// TwinCAT 3 PLC project _710_Clamping
// ProgramVersion: 3.1.4024.0
// libraries:
//   Tc2_Standard, * (Beckhoff Automation GmbH)
//   Tc2_System, * (Beckhoff Automation GmbH)
//   Tc3_Module, * (Beckhoff Automation GmbH)
//   VisuDialogs, * (System)
//   VisuSymbols,3.5.10.0,System
// project tree:
//   / GlobalTextList.TcGTLO, PlcTask.TcTTO, Visualization Manager.TcVMO (not stored)
//   GVLs/ Inputs.TcGVL, OP_Memory_DB.TcGVL, Outputs.TcGVL, ROBOT.TcGVL
//   GVLs/PARAMETER/ TRIAL.TcGVL
//   POUs/BIW/ Callblocks.TcPOU, Clamp.TcPOU, Fixture.TcPOU, MHRobot.TcPOU, ROLLER_DOOR.TcPOU, Trunion.TcPOU, Turntable.TcPOU, WeldRobot.TcPOU
//   POUs/ CLAMP_PROCESS.TcPOU, FEEDBACK_FB.TcPOU, FiX_1.TcTLO, MAIN.TcPOU, BLOCK_CALL.TcPOU, MODE_CONTROL.TcPOU, RollerDoor.TcPOU, SENSOR.TcPOU, TRUNION_FB.TcPOU, TURNTABLE_2POS.TcPOU, WELD_ROBOT.TcPOU, MH_ROBOT.TcPOU
//   VISUs/ AUTO_PROCESS.TcVIS, Visualization.TcVIS
// real-time tasks:
//   TASK PlcTask: cycle T#10ms, priority 20, ADS port 350

CONFIGURATION _710_Clamping
    RESOURCE PLC ON TwinCAT3
        TASK PlcTask(INTERVAL := T#10ms, PRIORITY := 20);
        PROGRAM MAIN WITH PlcTask : MAIN;
    END_RESOURCE
END_CONFIGURATION

// ---- GVLs/Inputs.TcGVL
{attribute 'qualified_only'}
VAR_GLOBAL



	i_CC1_Clamp_3_Sensor_HP : BOOL;
	i_CC1_Clamp_3_Sensor_WP : BOOL;
	i_CC1_Clamp_2_Sensor_HP : BOOL;
	i_CC1_Clamp_2_Sensor_WP : BOOL;
	i_CC1_Clamp_1_Sensor_HP : BOOL;
	i_CC1_Clamp_1_Sensor_WP : BOOL;
	i_CC6_Clamp_1_Sensor_HP : BOOL;
	i_CC6_Clamp_1_Sensor_WP : BOOL;
	i_CC4_Clamp_3_Sensor_HP : BOOL;
	i_CC4_Clamp_3_Sensor_WP : BOOL;
	i_PART_CONTROL_B13      : BOOL;
	i_PART_CONTROL_B27      : BOOL;
	i_PART_CONTROL_B14      : BOOL;
	i_PART_CONTROL_B28      : BOOL;
	i_CC4_Clamp_2_Sensor_HP : BOOL;
	i_CC4_Clamp_2_Sensor_WP : BOOL;
	i_CC4_Clamp_1_Sensor_HP : BOOL;
	i_CC4_Clamp_1_Sensor_WP : BOOL;
	i_CC2_Clamp_3_Sensor_HP : BOOL;
	i_CC2_Clamp_3_Sensor_WP : BOOL;
	i_PART_CONTROL_B12      : BOOL;
	i_PART_CONTROL_B26      : BOOL;
	i_PART_CONTROL_B11      : BOOL;
	i_PART_CONTROL_B25      : BOOL;
	i_PART_CONTROL_B10      : BOOL;
	i_PART_CONTROL_B24      : BOOL;
	i_CC3_Clamp_3_Sensor_HP : BOOL;
	i_CC3_Clamp_3_Sensor_WP : BOOL;
	i_CC3_Clamp_2_Sensor_HP : BOOL;
	i_CC3_Clamp_2_Sensor_WP : BOOL;
	i_CC3_Clamp_1_Sensor_HP : BOOL;
	i_CC3_Clamp_1_Sensor_WP : BOOL;
	i_PART_CONTROL_B7       : BOOL;
	i_PART_CONTROL_B21      : BOOL;
	i_PART_CONTROL_B6       : BOOL;
	i_PART_CONTROL_B20      : BOOL;
	i_PART_CONTROL_B5       : BOOL;
	i_PART_CONTROL_B19      : BOOL;
	i_PART_CONTROL_B4       : BOOL;
	i_PART_CONTROL_B18      : BOOL;
	i_PART_CONTROL_B3       : BOOL;
	i_PART_CONTROL_B17      : BOOL;
	i_PART_CONTROL_B2       : BOOL;
	i_PART_CONTROL_B16      : BOOL;
	i_CC2_Clamp_2_Sensor_HP : BOOL;
	i_CC2_Clamp_2_Sensor_WP : BOOL;
	i_CC2_Clamp_1_Sensor_HP : BOOL;
	i_CC2_Clamp_1_Sensor_WP : BOOL;
	i_PART_CONTROL_B9       : BOOL;
	i_PART_CONTROL_B23      : BOOL;
	i_PART_CONTROL_B8       : BOOL;
	i_PART_CONTROL_B22      : BOOL;
	i_CC5_Clamp_1_Sensor_HP : BOOL;
	i_CC5_Clamp_1_Sensor_WP : BOOL;
	i_PART_CONTROL_B1       : BOOL;
	i_PART_CONTROL_B15      : BOOL;
	i_Reset_PB              : BOOL;
	i_OPERATE_START_PB      : BOOL;
	i_CYCLE_START_PB        : BOOL;
    i_STOP_PB               : BOOL;
	//TT SENSOR
	i_1st_TT_Pos             : BOOL;
	i_2nd_TT_Pos             : BOOL;
	i_Drive_1_Ready         : BOOL;
	// TRUNION
	i_Drive_1_TT_Ready      : BOOL;
	i_Trunion_1st_Pos       : BOOL;
	i_Trunion_2nd_Pos       : BOOL;
	// ROLLER DOOR
	i_ROLL_DR_1_TT_Ready    : BOOL;
	i_ROLL_DR_Open_Pos_LS   : BOOL;
	i_ROLL_DR_Close_Pos_LS  : BOOL;
	//ROBOT_WELD
	Robot_Ready             : BOOL;
	Robot_Busy              : BOOL;
	Robot_Complete          : BOOL;
	Robot_Fault             : BOOL;
	PROGRAM_NUMBER          : INT;
	 //MH_ROBOT
	
	MH_Robot_Ready             : BOOL;
	MH_Robot_Busy              : BOOL;
	MH_Robot_Complete          : BOOL;
	MH_Robot_Fault             : BOOL;
	MH_PROGRAM_NUMBER          : INT;
	
	
END_VAR

// ---- GVLs/OP_Memory_DB.TcGVL
{attribute 'qualified_only'}
VAR_GLOBAL
	POWER_ON : BOOL;
    Auto_mode: BOOL;
	Manual_Mode: BOOL;
	TEMP : BOOL;
	
	
	M_CC1_CLAMPING_UNIT1_3_WP : BOOL;
	M_CC1_CLAMPING_UNIT1_3_HP : BOOL;
	M_CC2_CLAMPING_UNIT2_3_WP : BOOL;
	M_CC2_CLAMPING_UNIT2_3_HP : BOOL;
	M_CC3_CLAMPING_UNIT3_3_WP : BOOL;
	M_CC3_CLAMPING_UNIT3_3_HP : BOOL;
	M_CC4_CLAMPING_UNIT4_3_WP : BOOL;
	M_CC4_CLAMPING_UNIT4_3_HP : BOOL;
	M_CC5_CLAMPING_UNIT5_1_WP : BOOL;
	M_CC5_CLAMPING_UNIT5_1_HP : BOOL;
	M_CC6_CLAMPING_UNIT6_1_WP : BOOL;
	M_CC6_CLAMPING_UNIT6_1_HP : BOOL;
    A_CC1_CLAMPING_UNIT1_3_WP : BOOL;
	A_CC1_CLAMPING_UNIT1_3_HP : BOOL;
	A_CC2_CLAMPING_UNIT2_3_WP : BOOL;
	A_CC2_CLAMPING_UNIT2_3_HP : BOOL;
	A_CC3_CLAMPING_UNIT3_3_WP : BOOL;
	A_CC3_CLAMPING_UNIT3_3_HP : BOOL;
	A_CC4_CLAMPING_UNIT4_3_WP : BOOL;
	A_CC4_CLAMPING_UNIT4_3_HP : BOOL;
	A_CC5_CLAMPING_UNIT5_1_WP : BOOL;
	A_CC5_CLAMPING_UNIT5_1_HP : BOOL;
	A_CC6_CLAMPING_UNIT6_1_WP : BOOL;
	A_CC6_CLAMPING_UNIT6_1_HP : BOOL;
	TEMP_CC1_WP_FEEDBACK : BOOL;
	TEMP_CC1_HP_FEEDBACK : BOOL;
	TEMP_CC2_WP_FEEDBACK : BOOL;
	TEMP_CC2_HP_FEEDBACK : BOOL;
	TEMP_CC3_WP_FEEDBACK : BOOL;
	TEMP_CC3_HP_FEEDBACK : BOOL;
	TEMP_CC4_WP_FEEDBACK : BOOL;
	TEMP_CC4_HP_FEEDBACK : BOOL;
	TEMP_CC5_WP_FEEDBACK : BOOL;
	TEMP_CC5_HP_FEEDBACK : BOOL;
	TEMP_CC6_WP_FEEDBACK : BOOL;
	TEMP_CC6_HP_FEEDBACK : BOOL;
	A_FIX1_ALL_CLAMP_WORK : BOOL;
	A_FIX1_ALL_CLAMP_HOME : BOOL;
	A_FIX2_ALL_CLAMP_WORK : BOOL;
	A_FIX2_ALL_CLAMP_HOME : BOOL;
	M_FIX1_ALL_CLAMP_HOME_PB : BOOL;
	//SENSOR
	A_FIX1_PART_1ST : BOOL;
	A_FIX1_PART_2ND : BOOL;
	A_FIX1_PART_3RD : BOOL;
	A_FIX1_PART_4TH : BOOL;
	A_FIX1_PART_5TH : BOOL;
	A_FIX1_PART_6TH : BOOL;
	A_FIX2_PART_1ST : BOOL;
	A_FIX2_PART_2ND : BOOL;
	A_FIX2_PART_3RD : BOOL;
	A_FIX2_PART_4TH : BOOL;
	A_FIX2_PART_5TH : BOOL;
	A_FIX2_PART_6TH : BOOL;
	// TT POSITION
	M_1ST_POSITION_TT_CMD : BOOL;
	M_2ND_POSITION_TT_CMD : BOOL;
	A_1ST_POSITION_TT_CMD : BOOL;
	A_2ND_POSITION_TT_CMD : BOOL;
	A_FEEDBACK_TT_FWD : BOOL;
	A_FEEDBACK_TT_REV : BOOL;
	// Trunion POSITION
	A_Clamp_ok : BOOL;
	M_Fwd_POSITION : BOOL;
	M_Rev_POSITION : BOOL;
	A_Fwd_POSITION : BOOL;
	A_Rev_POSITION : BOOL;
	A_FEEDBACK_TRUNION_FWD : BOOL;
	A_FEEDBACK_TRUNION_REV : BOOL;
	//ROLLER DOOR
	M_Roll_Dr_Open  : BOOL;
	M_Roll_Dr_Close : BOOL;
	A_Open_CMD      : BOOL;
    A_Close_CMD     : BOOL;
	A_Safety_Beam : BOOL;
	A_FEEDBACK_RD_OPEN : BOOL;
	A_FEEDBACK_RD_CLOSE : BOOL;
	//ROBOT
	ROBOT_START : BOOL;
	SAFETY_OK : BOOL;
	ROBOT_JOG : BOOL;
	ROBOT_COMPLETE : BOOL;
	ROBOT_BUSY : BOOL;
	ROBOT_HOME : BOOL;
	TEMP_ROB : BOOL;
	//MH_ROBOT
	MH_ROBOT_START : BOOL;
	MH_SAFETY_OK : BOOL;
	MH_ROBOT_JOG : BOOL;
	MH_ROBOT_COMPLETE : BOOL;
	MH_ROBOT_BUSY : BOOL;
	MH_ROBOT_HOME : BOOL;
	MH_TEMP_ROB : BOOL;
	
	
	
END_VAR

// ---- GVLs/Outputs.TcGVL
{attribute 'qualified_only'}
VAR_GLOBAL


	o_CC1_CLAMPING_UNIT1_3_WP : BOOL;
	o_CC1_CLAMPING_UNIT1_3_HP : BOOL;
	o_CC2_CLAMPING_UNIT2_3_WP : BOOL;
	o_CC2_CLAMPING_UNIT2_3_HP : BOOL;
	o_CC3_CLAMPING_UNIT3_3_WP : BOOL;
	o_CC3_CLAMPING_UNIT3_3_HP : BOOL;
	o_CC4_CLAMPING_UNIT4_3_WP : BOOL;
	o_CC4_CLAMPING_UNIT4_3_HP : BOOL;
	o_CC5_CLAMPING_UNIT5_1_WP : BOOL;
	o_CC5_CLAMPING_UNIT5_1_HP : BOOL;
	o_CC6_CLAMPING_UNIT6_1_WP : BOOL;
	o_CC6_CLAMPING_UNIT6_1_HP : BOOL;
	// TURN TABLE
	o_POSITION_CW_TT : BOOL;
	o_POSITION_CCW_TT : BOOL;
	//TRUNION
	o_Motor_Fwd       : BOOL;
    o_Motor_Rev       : BOOL;
	//ROLLER DOOR
	o_ROLL_DR_Open       : BOOL;
    o_ROLL_DR_Close       : BOOL;
	//Robot
	ROBOT_START : BOOL;
	ROBOT_RESET : BOOL;
	PROGRAM_0 : BOOL;
	PROGRAM_1 : BOOL;
	PROGRAM_2 : BOOL;
	PROGRAM_3 : BOOL;
	//MH_ROBOT 
	MH_ROBOT_START : BOOL;
	MH_ROBOT_RESET : BOOL;
	MH_PROGRAM_0 : BOOL;
	MH_PROGRAM_1 : BOOL;
	MH_PROGRAM_2 : BOOL;
	MH_PROGRAM_3 : BOOL;
	O_FAULT_LAMP : BOOL;
	
END_VAR

// ---- GVLs/PARAMETER/TRIAL.TcGVL
{attribute 'qualified_only'}
VAR_GLOBAL
	
END_VAR

// ---- GVLs/ROBOT.TcGVL
{attribute 'qualified_only'}
VAR_GLOBAL
	START : BOOL;
	STOP : BOOL;
	SAFETY_OK : BOOL;
END_VAR

// ---- POUs/MAIN.TcPOU
PROGRAM MAIN
VAR
END_VAR

BLOCK_CALL();

END_PROGRAM

// ---- POUs/BLOCK_CALL.TcPOU
PROGRAM BLOCK_CALL
VAR
	CLAMP_1_DB : CLAMP_PROCESS;
	CLAMP_2_DB : CLAMP_PROCESS;
	CLAMP_3_DB : CLAMP_PROCESS;
	CLAMP_4_DB : CLAMP_PROCESS;
	CLAMP_5_DB : CLAMP_PROCESS;
	CLAMP_6_DB : CLAMP_PROCESS;
	Feedback_1_DB : Feedback_FB;
	Feedback_2_DB : Feedback_FB;
	Feedback_3_DB : Feedback_FB;
	Feedback_4_DB : Feedback_FB;
	Feedback_5_DB : Feedback_FB;
	Feedback_6_DB : Feedback_FB;
	Feedback_TT1_DB : Feedback_FB;
	Feedback_Trunion_1_DB : Feedback_FB;
	TURNTABLE_2POS_DB : TURNTABLE_2POS;
	TRUNION1_DB : TRUNION_FB;
	ROLLER_DOOR_DB : ROLLER_DOOR;
	RollerDoor_DB : RollerDoor;
    Feedback_RD1_DB : Feedback_FB;
	WELD_ROBOT_DB : WELD_ROBOT;
	MH_ROBOT_DB : MH_ROBOT;
	MODE_CONTROL_DB : MODE_CONTROL;
	SENSOR_DB : SENSOR;
END_VAR

// note: this text did not pass the execution check against the stored diagram
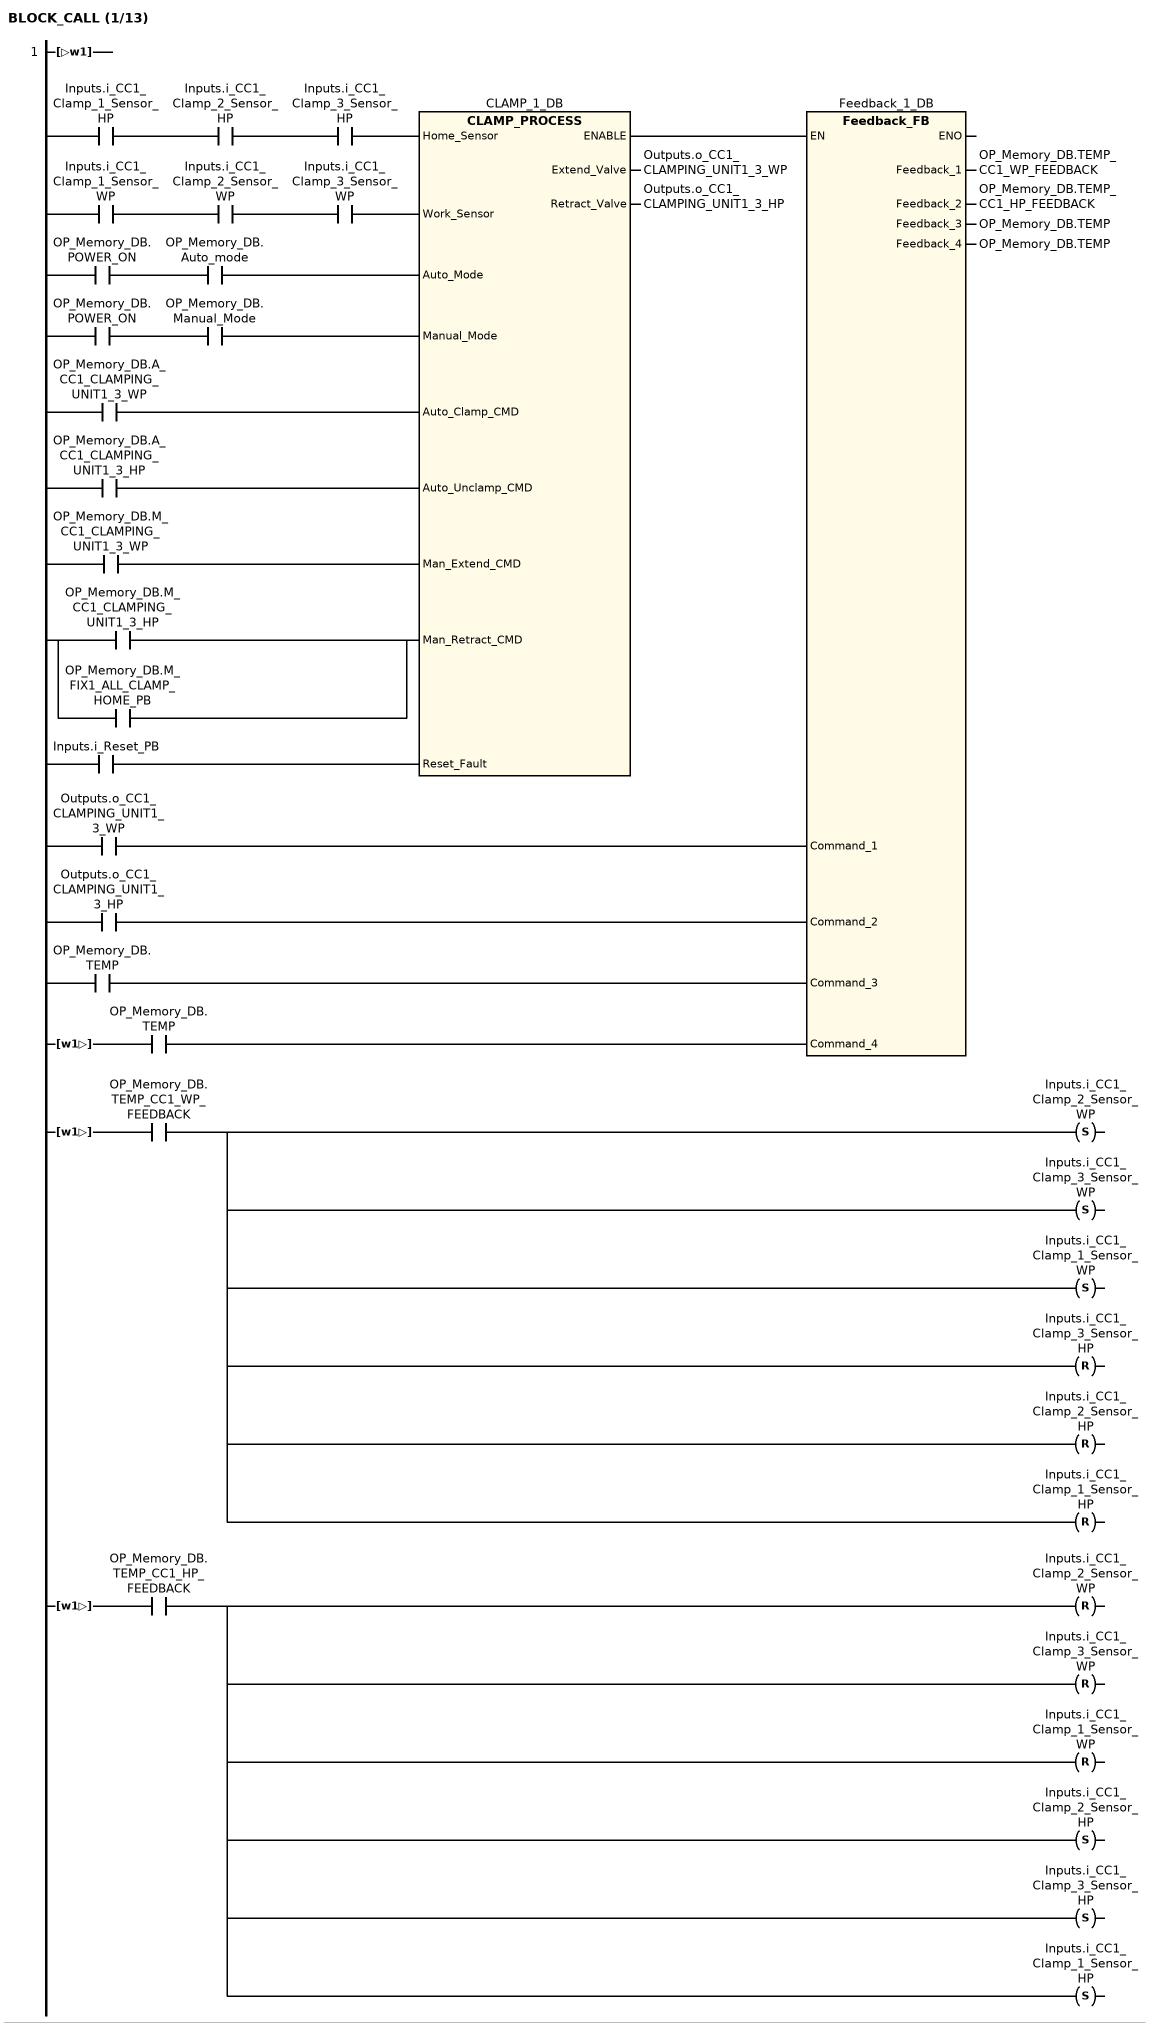
// NETWORK 1
CLAMP_1_DB(
    Home_Sensor := Inputs.i_CC1_Clamp_1_Sensor_HP AND Inputs.i_CC1_Clamp_2_Sensor_HP AND Inputs.i_CC1_Clamp_3_Sensor_HP,
    Work_Sensor := Inputs.i_CC1_Clamp_1_Sensor_WP AND Inputs.i_CC1_Clamp_2_Sensor_WP AND Inputs.i_CC1_Clamp_3_Sensor_WP,
    Auto_Mode := OP_Memory_DB.POWER_ON AND OP_Memory_DB.Auto_mode,
    Manual_Mode := OP_Memory_DB.POWER_ON AND OP_Memory_DB.Manual_Mode,
    Auto_Clamp_CMD := OP_Memory_DB.A_CC1_CLAMPING_UNIT1_3_WP,
    Auto_Unclamp_CMD := OP_Memory_DB.A_CC1_CLAMPING_UNIT1_3_HP,
    Man_Extend_CMD := OP_Memory_DB.M_CC1_CLAMPING_UNIT1_3_WP,
    Man_Retract_CMD := OP_Memory_DB.M_CC1_CLAMPING_UNIT1_3_HP OR OP_Memory_DB.M_FIX1_ALL_CLAMP_HOME_PB,
    Reset_Fault := Inputs.i_Reset_PB,
    Extend_Valve => Outputs.o_CC1_CLAMPING_UNIT1_3_WP,
    Retract_Valve => Outputs.o_CC1_CLAMPING_UNIT1_3_HP); // CLAMP_PROCESS
Feedback_1_DB(
    EN := CLAMP_1_DB.ENABLE,
    Command_1 := Outputs.o_CC1_CLAMPING_UNIT1_3_WP,
    Command_2 := Outputs.o_CC1_CLAMPING_UNIT1_3_HP,
    Command_3 := OP_Memory_DB.TEMP,
    Command_4 := OP_Memory_DB.TEMP,
    Feedback_1 => OP_Memory_DB.TEMP_CC1_WP_FEEDBACK,
    Feedback_2 => OP_Memory_DB.TEMP_CC1_HP_FEEDBACK,
    Feedback_3 => OP_Memory_DB.TEMP,
    Feedback_4 => OP_Memory_DB.TEMP); // Feedback_FB
Inputs.i_CC1_Clamp_2_Sensor_WP S= OP_Memory_DB.TEMP_CC1_WP_FEEDBACK;
Inputs.i_CC1_Clamp_3_Sensor_WP S= OP_Memory_DB.TEMP_CC1_WP_FEEDBACK;
Inputs.i_CC1_Clamp_1_Sensor_WP S= OP_Memory_DB.TEMP_CC1_WP_FEEDBACK;
Inputs.i_CC1_Clamp_3_Sensor_HP R= OP_Memory_DB.TEMP_CC1_WP_FEEDBACK;
Inputs.i_CC1_Clamp_2_Sensor_HP R= OP_Memory_DB.TEMP_CC1_WP_FEEDBACK;
Inputs.i_CC1_Clamp_1_Sensor_HP R= OP_Memory_DB.TEMP_CC1_WP_FEEDBACK;
Inputs.i_CC1_Clamp_2_Sensor_WP R= OP_Memory_DB.TEMP_CC1_HP_FEEDBACK;
Inputs.i_CC1_Clamp_3_Sensor_WP R= OP_Memory_DB.TEMP_CC1_HP_FEEDBACK;
Inputs.i_CC1_Clamp_1_Sensor_WP R= OP_Memory_DB.TEMP_CC1_HP_FEEDBACK;
Inputs.i_CC1_Clamp_2_Sensor_HP S= OP_Memory_DB.TEMP_CC1_HP_FEEDBACK;
Inputs.i_CC1_Clamp_3_Sensor_HP S= OP_Memory_DB.TEMP_CC1_HP_FEEDBACK;
Inputs.i_CC1_Clamp_1_Sensor_HP S= OP_Memory_DB.TEMP_CC1_HP_FEEDBACK;

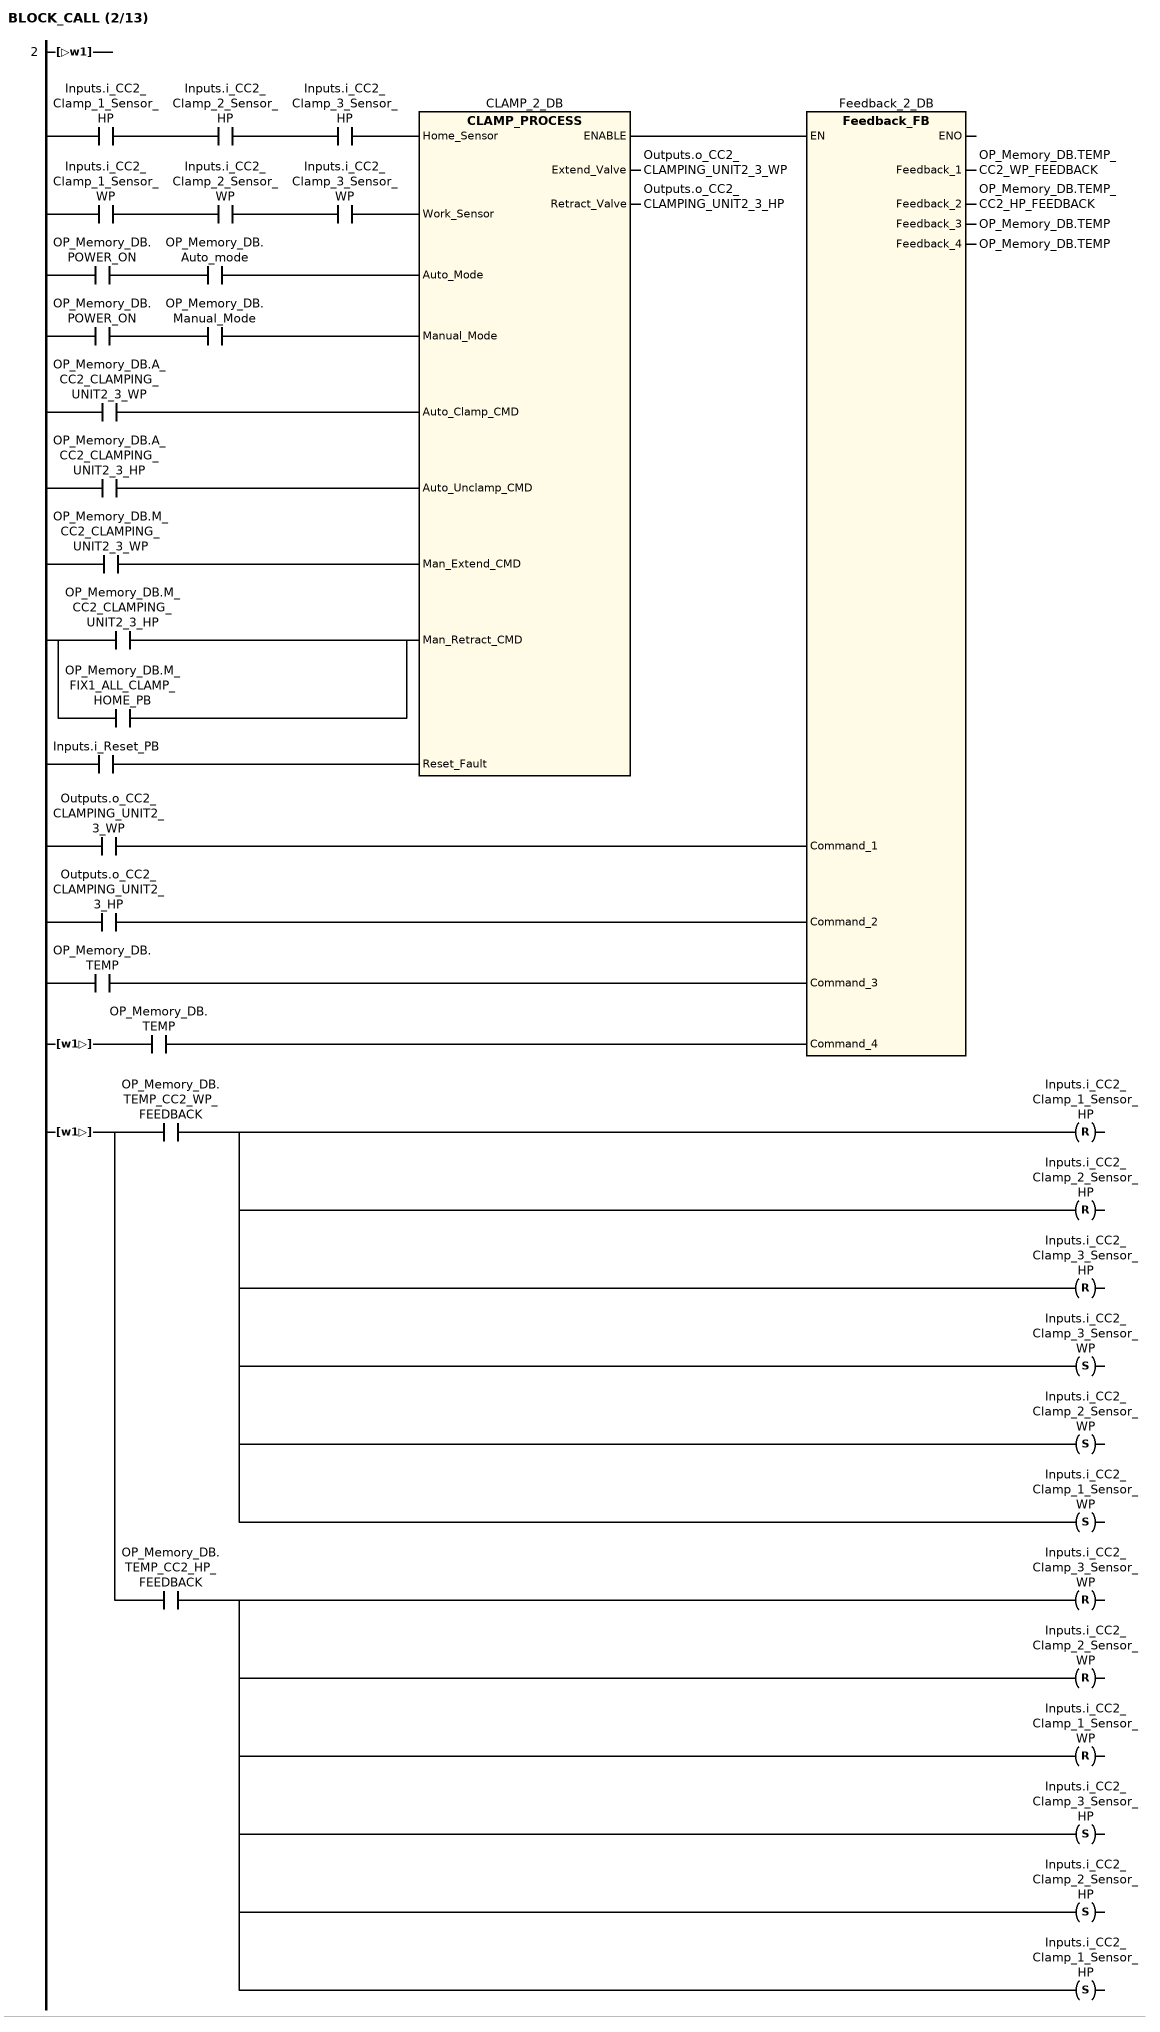
// NETWORK 2
CLAMP_2_DB(
    Home_Sensor := Inputs.i_CC2_Clamp_1_Sensor_HP AND Inputs.i_CC2_Clamp_2_Sensor_HP AND Inputs.i_CC2_Clamp_3_Sensor_HP,
    Work_Sensor := Inputs.i_CC2_Clamp_1_Sensor_WP AND Inputs.i_CC2_Clamp_2_Sensor_WP AND Inputs.i_CC2_Clamp_3_Sensor_WP,
    Auto_Mode := OP_Memory_DB.POWER_ON AND OP_Memory_DB.Auto_mode,
    Manual_Mode := OP_Memory_DB.POWER_ON AND OP_Memory_DB.Manual_Mode,
    Auto_Clamp_CMD := OP_Memory_DB.A_CC2_CLAMPING_UNIT2_3_WP,
    Auto_Unclamp_CMD := OP_Memory_DB.A_CC2_CLAMPING_UNIT2_3_HP,
    Man_Extend_CMD := OP_Memory_DB.M_CC2_CLAMPING_UNIT2_3_WP,
    Man_Retract_CMD := OP_Memory_DB.M_CC2_CLAMPING_UNIT2_3_HP OR OP_Memory_DB.M_FIX1_ALL_CLAMP_HOME_PB,
    Reset_Fault := Inputs.i_Reset_PB,
    Extend_Valve => Outputs.o_CC2_CLAMPING_UNIT2_3_WP,
    Retract_Valve => Outputs.o_CC2_CLAMPING_UNIT2_3_HP); // CLAMP_PROCESS
Feedback_2_DB(
    EN := CLAMP_2_DB.ENABLE,
    Command_1 := Outputs.o_CC2_CLAMPING_UNIT2_3_WP,
    Command_2 := Outputs.o_CC2_CLAMPING_UNIT2_3_HP,
    Command_3 := OP_Memory_DB.TEMP,
    Command_4 := OP_Memory_DB.TEMP,
    Feedback_1 => OP_Memory_DB.TEMP_CC2_WP_FEEDBACK,
    Feedback_2 => OP_Memory_DB.TEMP_CC2_HP_FEEDBACK,
    Feedback_3 => OP_Memory_DB.TEMP,
    Feedback_4 => OP_Memory_DB.TEMP); // Feedback_FB
Inputs.i_CC2_Clamp_1_Sensor_HP R= OP_Memory_DB.TEMP_CC2_WP_FEEDBACK;
Inputs.i_CC2_Clamp_2_Sensor_HP R= OP_Memory_DB.TEMP_CC2_WP_FEEDBACK;
Inputs.i_CC2_Clamp_3_Sensor_HP R= OP_Memory_DB.TEMP_CC2_WP_FEEDBACK;
Inputs.i_CC2_Clamp_3_Sensor_WP S= OP_Memory_DB.TEMP_CC2_WP_FEEDBACK;
Inputs.i_CC2_Clamp_2_Sensor_WP S= OP_Memory_DB.TEMP_CC2_WP_FEEDBACK;
Inputs.i_CC2_Clamp_1_Sensor_WP S= OP_Memory_DB.TEMP_CC2_WP_FEEDBACK;
Inputs.i_CC2_Clamp_3_Sensor_WP R= OP_Memory_DB.TEMP_CC2_HP_FEEDBACK;
Inputs.i_CC2_Clamp_2_Sensor_WP R= OP_Memory_DB.TEMP_CC2_HP_FEEDBACK;
Inputs.i_CC2_Clamp_1_Sensor_WP R= OP_Memory_DB.TEMP_CC2_HP_FEEDBACK;
Inputs.i_CC2_Clamp_3_Sensor_HP S= OP_Memory_DB.TEMP_CC2_HP_FEEDBACK;
Inputs.i_CC2_Clamp_2_Sensor_HP S= OP_Memory_DB.TEMP_CC2_HP_FEEDBACK;
Inputs.i_CC2_Clamp_1_Sensor_HP S= OP_Memory_DB.TEMP_CC2_HP_FEEDBACK;

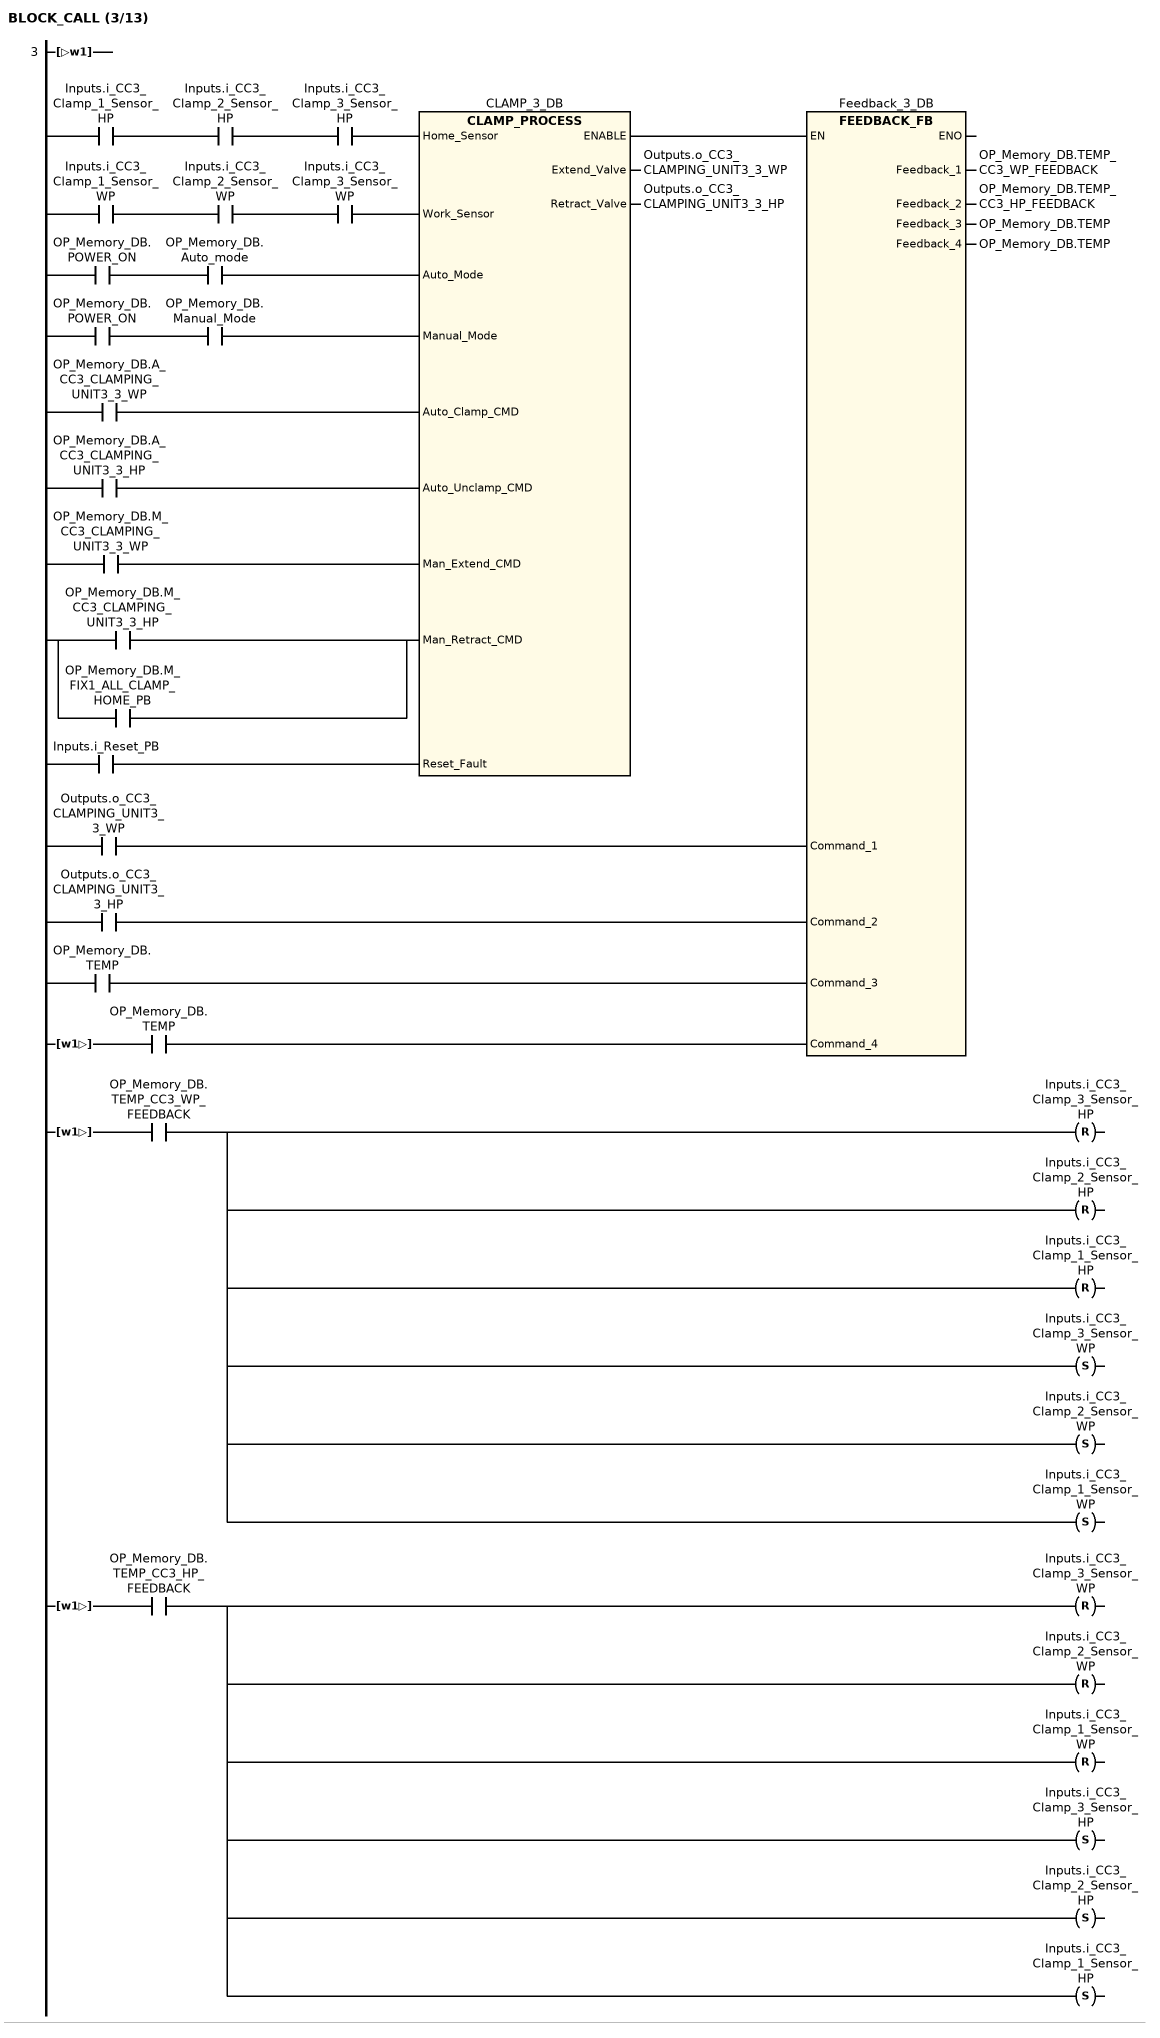
// NETWORK 3
CLAMP_3_DB(
    Home_Sensor := Inputs.i_CC3_Clamp_1_Sensor_HP AND Inputs.i_CC3_Clamp_2_Sensor_HP AND Inputs.i_CC3_Clamp_3_Sensor_HP,
    Work_Sensor := Inputs.i_CC3_Clamp_1_Sensor_WP AND Inputs.i_CC3_Clamp_2_Sensor_WP AND Inputs.i_CC3_Clamp_3_Sensor_WP,
    Auto_Mode := OP_Memory_DB.POWER_ON AND OP_Memory_DB.Auto_mode,
    Manual_Mode := OP_Memory_DB.POWER_ON AND OP_Memory_DB.Manual_Mode,
    Auto_Clamp_CMD := OP_Memory_DB.A_CC3_CLAMPING_UNIT3_3_WP,
    Auto_Unclamp_CMD := OP_Memory_DB.A_CC3_CLAMPING_UNIT3_3_HP,
    Man_Extend_CMD := OP_Memory_DB.M_CC3_CLAMPING_UNIT3_3_WP,
    Man_Retract_CMD := OP_Memory_DB.M_CC3_CLAMPING_UNIT3_3_HP OR OP_Memory_DB.M_FIX1_ALL_CLAMP_HOME_PB,
    Reset_Fault := Inputs.i_Reset_PB,
    Extend_Valve => Outputs.o_CC3_CLAMPING_UNIT3_3_WP,
    Retract_Valve => Outputs.o_CC3_CLAMPING_UNIT3_3_HP); // CLAMP_PROCESS
Feedback_3_DB(
    EN := CLAMP_3_DB.ENABLE,
    Command_1 := Outputs.o_CC3_CLAMPING_UNIT3_3_WP,
    Command_2 := Outputs.o_CC3_CLAMPING_UNIT3_3_HP,
    Command_3 := OP_Memory_DB.TEMP,
    Command_4 := OP_Memory_DB.TEMP,
    Feedback_1 => OP_Memory_DB.TEMP_CC3_WP_FEEDBACK,
    Feedback_2 => OP_Memory_DB.TEMP_CC3_HP_FEEDBACK,
    Feedback_3 => OP_Memory_DB.TEMP,
    Feedback_4 => OP_Memory_DB.TEMP); // FEEDBACK_FB
Inputs.i_CC3_Clamp_3_Sensor_HP R= OP_Memory_DB.TEMP_CC3_WP_FEEDBACK;
Inputs.i_CC3_Clamp_2_Sensor_HP R= OP_Memory_DB.TEMP_CC3_WP_FEEDBACK;
Inputs.i_CC3_Clamp_1_Sensor_HP R= OP_Memory_DB.TEMP_CC3_WP_FEEDBACK;
Inputs.i_CC3_Clamp_3_Sensor_WP S= OP_Memory_DB.TEMP_CC3_WP_FEEDBACK;
Inputs.i_CC3_Clamp_2_Sensor_WP S= OP_Memory_DB.TEMP_CC3_WP_FEEDBACK;
Inputs.i_CC3_Clamp_1_Sensor_WP S= OP_Memory_DB.TEMP_CC3_WP_FEEDBACK;
Inputs.i_CC3_Clamp_3_Sensor_WP R= OP_Memory_DB.TEMP_CC3_HP_FEEDBACK;
Inputs.i_CC3_Clamp_2_Sensor_WP R= OP_Memory_DB.TEMP_CC3_HP_FEEDBACK;
Inputs.i_CC3_Clamp_1_Sensor_WP R= OP_Memory_DB.TEMP_CC3_HP_FEEDBACK;
Inputs.i_CC3_Clamp_3_Sensor_HP S= OP_Memory_DB.TEMP_CC3_HP_FEEDBACK;
Inputs.i_CC3_Clamp_2_Sensor_HP S= OP_Memory_DB.TEMP_CC3_HP_FEEDBACK;
Inputs.i_CC3_Clamp_1_Sensor_HP S= OP_Memory_DB.TEMP_CC3_HP_FEEDBACK;

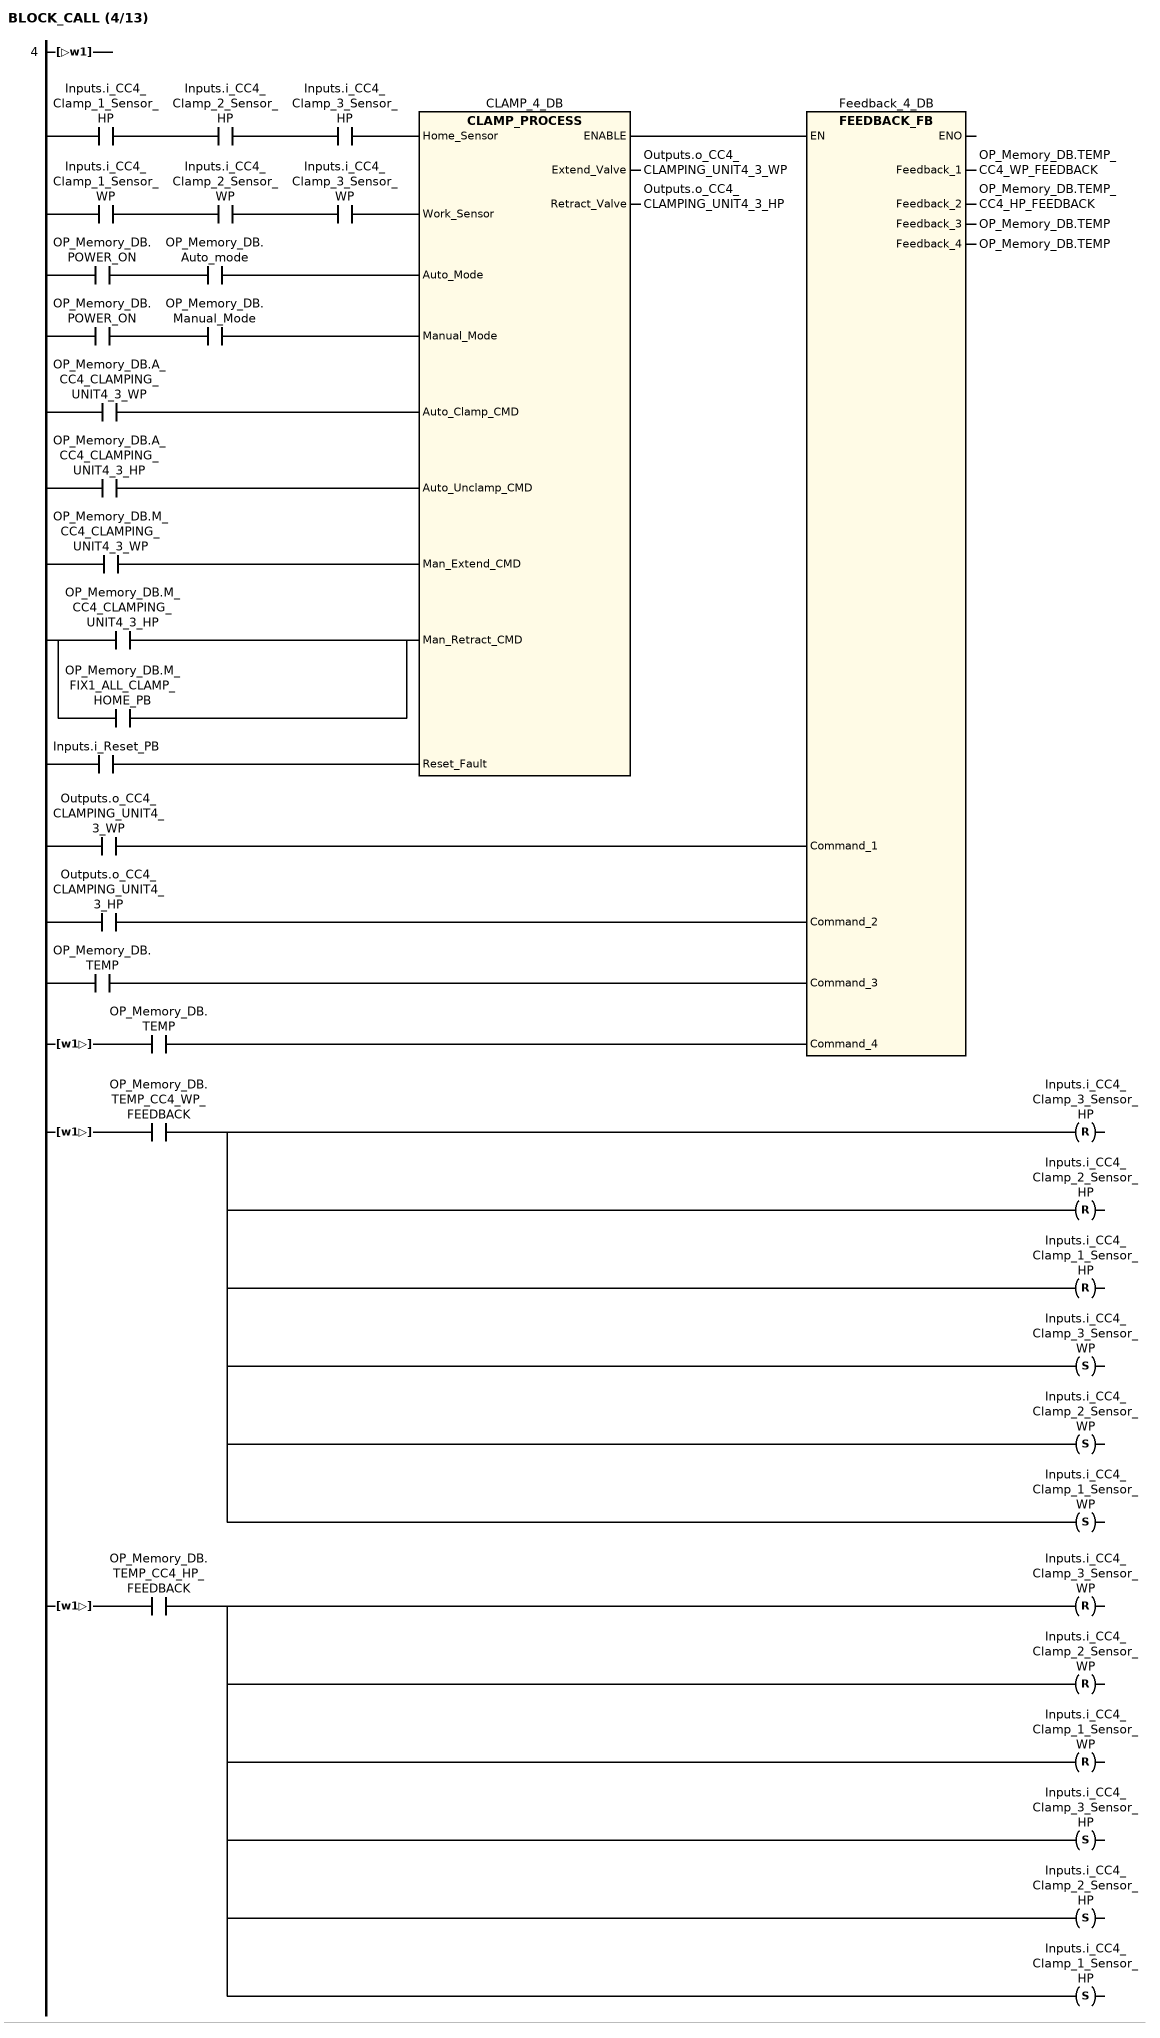
// NETWORK 4
CLAMP_4_DB(
    Home_Sensor := Inputs.i_CC4_Clamp_1_Sensor_HP AND Inputs.i_CC4_Clamp_2_Sensor_HP AND Inputs.i_CC4_Clamp_3_Sensor_HP,
    Work_Sensor := Inputs.i_CC4_Clamp_1_Sensor_WP AND Inputs.i_CC4_Clamp_2_Sensor_WP AND Inputs.i_CC4_Clamp_3_Sensor_WP,
    Auto_Mode := OP_Memory_DB.POWER_ON AND OP_Memory_DB.Auto_mode,
    Manual_Mode := OP_Memory_DB.POWER_ON AND OP_Memory_DB.Manual_Mode,
    Auto_Clamp_CMD := OP_Memory_DB.A_CC4_CLAMPING_UNIT4_3_WP,
    Auto_Unclamp_CMD := OP_Memory_DB.A_CC4_CLAMPING_UNIT4_3_HP,
    Man_Extend_CMD := OP_Memory_DB.M_CC4_CLAMPING_UNIT4_3_WP,
    Man_Retract_CMD := OP_Memory_DB.M_CC4_CLAMPING_UNIT4_3_HP OR OP_Memory_DB.M_FIX1_ALL_CLAMP_HOME_PB,
    Reset_Fault := Inputs.i_Reset_PB,
    Extend_Valve => Outputs.o_CC4_CLAMPING_UNIT4_3_WP,
    Retract_Valve => Outputs.o_CC4_CLAMPING_UNIT4_3_HP); // CLAMP_PROCESS
Feedback_4_DB(
    EN := CLAMP_4_DB.ENABLE,
    Command_1 := Outputs.o_CC4_CLAMPING_UNIT4_3_WP,
    Command_2 := Outputs.o_CC4_CLAMPING_UNIT4_3_HP,
    Command_3 := OP_Memory_DB.TEMP,
    Command_4 := OP_Memory_DB.TEMP,
    Feedback_1 => OP_Memory_DB.TEMP_CC4_WP_FEEDBACK,
    Feedback_2 => OP_Memory_DB.TEMP_CC4_HP_FEEDBACK,
    Feedback_3 => OP_Memory_DB.TEMP,
    Feedback_4 => OP_Memory_DB.TEMP); // FEEDBACK_FB
Inputs.i_CC4_Clamp_3_Sensor_HP R= OP_Memory_DB.TEMP_CC4_WP_FEEDBACK;
Inputs.i_CC4_Clamp_2_Sensor_HP R= OP_Memory_DB.TEMP_CC4_WP_FEEDBACK;
Inputs.i_CC4_Clamp_1_Sensor_HP R= OP_Memory_DB.TEMP_CC4_WP_FEEDBACK;
Inputs.i_CC4_Clamp_3_Sensor_WP S= OP_Memory_DB.TEMP_CC4_WP_FEEDBACK;
Inputs.i_CC4_Clamp_2_Sensor_WP S= OP_Memory_DB.TEMP_CC4_WP_FEEDBACK;
Inputs.i_CC4_Clamp_1_Sensor_WP S= OP_Memory_DB.TEMP_CC4_WP_FEEDBACK;
Inputs.i_CC4_Clamp_3_Sensor_WP R= OP_Memory_DB.TEMP_CC4_HP_FEEDBACK;
Inputs.i_CC4_Clamp_2_Sensor_WP R= OP_Memory_DB.TEMP_CC4_HP_FEEDBACK;
Inputs.i_CC4_Clamp_1_Sensor_WP R= OP_Memory_DB.TEMP_CC4_HP_FEEDBACK;
Inputs.i_CC4_Clamp_3_Sensor_HP S= OP_Memory_DB.TEMP_CC4_HP_FEEDBACK;
Inputs.i_CC4_Clamp_2_Sensor_HP S= OP_Memory_DB.TEMP_CC4_HP_FEEDBACK;
Inputs.i_CC4_Clamp_1_Sensor_HP S= OP_Memory_DB.TEMP_CC4_HP_FEEDBACK;

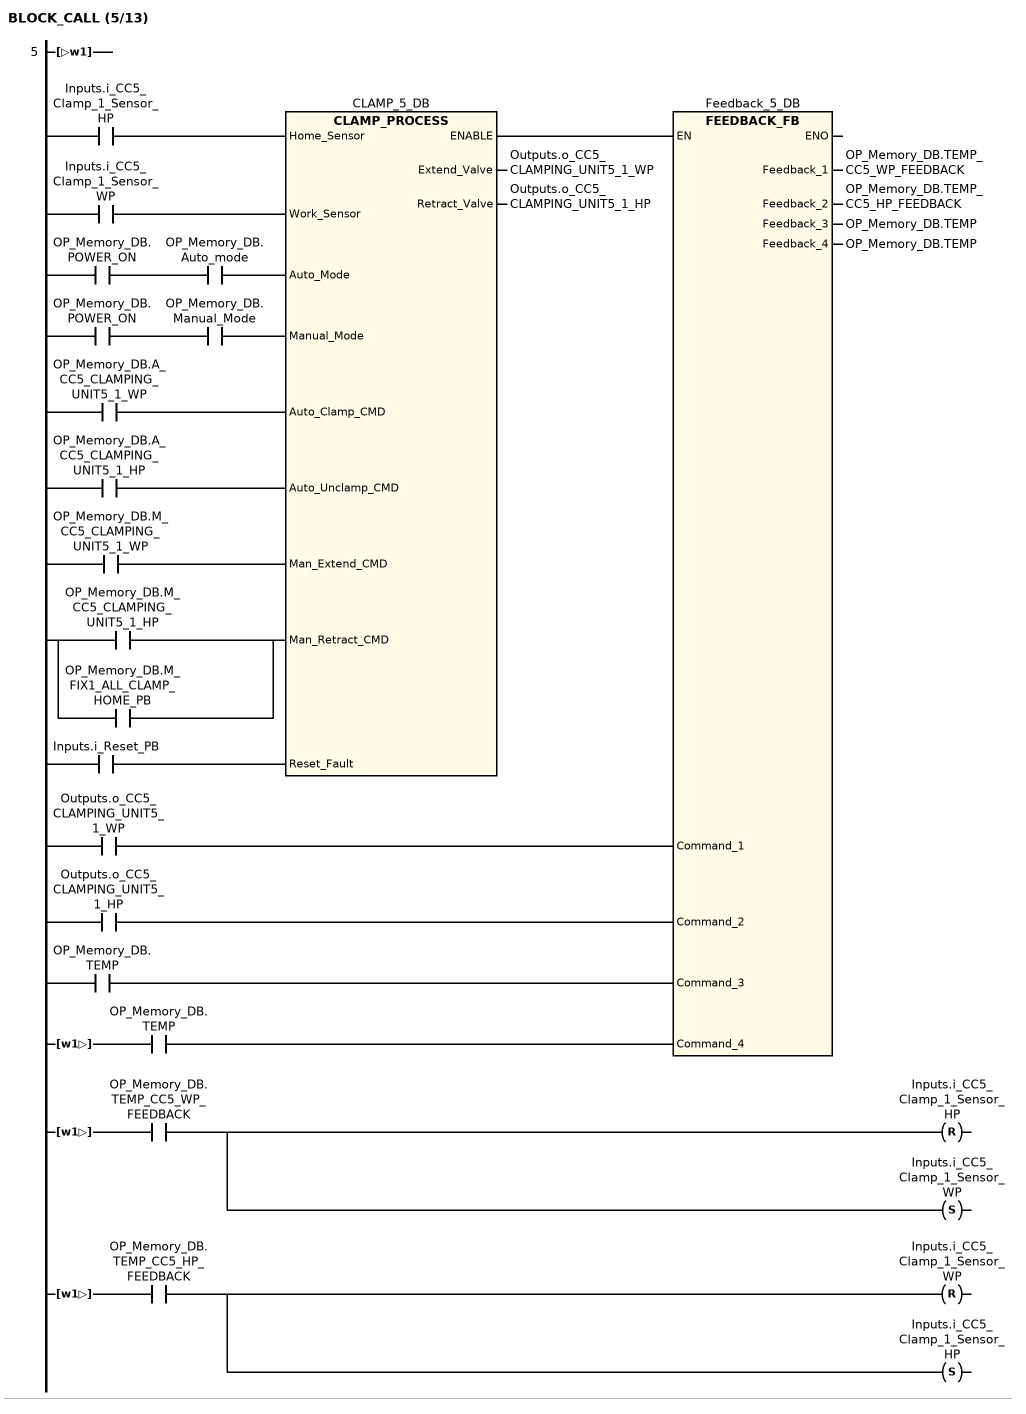
// NETWORK 5
CLAMP_5_DB(
    Home_Sensor := Inputs.i_CC5_Clamp_1_Sensor_HP,
    Work_Sensor := Inputs.i_CC5_Clamp_1_Sensor_WP,
    Auto_Mode := OP_Memory_DB.POWER_ON AND OP_Memory_DB.Auto_mode,
    Manual_Mode := OP_Memory_DB.POWER_ON AND OP_Memory_DB.Manual_Mode,
    Auto_Clamp_CMD := OP_Memory_DB.A_CC5_CLAMPING_UNIT5_1_WP,
    Auto_Unclamp_CMD := OP_Memory_DB.A_CC5_CLAMPING_UNIT5_1_HP,
    Man_Extend_CMD := OP_Memory_DB.M_CC5_CLAMPING_UNIT5_1_WP,
    Man_Retract_CMD := OP_Memory_DB.M_CC5_CLAMPING_UNIT5_1_HP OR OP_Memory_DB.M_FIX1_ALL_CLAMP_HOME_PB,
    Reset_Fault := Inputs.i_Reset_PB,
    Extend_Valve => Outputs.o_CC5_CLAMPING_UNIT5_1_WP,
    Retract_Valve => Outputs.o_CC5_CLAMPING_UNIT5_1_HP); // CLAMP_PROCESS
Feedback_5_DB(
    EN := CLAMP_5_DB.ENABLE,
    Command_1 := Outputs.o_CC5_CLAMPING_UNIT5_1_WP,
    Command_2 := Outputs.o_CC5_CLAMPING_UNIT5_1_HP,
    Command_3 := OP_Memory_DB.TEMP,
    Command_4 := OP_Memory_DB.TEMP,
    Feedback_1 => OP_Memory_DB.TEMP_CC5_WP_FEEDBACK,
    Feedback_2 => OP_Memory_DB.TEMP_CC5_HP_FEEDBACK,
    Feedback_3 => OP_Memory_DB.TEMP,
    Feedback_4 => OP_Memory_DB.TEMP); // FEEDBACK_FB
Inputs.i_CC5_Clamp_1_Sensor_HP R= OP_Memory_DB.TEMP_CC5_WP_FEEDBACK;
Inputs.i_CC5_Clamp_1_Sensor_WP S= OP_Memory_DB.TEMP_CC5_WP_FEEDBACK;
Inputs.i_CC5_Clamp_1_Sensor_WP R= OP_Memory_DB.TEMP_CC5_HP_FEEDBACK;
Inputs.i_CC5_Clamp_1_Sensor_HP S= OP_Memory_DB.TEMP_CC5_HP_FEEDBACK;

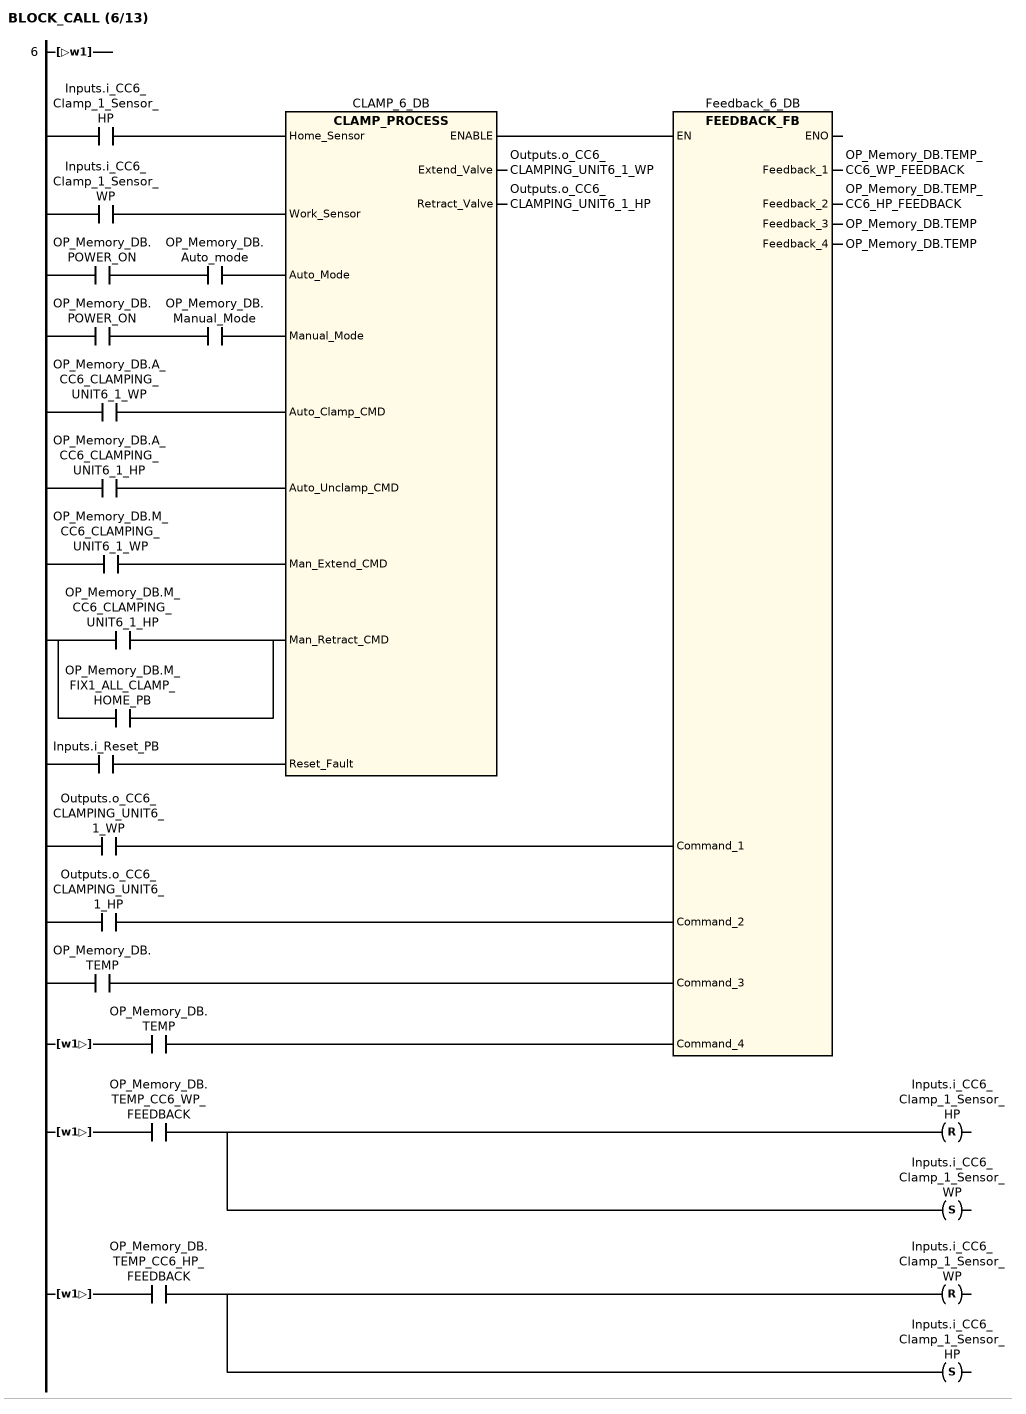
// NETWORK 6
CLAMP_6_DB(
    Home_Sensor := Inputs.i_CC6_Clamp_1_Sensor_HP,
    Work_Sensor := Inputs.i_CC6_Clamp_1_Sensor_WP,
    Auto_Mode := OP_Memory_DB.POWER_ON AND OP_Memory_DB.Auto_mode,
    Manual_Mode := OP_Memory_DB.POWER_ON AND OP_Memory_DB.Manual_Mode,
    Auto_Clamp_CMD := OP_Memory_DB.A_CC6_CLAMPING_UNIT6_1_WP,
    Auto_Unclamp_CMD := OP_Memory_DB.A_CC6_CLAMPING_UNIT6_1_HP,
    Man_Extend_CMD := OP_Memory_DB.M_CC6_CLAMPING_UNIT6_1_WP,
    Man_Retract_CMD := OP_Memory_DB.M_CC6_CLAMPING_UNIT6_1_HP OR OP_Memory_DB.M_FIX1_ALL_CLAMP_HOME_PB,
    Reset_Fault := Inputs.i_Reset_PB,
    Extend_Valve => Outputs.o_CC6_CLAMPING_UNIT6_1_WP,
    Retract_Valve => Outputs.o_CC6_CLAMPING_UNIT6_1_HP); // CLAMP_PROCESS
Feedback_6_DB(
    EN := CLAMP_6_DB.ENABLE,
    Command_1 := Outputs.o_CC6_CLAMPING_UNIT6_1_WP,
    Command_2 := Outputs.o_CC6_CLAMPING_UNIT6_1_HP,
    Command_3 := OP_Memory_DB.TEMP,
    Command_4 := OP_Memory_DB.TEMP,
    Feedback_1 => OP_Memory_DB.TEMP_CC6_WP_FEEDBACK,
    Feedback_2 => OP_Memory_DB.TEMP_CC6_HP_FEEDBACK,
    Feedback_3 => OP_Memory_DB.TEMP,
    Feedback_4 => OP_Memory_DB.TEMP); // FEEDBACK_FB
Inputs.i_CC6_Clamp_1_Sensor_HP R= OP_Memory_DB.TEMP_CC6_WP_FEEDBACK;
Inputs.i_CC6_Clamp_1_Sensor_WP S= OP_Memory_DB.TEMP_CC6_WP_FEEDBACK;
Inputs.i_CC6_Clamp_1_Sensor_WP R= OP_Memory_DB.TEMP_CC6_HP_FEEDBACK;
Inputs.i_CC6_Clamp_1_Sensor_HP S= OP_Memory_DB.TEMP_CC6_HP_FEEDBACK;

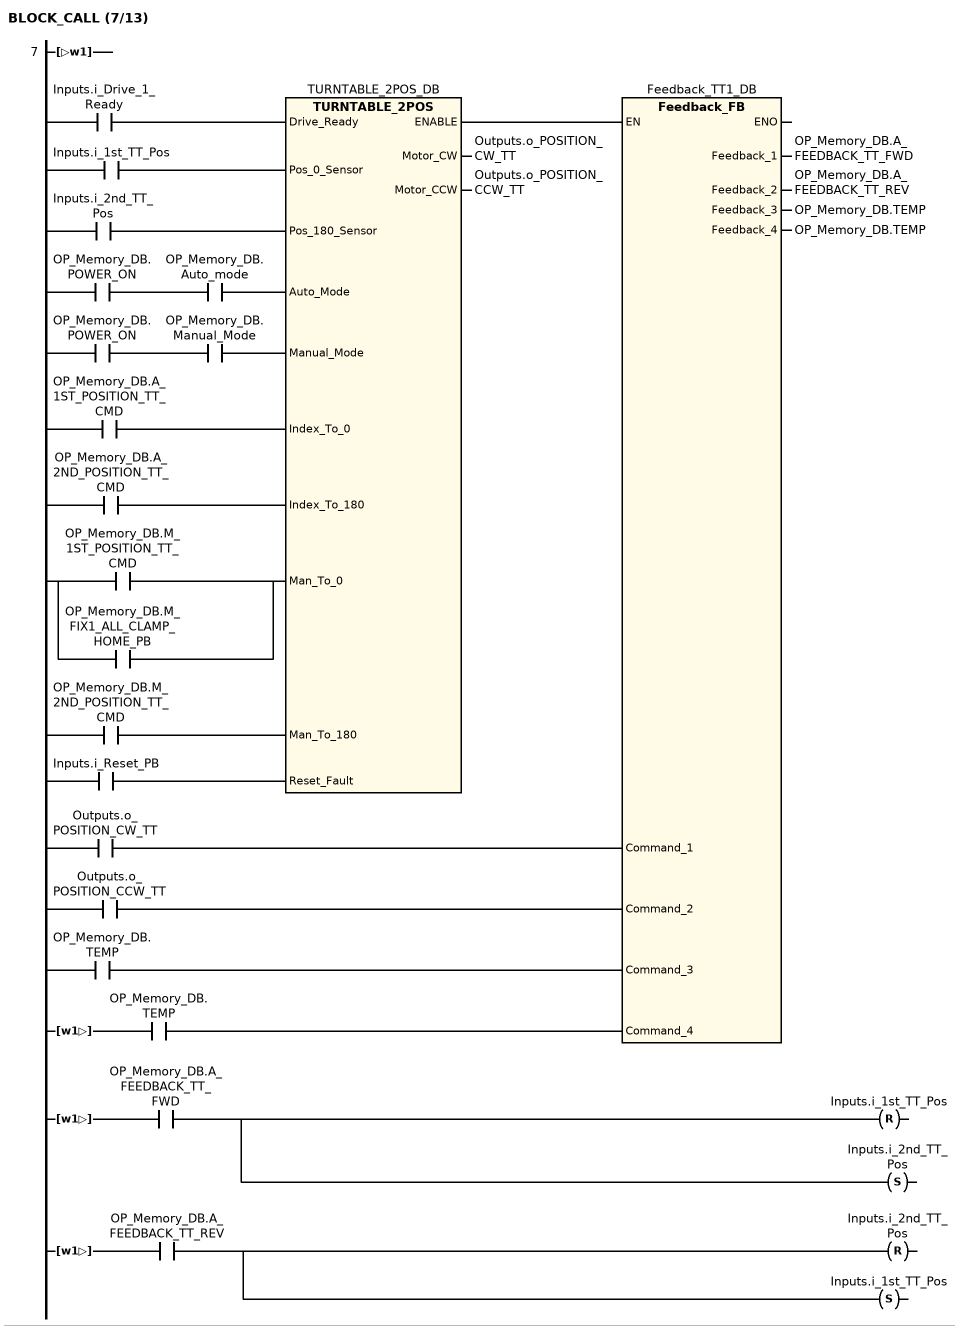
// NETWORK 7
TURNTABLE_2POS_DB(
    Drive_Ready := Inputs.i_Drive_1_Ready,
    Pos_0_Sensor := Inputs.i_1st_TT_Pos,
    Pos_180_Sensor := Inputs.i_2nd_TT_Pos,
    Auto_Mode := OP_Memory_DB.POWER_ON AND OP_Memory_DB.Auto_mode,
    Manual_Mode := OP_Memory_DB.POWER_ON AND OP_Memory_DB.Manual_Mode,
    Index_To_0 := OP_Memory_DB.A_1ST_POSITION_TT_CMD,
    Index_To_180 := OP_Memory_DB.A_2ND_POSITION_TT_CMD,
    Man_To_0 := OP_Memory_DB.M_1ST_POSITION_TT_CMD OR OP_Memory_DB.M_FIX1_ALL_CLAMP_HOME_PB,
    Man_To_180 := OP_Memory_DB.M_2ND_POSITION_TT_CMD,
    Reset_Fault := Inputs.i_Reset_PB,
    Motor_CW => Outputs.o_POSITION_CW_TT,
    Motor_CCW => Outputs.o_POSITION_CCW_TT); // TURNTABLE_2POS
Feedback_TT1_DB(
    EN := TURNTABLE_2POS_DB.ENABLE,
    Command_1 := Outputs.o_POSITION_CW_TT,
    Command_2 := Outputs.o_POSITION_CCW_TT,
    Command_3 := OP_Memory_DB.TEMP,
    Command_4 := OP_Memory_DB.TEMP,
    Feedback_1 => OP_Memory_DB.A_FEEDBACK_TT_FWD,
    Feedback_2 => OP_Memory_DB.A_FEEDBACK_TT_REV,
    Feedback_3 => OP_Memory_DB.TEMP,
    Feedback_4 => OP_Memory_DB.TEMP); // Feedback_FB
Inputs.i_1st_TT_Pos R= OP_Memory_DB.A_FEEDBACK_TT_FWD;
Inputs.i_2nd_TT_Pos S= OP_Memory_DB.A_FEEDBACK_TT_FWD;
Inputs.i_2nd_TT_Pos R= OP_Memory_DB.A_FEEDBACK_TT_REV;
Inputs.i_1st_TT_Pos S= OP_Memory_DB.A_FEEDBACK_TT_REV;

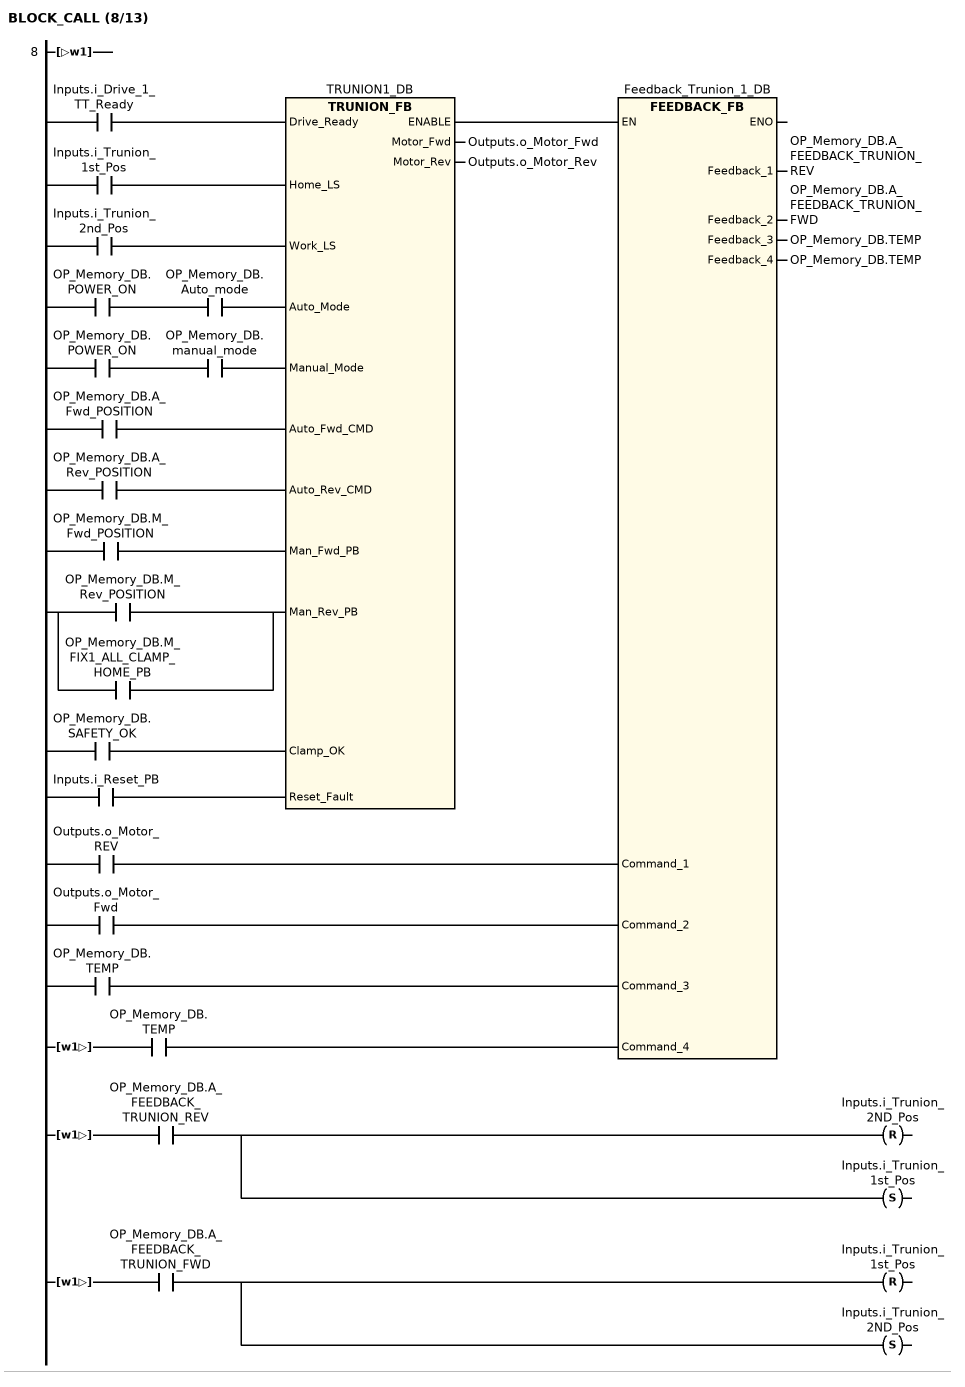
// NETWORK 8
TRUNION1_DB(
    Drive_Ready := Inputs.i_Drive_1_TT_Ready,
    Home_LS := Inputs.i_Trunion_1st_Pos,
    Work_LS := Inputs.i_Trunion_2nd_Pos,
    Auto_Mode := OP_Memory_DB.POWER_ON AND OP_Memory_DB.Auto_mode,
    Manual_Mode := OP_Memory_DB.POWER_ON AND OP_Memory_DB.manual_mode,
    Auto_Fwd_CMD := OP_Memory_DB.A_Fwd_POSITION,
    Auto_Rev_CMD := OP_Memory_DB.A_Rev_POSITION,
    Man_Fwd_PB := OP_Memory_DB.M_Fwd_POSITION,
    Man_Rev_PB := OP_Memory_DB.M_Rev_POSITION OR OP_Memory_DB.M_FIX1_ALL_CLAMP_HOME_PB,
    Clamp_OK := OP_Memory_DB.SAFETY_OK,
    Reset_Fault := Inputs.i_Reset_PB,
    Motor_Fwd => Outputs.o_Motor_Fwd,
    Motor_Rev => Outputs.o_Motor_Rev); // TRUNION_FB
Feedback_Trunion_1_DB(
    EN := TRUNION1_DB.ENABLE,
    Command_1 := Outputs.o_Motor_REV,
    Command_2 := Outputs.o_Motor_Fwd,
    Command_3 := OP_Memory_DB.TEMP,
    Command_4 := OP_Memory_DB.TEMP,
    Feedback_1 => OP_Memory_DB.A_FEEDBACK_TRUNION_REV,
    Feedback_2 => OP_Memory_DB.A_FEEDBACK_TRUNION_FWD,
    Feedback_3 => OP_Memory_DB.TEMP,
    Feedback_4 => OP_Memory_DB.TEMP); // FEEDBACK_FB
Inputs.i_Trunion_2ND_Pos R= OP_Memory_DB.A_FEEDBACK_TRUNION_REV;
Inputs.i_Trunion_1st_Pos S= OP_Memory_DB.A_FEEDBACK_TRUNION_REV;
Inputs.i_Trunion_1st_Pos R= OP_Memory_DB.A_FEEDBACK_TRUNION_FWD;
Inputs.i_Trunion_2ND_Pos S= OP_Memory_DB.A_FEEDBACK_TRUNION_FWD;

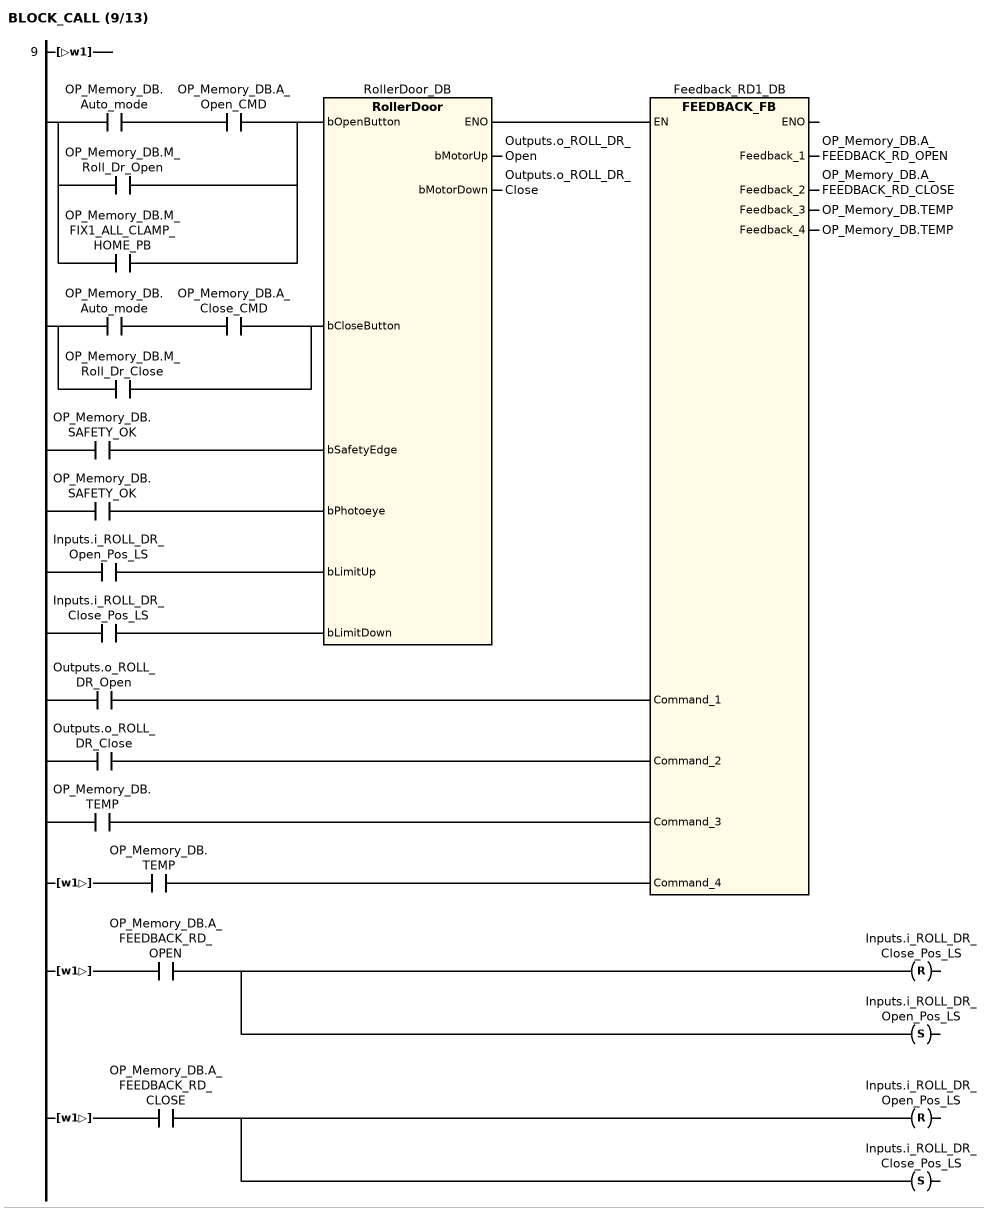
// NETWORK 9
RollerDoor_DB(
    bOpenButton := OP_Memory_DB.Auto_mode AND OP_Memory_DB.A_Open_CMD OR OP_Memory_DB.M_Roll_Dr_Open OR OP_Memory_DB.M_FIX1_ALL_CLAMP_HOME_PB,
    bCloseButton := OP_Memory_DB.Auto_mode AND OP_Memory_DB.A_Close_CMD OR OP_Memory_DB.M_Roll_Dr_Close,
    bSafetyEdge := OP_Memory_DB.SAFETY_OK,
    bPhotoeye := OP_Memory_DB.SAFETY_OK,
    bLimitUp := Inputs.i_ROLL_DR_Open_Pos_LS,
    bLimitDown := Inputs.i_ROLL_DR_Close_Pos_LS,
    bMotorUp => Outputs.o_ROLL_DR_Open,
    bMotorDown => Outputs.o_ROLL_DR_Close); // RollerDoor
Feedback_RD1_DB(
    EN := TRUE,
    Command_1 := Outputs.o_ROLL_DR_Open,
    Command_2 := Outputs.o_ROLL_DR_Close,
    Command_3 := OP_Memory_DB.TEMP,
    Command_4 := OP_Memory_DB.TEMP,
    Feedback_1 => OP_Memory_DB.A_FEEDBACK_RD_OPEN,
    Feedback_2 => OP_Memory_DB.A_FEEDBACK_RD_CLOSE,
    Feedback_3 => OP_Memory_DB.TEMP,
    Feedback_4 => OP_Memory_DB.TEMP); // FEEDBACK_FB
Inputs.i_ROLL_DR_Close_Pos_LS R= OP_Memory_DB.A_FEEDBACK_RD_OPEN;
Inputs.i_ROLL_DR_Open_Pos_LS S= OP_Memory_DB.A_FEEDBACK_RD_OPEN;
Inputs.i_ROLL_DR_Open_Pos_LS R= OP_Memory_DB.A_FEEDBACK_RD_CLOSE;
Inputs.i_ROLL_DR_Close_Pos_LS S= OP_Memory_DB.A_FEEDBACK_RD_CLOSE;

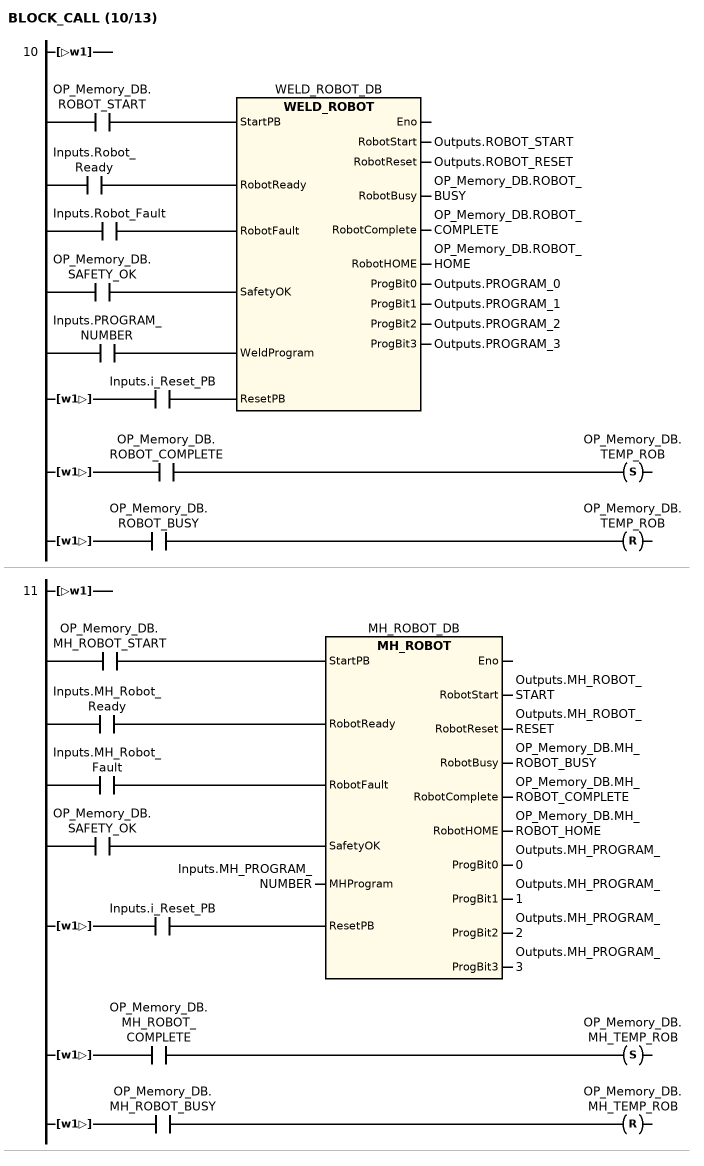
// NETWORK 10
WELD_ROBOT_DB(
    StartPB := OP_Memory_DB.ROBOT_START,
    RobotReady := Inputs.Robot_Ready,
    RobotFault := Inputs.Robot_Fault,
    SafetyOK := OP_Memory_DB.SAFETY_OK,
    WeldProgram := Inputs.PROGRAM_NUMBER,
    ResetPB := Inputs.i_Reset_PB,
    RobotStart => Outputs.ROBOT_START,
    RobotReset => Outputs.ROBOT_RESET,
    RobotBusy => OP_Memory_DB.ROBOT_BUSY,
    RobotComplete => OP_Memory_DB.ROBOT_COMPLETE,
    RobotHOME => OP_Memory_DB.ROBOT_HOME,
    ProgBit0 => Outputs.PROGRAM_0,
    ProgBit1 => Outputs.PROGRAM_1,
    ProgBit2 => Outputs.PROGRAM_2,
    ProgBit3 => Outputs.PROGRAM_3); // WELD_ROBOT
OP_Memory_DB.TEMP_ROB S= OP_Memory_DB.ROBOT_COMPLETE;
OP_Memory_DB.TEMP_ROB R= OP_Memory_DB.ROBOT_BUSY;

// NETWORK 11
MH_ROBOT_DB(
    StartPB := OP_Memory_DB.MH_ROBOT_START,
    RobotReady := Inputs.MH_Robot_Ready,
    RobotFault := Inputs.MH_Robot_Fault,
    SafetyOK := OP_Memory_DB.SAFETY_OK,
    MHProgram := Inputs.MH_PROGRAM_NUMBER,
    ResetPB := Inputs.i_Reset_PB,
    RobotStart => Outputs.MH_ROBOT_START,
    RobotReset => Outputs.MH_ROBOT_RESET,
    RobotBusy => OP_Memory_DB.MH_ROBOT_BUSY,
    RobotComplete => OP_Memory_DB.MH_ROBOT_COMPLETE,
    RobotHOME => OP_Memory_DB.MH_ROBOT_HOME,
    ProgBit0 => Outputs.MH_PROGRAM_0,
    ProgBit1 => Outputs.MH_PROGRAM_1,
    ProgBit2 => Outputs.MH_PROGRAM_2,
    ProgBit3 => Outputs.MH_PROGRAM_3); // MH_ROBOT
OP_Memory_DB.MH_TEMP_ROB S= OP_Memory_DB.MH_ROBOT_COMPLETE;
OP_Memory_DB.MH_TEMP_ROB R= OP_Memory_DB.MH_ROBOT_BUSY;

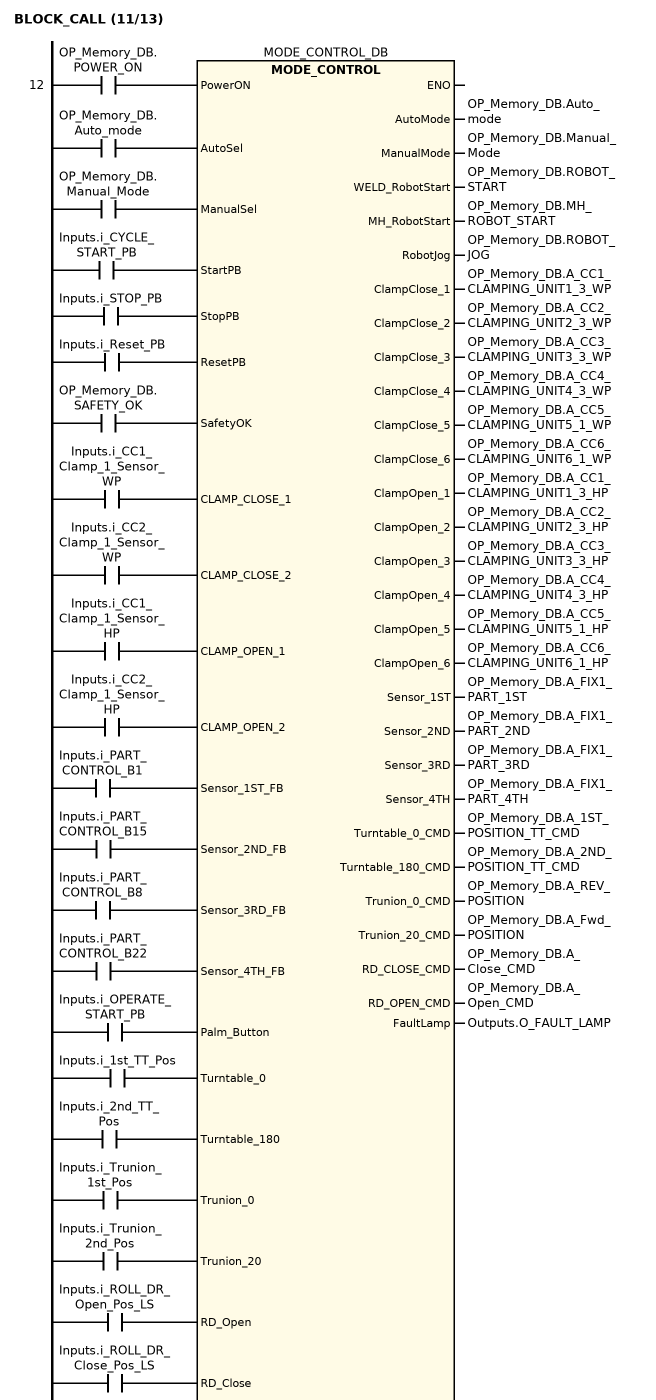
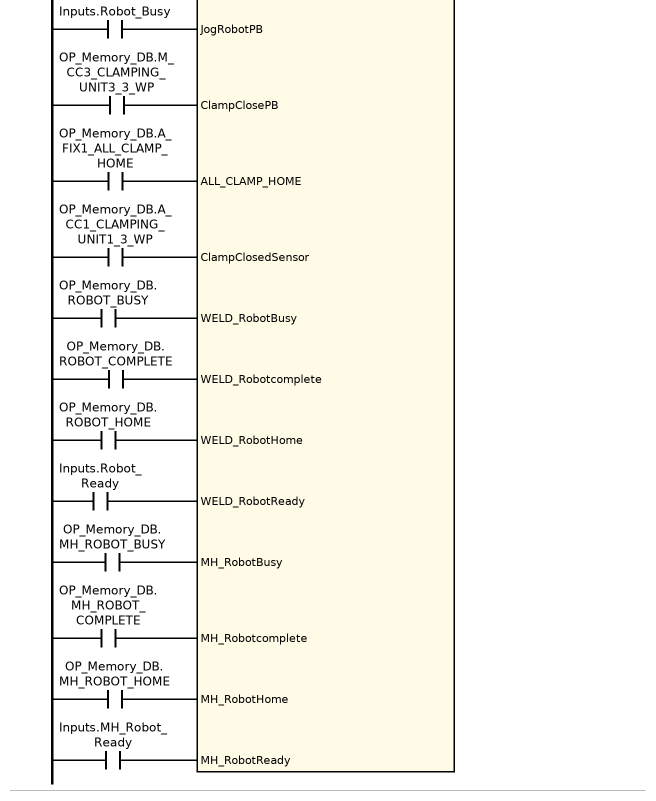
// NETWORK 12
MODE_CONTROL_DB(
    PowerON := OP_Memory_DB.POWER_ON,
    AutoSel := OP_Memory_DB.Auto_mode,
    ManualSel := OP_Memory_DB.Manual_Mode,
    StartPB := Inputs.i_CYCLE_START_PB,
    StopPB := Inputs.i_STOP_PB,
    ResetPB := Inputs.i_Reset_PB,
    SafetyOK := OP_Memory_DB.SAFETY_OK,
    CLAMP_CLOSE_1 := Inputs.i_CC1_Clamp_1_Sensor_WP,
    CLAMP_CLOSE_2 := Inputs.i_CC2_Clamp_1_Sensor_WP,
    CLAMP_OPEN_1 := Inputs.i_CC1_Clamp_1_Sensor_HP,
    CLAMP_OPEN_2 := Inputs.i_CC2_Clamp_1_Sensor_HP,
    Sensor_1ST_FB := Inputs.i_PART_CONTROL_B1,
    Sensor_2ND_FB := Inputs.i_PART_CONTROL_B15,
    Sensor_3RD_FB := Inputs.i_PART_CONTROL_B8,
    Sensor_4TH_FB := Inputs.i_PART_CONTROL_B22,
    Palm_Button := Inputs.i_OPERATE_START_PB,
    Turntable_0 := Inputs.i_1st_TT_Pos,
    Turntable_180 := Inputs.i_2nd_TT_Pos,
    Trunion_0 := Inputs.i_Trunion_1st_Pos,
    Trunion_20 := Inputs.i_Trunion_2nd_Pos,
    RD_Open := Inputs.i_ROLL_DR_Open_Pos_LS,
    RD_Close := Inputs.i_ROLL_DR_Close_Pos_LS,
    JogRobotPB := Inputs.Robot_Busy,
    ClampClosePB := OP_Memory_DB.M_CC3_CLAMPING_UNIT3_3_WP,
    ALL_CLAMP_HOME := OP_Memory_DB.A_FIX1_ALL_CLAMP_HOME,
    ClampClosedSensor := OP_Memory_DB.A_CC1_CLAMPING_UNIT1_3_WP,
    WELD_RobotBusy := OP_Memory_DB.ROBOT_BUSY,
    WELD_Robotcomplete := OP_Memory_DB.ROBOT_COMPLETE,
    WELD_RobotHome := OP_Memory_DB.ROBOT_HOME,
    WELD_RobotReady := Inputs.Robot_Ready,
    MH_RobotBusy := OP_Memory_DB.MH_ROBOT_BUSY,
    MH_Robotcomplete := OP_Memory_DB.MH_ROBOT_COMPLETE,
    MH_RobotHome := OP_Memory_DB.MH_ROBOT_HOME,
    MH_RobotReady := Inputs.MH_Robot_Ready,
    AutoMode => OP_Memory_DB.Auto_mode,
    ManualMode => OP_Memory_DB.Manual_Mode,
    WELD_RobotStart => OP_Memory_DB.ROBOT_START,
    MH_RobotStart => OP_Memory_DB.MH_ROBOT_START,
    RobotJog => OP_Memory_DB.ROBOT_JOG,
    ClampClose_1 => OP_Memory_DB.A_CC1_CLAMPING_UNIT1_3_WP,
    ClampClose_2 => OP_Memory_DB.A_CC2_CLAMPING_UNIT2_3_WP,
    ClampClose_3 => OP_Memory_DB.A_CC3_CLAMPING_UNIT3_3_WP,
    ClampClose_4 => OP_Memory_DB.A_CC4_CLAMPING_UNIT4_3_WP,
    ClampClose_5 => OP_Memory_DB.A_CC5_CLAMPING_UNIT5_1_WP,
    ClampClose_6 => OP_Memory_DB.A_CC6_CLAMPING_UNIT6_1_WP,
    ClampOpen_1 => OP_Memory_DB.A_CC1_CLAMPING_UNIT1_3_HP,
    ClampOpen_2 => OP_Memory_DB.A_CC2_CLAMPING_UNIT2_3_HP,
    ClampOpen_3 => OP_Memory_DB.A_CC3_CLAMPING_UNIT3_3_HP,
    ClampOpen_4 => OP_Memory_DB.A_CC4_CLAMPING_UNIT4_3_HP,
    ClampOpen_5 => OP_Memory_DB.A_CC5_CLAMPING_UNIT5_1_HP,
    ClampOpen_6 => OP_Memory_DB.A_CC6_CLAMPING_UNIT6_1_HP,
    Sensor_1ST => OP_Memory_DB.A_FIX1_PART_1ST,
    Sensor_2ND => OP_Memory_DB.A_FIX1_PART_2ND,
    Sensor_3RD => OP_Memory_DB.A_FIX1_PART_3RD,
    Sensor_4TH => OP_Memory_DB.A_FIX1_PART_4TH,
    Turntable_0_CMD => OP_Memory_DB.A_1ST_POSITION_TT_CMD,
    Turntable_180_CMD => OP_Memory_DB.A_2ND_POSITION_TT_CMD,
    Trunion_0_CMD => OP_Memory_DB.A_REV_POSITION,
    Trunion_20_CMD => OP_Memory_DB.A_Fwd_POSITION,
    RD_CLOSE_CMD => OP_Memory_DB.A_Close_CMD,
    RD_OPEN_CMD => OP_Memory_DB.A_Open_CMD,
    FaultLamp => Outputs.O_FAULT_LAMP); // MODE_CONTROL

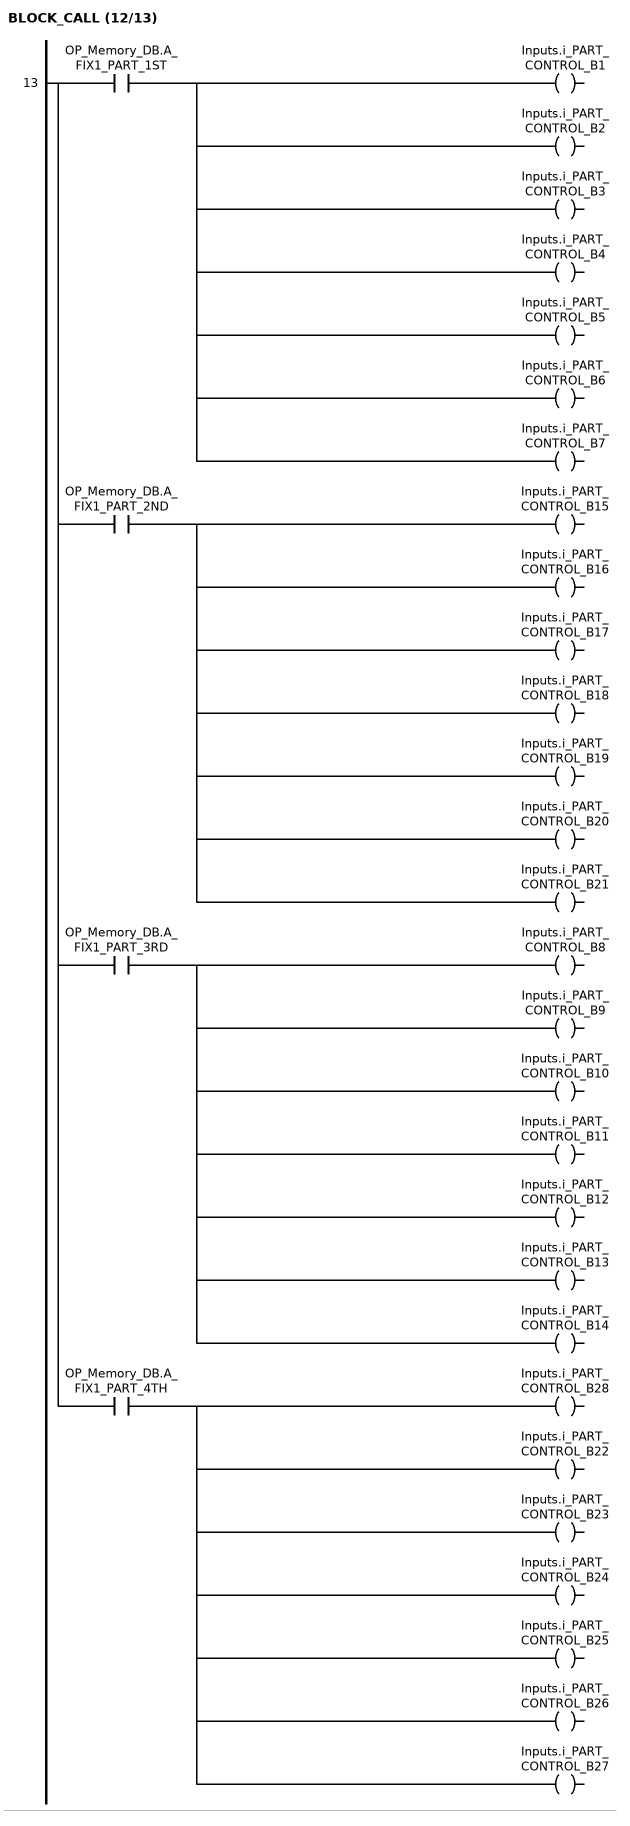
// NETWORK 13
Inputs.i_PART_CONTROL_B1 := OP_Memory_DB.A_FIX1_PART_1ST;
Inputs.i_PART_CONTROL_B2 := OP_Memory_DB.A_FIX1_PART_1ST;
Inputs.i_PART_CONTROL_B3 := OP_Memory_DB.A_FIX1_PART_1ST;
Inputs.i_PART_CONTROL_B4 := OP_Memory_DB.A_FIX1_PART_1ST;
Inputs.i_PART_CONTROL_B5 := OP_Memory_DB.A_FIX1_PART_1ST;
Inputs.i_PART_CONTROL_B6 := OP_Memory_DB.A_FIX1_PART_1ST;
Inputs.i_PART_CONTROL_B7 := OP_Memory_DB.A_FIX1_PART_1ST;
Inputs.i_PART_CONTROL_B15 := OP_Memory_DB.A_FIX1_PART_2ND;
Inputs.i_PART_CONTROL_B16 := OP_Memory_DB.A_FIX1_PART_2ND;
Inputs.i_PART_CONTROL_B17 := OP_Memory_DB.A_FIX1_PART_2ND;
Inputs.i_PART_CONTROL_B18 := OP_Memory_DB.A_FIX1_PART_2ND;
Inputs.i_PART_CONTROL_B19 := OP_Memory_DB.A_FIX1_PART_2ND;
Inputs.i_PART_CONTROL_B20 := OP_Memory_DB.A_FIX1_PART_2ND;
Inputs.i_PART_CONTROL_B21 := OP_Memory_DB.A_FIX1_PART_2ND;
Inputs.i_PART_CONTROL_B8 := OP_Memory_DB.A_FIX1_PART_3RD;
Inputs.i_PART_CONTROL_B9 := OP_Memory_DB.A_FIX1_PART_3RD;
Inputs.i_PART_CONTROL_B10 := OP_Memory_DB.A_FIX1_PART_3RD;
Inputs.i_PART_CONTROL_B11 := OP_Memory_DB.A_FIX1_PART_3RD;
Inputs.i_PART_CONTROL_B12 := OP_Memory_DB.A_FIX1_PART_3RD;
Inputs.i_PART_CONTROL_B13 := OP_Memory_DB.A_FIX1_PART_3RD;
Inputs.i_PART_CONTROL_B14 := OP_Memory_DB.A_FIX1_PART_3RD;
Inputs.i_PART_CONTROL_B28 := OP_Memory_DB.A_FIX1_PART_4TH;
Inputs.i_PART_CONTROL_B22 := OP_Memory_DB.A_FIX1_PART_4TH;
Inputs.i_PART_CONTROL_B23 := OP_Memory_DB.A_FIX1_PART_4TH;
Inputs.i_PART_CONTROL_B24 := OP_Memory_DB.A_FIX1_PART_4TH;
Inputs.i_PART_CONTROL_B25 := OP_Memory_DB.A_FIX1_PART_4TH;
Inputs.i_PART_CONTROL_B26 := OP_Memory_DB.A_FIX1_PART_4TH;
Inputs.i_PART_CONTROL_B27 := OP_Memory_DB.A_FIX1_PART_4TH;

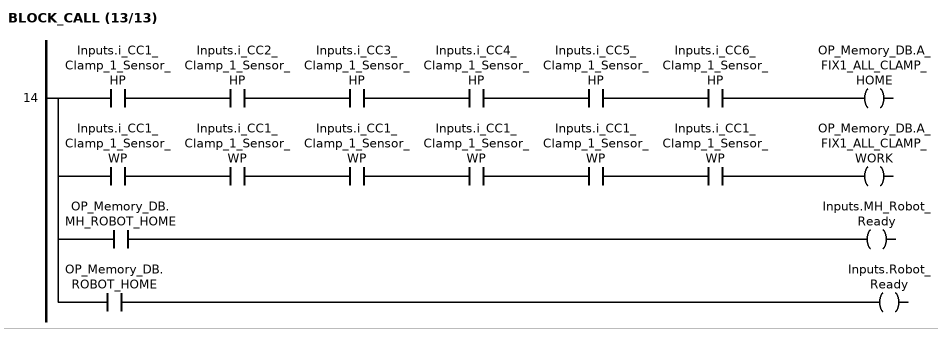
// NETWORK 14
OP_Memory_DB.A_FIX1_ALL_CLAMP_HOME := ((((Inputs.i_CC1_Clamp_1_Sensor_HP AND Inputs.i_CC2_Clamp_1_Sensor_HP) AND Inputs.i_CC3_Clamp_1_Sensor_HP) AND Inputs.i_CC4_Clamp_1_Sensor_HP) AND Inputs.i_CC5_Clamp_1_Sensor_HP) AND Inputs.i_CC6_Clamp_1_Sensor_HP;
OP_Memory_DB.A_FIX1_ALL_CLAMP_WORK := ((((Inputs.i_CC1_Clamp_1_Sensor_WP AND Inputs.i_CC1_Clamp_1_Sensor_WP) AND Inputs.i_CC1_Clamp_1_Sensor_WP) AND Inputs.i_CC1_Clamp_1_Sensor_WP) AND Inputs.i_CC1_Clamp_1_Sensor_WP) AND Inputs.i_CC1_Clamp_1_Sensor_WP;
Inputs.MH_Robot_Ready := OP_Memory_DB.MH_ROBOT_HOME;
Inputs.Robot_Ready := OP_Memory_DB.ROBOT_HOME;

END_PROGRAM

// ---- POUs/CLAMP_PROCESS.TcPOU
FUNCTION_BLOCK CLAMP_PROCESS
VAR_INPUT
    Home_Sensor       : BOOL;
    Work_Sensor       : BOOL;
    Auto_Mode         : BOOL;
    Manual_Mode       : BOOL;

    Auto_Clamp_CMD    : BOOL;
    Auto_Unclamp_CMD  : BOOL;

    Man_Extend_CMD    : BOOL;
    Man_Retract_CMD   : BOOL;

    Reset_Fault       : BOOL;

END_VAR
VAR_OUTPUT
	ENABLE : BOOL;
	 Extend_Valve      : BOOL;
    Retract_Valve     : BOOL;

END_VAR
VAR
  State             : INT := 0;
  // Timers
    T_Extend          : TON;
    T_Retract         : TON;

    // Alarms
    Alarm_Extend_Timeout : BOOL;
    Alarm_Retract_Timeout: BOOL;
    Alarm_Sensor_Error   : BOOL;

END_VAR

// ----------------------------
// Mode Selection
// ----------------------------
IF Auto_Mode THEN

    CASE State OF

        // HOME
        0:
            IF Auto_Clamp_CMD THEN
                State := 1;
            END_IF;

        // MOVING TO WORK
        1:
            Extend_Valve := TRUE;

            T_Extend(IN := TRUE, PT := T#2S);

            IF Work_Sensor THEN
                Extend_Valve := FALSE;
                T_Extend(IN := FALSE);
                State := 2;
            ELSIF T_Extend.Q THEN
                Alarm_Extend_Timeout := TRUE;
                State := 99;
            END_IF;
			 // WORK
        2:
            IF Auto_Unclamp_CMD THEN
                State := 3;
            END_IF;

        // MOVING TO HOME
        3:
            Retract_Valve := TRUE;

            T_Retract(IN := TRUE, PT := T#2S);

            IF Home_Sensor THEN
                Retract_Valve := FALSE;
                T_Retract(IN := FALSE);
                State := 0;
            ELSIF T_Retract.Q THEN
                Alarm_Retract_Timeout := TRUE;
                State := 99;
            END_IF;

        // FAULT
        99:
            Extend_Valve  := FALSE;
            Retract_Valve := FALSE;

            IF Reset_Fault THEN
                Alarm_Extend_Timeout  := FALSE;
                Alarm_Retract_Timeout := FALSE;
                Alarm_Sensor_Error    := FALSE;
                State := 0;
            END_IF;
 END_CASE;

END_IF;
// ----------------------------
// Manual Mode
// ----------------------------
IF Manual_Mode AND NOT Auto_Mode THEN
    State := 0;
    // No state machine, direct control with interlock
    IF Man_Extend_CMD AND NOT Work_Sensor THEN
        Extend_Valve := TRUE;
    ELSE
        Extend_Valve := FALSE;
    END_IF;

    IF Man_Retract_CMD AND NOT Home_Sensor THEN
        Retract_Valve := TRUE;
    ELSE
        Retract_Valve := FALSE;
    END_IF;

END_IF;


// ----------------------------
// Final Safety Interlock
// ----------------------------
IF Extend_Valve AND Retract_Valve THEN
    Extend_Valve  := FALSE;
    Retract_Valve := FALSE;
END_IF;

END_FUNCTION_BLOCK

// ---- POUs/FEEDBACK_FB.TcPOU
FUNCTION_BLOCK FEEDBACK_FB
VAR_INPUT
	EN : BOOL;
	Command_1  : BOOL;
	Command_2  : BOOL;
	Command_3  : BOOL;
	Command_4  : BOOL;
END_VAR
VAR_OUTPUT
	ENO           : BOOL;
	Feedback_1    : BOOL;     
    Feedback_2    : BOOL;
	Feedback_3    : BOOL;     
    Feedback_4    : BOOL;     
	
END_VAR
VAR
	   fb1_Time       : TON;
	   fb2_Time       : TON;
	   fb3_Time       : TON;
	   fb4_Time       : TON;
	   fbDelay1 : TIME := T#1S;
	   fbDelay2 : TIME := T#1S;
	   fbDelay3 : TIME := T#1S;
	   fbDelay4 : TIME := T#1S;
END_VAR


////////////////FEEDBACK 1 DELAY//////////////

IF Command_1 THEN
	fb1_Time(IN := Command_1, PT :=fbDelay1);
	Feedback_1 := fb1_Time.Q;
ELSE 
	Feedback_1 :=FALSE;
	fb1_Time(IN := FALSE);
END_IF;
	
////////////////FEEDBACK 2 DELAY//////////////

IF Command_2 THEN
	fb2_Time(IN := Command_2, PT := fbDelay2);
	Feedback_2 := fb2_Time.Q;
ELSE 
	Feedback_2 :=FALSE;	
	fb2_Time(IN := FALSE);
END_IF;
	
////////////////FEEDBACK 3 DELAY//////////////

IF Command_3 THEN
	fB3_Time(IN := Command_3, PT := fbDelay3);
	Feedback_3 := fb3_Time.Q;
ELSE 
	Feedback_3 :=FALSE;	
	fb3_Time(IN := FALSE);
END_IF;
	
////////////////FEEDBACK 4 DELAY//////////////

IF Command_4 THEN
	fb4_Time(IN := Command_4, PT := fbDelay4);
	Feedback_4 := fb4_Time.Q;
ELSE 
	Feedback_4 :=FALSE;	
	fb4_Time(IN := FALSE);
END_IF;

END_FUNCTION_BLOCK

// ---- POUs/TURNTABLE_2POS.TcPOU
FUNCTION_BLOCK TURNTABLE_2POS
VAR_INPUT
	Drive_Ready : BOOL;
    Pos_0_Sensor    : BOOL;
    Pos_180_Sensor    : BOOL;

    Auto_Mode      : BOOL;
    Manual_Mode    : BOOL;

    Index_To_0     : BOOL;
    Index_To_180     : BOOL;

    Man_To_0       : BOOL;
    Man_To_180       : BOOL;

    Reset_Fault    : BOOL;
END_VAR
VAR_OUTPUT
	ENABLE : BOOL;
    Motor_CW       : BOOL;
    Motor_CCW      : BOOL;
END_VAR
VAR
	  State          : INT := 0;
	  T_Move         : TON;
	  Alarm_Move_Timeout : BOOL;
      Alarm_Sensor_Error : BOOL;
END_VAR

// Sensor Validation
// ----------------------------
IF Pos_0_Sensor AND Pos_180_Sensor THEN
    Alarm_Sensor_Error := TRUE;
    State := 99;
END_IF;


// ----------------------------
// AUTO MODE
// ----------------------------
IF Auto_Mode THEN

    CASE State OF

        // At Position 0*
        0:
            IF Index_To_180 THEN
                State := 1;
            END_IF;
			 // Moving to 180*
        1:
            Motor_CW := TRUE;
            T_Move(IN := TRUE, PT := T#8S);

            IF Pos_180_Sensor THEN
                Motor_CW := FALSE;
                T_Move(IN := FALSE);
                State := 2;
            ELSIF T_Move.Q THEN
                Alarm_Move_Timeout := TRUE;
                State := 99;
            END_IF;

        // At Position B
        2:
            IF Index_To_0 THEN
                State := 3;
            END_IF;
 // Moving to A
        3:
            Motor_CCW := TRUE;
            T_Move(IN := TRUE, PT := T#6S);

            IF Pos_0_Sensor THEN
                Motor_CCW := FALSE;
                T_Move(IN := FALSE);
                State := 0;
            ELSIF T_Move.Q THEN
                Alarm_Move_Timeout := TRUE;
                State := 99;
            END_IF;

        // Fault
        99:
            Motor_CW  := FALSE;
            Motor_CCW := FALSE;

            IF Reset_Fault THEN
                Alarm_Move_Timeout := FALSE;
                Alarm_Sensor_Error := FALSE;
                State := 0;
            END_IF;
			 END_CASE;

END_IF;


// ----------------------------
// MANUAL MODE
// ----------------------------
IF Manual_Mode AND NOT Auto_Mode THEN
      State := 0;
    IF Man_To_180 AND NOT Pos_180_Sensor THEN
        Motor_CW := TRUE;
    ELSE
        Motor_CW := FALSE;
    END_IF;

    IF Man_To_0 AND NOT Pos_0_Sensor THEN
        Motor_CCW := TRUE;
    ELSE
        Motor_CCW := FALSE;
    END_IF;

END_IF;
// ----------------------------
// FINAL SAFETY INTERLOCK
// ----------------------------
IF Motor_CW AND Motor_CCW THEN
    Motor_CW  := FALSE;
    Motor_CCW := FALSE;
END_IF;

END_FUNCTION_BLOCK

// ---- POUs/TRUNION_FB.TcPOU
FUNCTION_BLOCK TRUNION_FB
VAR_INPUT
	Drive_Ready : BOOL;
    Home_LS         : BOOL;
    Work_LS         : BOOL;

    Auto_Mode       : BOOL;
    Manual_Mode     : BOOL;

    Auto_Fwd_CMD    : BOOL;
    Auto_Rev_CMD    : BOOL;

    Man_Fwd_PB      : BOOL;
    Man_Rev_PB      : BOOL;

    Clamp_OK        : BOOL;

    Reset_Fault     : BOOL;

END_VAR
VAR_OUTPUT
	ENABLE : BOOL;
	Motor_Fwd       : BOOL;
    Motor_Rev       : BOOL;
END_VAR
VAR
	State           : INT := 0;
	// Timer
    T_Move          : TON;
    // Status
    Busy            : BOOL;
    At_Home         : BOOL;
    At_Work         : BOOL;
    Fault           : BOOL;
    // Alarms
    Alarm_MoveTimeout : BOOL;
    Alarm_SensorFault : BOOL;
    Alarm_ClampMissing: BOOL;
END_VAR

// SENSOR VALIDATION
// --------------------------------------
(*IF NOT Drive_Ready AND Home_LS AND Work_LS THEN
    Alarm_SensorFault := TRUE;
    Fault := TRUE;
    State := 99;
END_IF;*)


// --------------------------------------
// AUTO MODE
// --------------------------------------
IF Auto_Mode THEN

    CASE State OF

        // ----------------------------------
        // HOME POSITION
        // ----------------------------------
        0:
            At_Home := TRUE;
            At_Work := FALSE;
            Busy := FALSE;

            IF Auto_Fwd_CMD THEN
				   // Clamp check before motion
                IF Clamp_OK THEN
                    State := 1;
                ELSE
                    Alarm_ClampMissing := TRUE;
                    Fault := TRUE;
                    State := 99;
                END_IF;

            END_IF;


        // ----------------------------------
        // MOVING FORWARD
        // ----------------------------------
		1:
            Busy := TRUE;

            Motor_Fwd := TRUE;
            Motor_Rev := FALSE;

            T_Move(IN := TRUE, PT := T#8S);

            IF Work_LS THEN

                Motor_Fwd := FALSE;
                T_Move(IN := FALSE);

                At_Home := FALSE;
                At_Work := TRUE;
                Busy := FALSE;

                State := 2;

            ELSIF T_Move.Q THEN

                Alarm_MoveTimeout := TRUE;
                Fault := TRUE;
                State := 99;
			END_IF;
			 // ----------------------------------
        // WORK POSITION
        // ----------------------------------
        2:
            IF Auto_Rev_CMD THEN
                State := 3;
            END_IF;


        // ----------------------------------
        // MOVING HOME
        // ----------------------------------
        3:
            Busy := TRUE;

            Motor_Fwd := FALSE;
            Motor_Rev := TRUE;

            T_Move(IN := TRUE, PT := T#8S);
			 IF Home_LS THEN

                Motor_Rev := FALSE;
                T_Move(IN := FALSE);

                At_Home := TRUE;
                At_Work := FALSE;
                Busy := FALSE;

                State := 0;

            ELSIF T_Move.Q THEN

                Alarm_MoveTimeout := TRUE;
                Fault := TRUE;
                State := 99;

            END_IF;

  // ----------------------------------
        // FAULT STATE
        // ----------------------------------
        99:
            Motor_Fwd := FALSE;
            Motor_Rev := FALSE;
            Busy := FALSE;

            IF Reset_Fault THEN

                Alarm_MoveTimeout := FALSE;
                Alarm_SensorFault := FALSE;
                Alarm_ClampMissing := FALSE;

                Fault := FALSE;

                State := 0;

            END_IF;

    END_CASE;

END_IF;
// --------------------------------------
// MANUAL MODE
// --------------------------------------
IF Manual_Mode AND NOT Auto_Mode THEN
     State := 0;
    // Forward Jog
    IF Man_Fwd_PB AND NOT Work_LS THEN

        IF Clamp_OK THEN
			
            Motor_Fwd := TRUE;
        ELSE
            Alarm_ClampMissing := TRUE;
        END_IF;

    ELSE
        Motor_Fwd := FALSE;
    END_IF;


    // Reverse Jog
    IF Man_Rev_PB AND NOT Home_LS THEN
        Motor_Rev := TRUE;
    ELSE
        Motor_Rev := FALSE;
    END_IF;

END_IF;
// --------------------------------------
// SAFETY INTERLOCK
// --------------------------------------
IF Motor_Fwd AND Motor_Rev THEN
    Motor_Fwd := FALSE;
    Motor_Rev := FALSE;
END_IF;

END_FUNCTION_BLOCK

// ---- POUs/BIW/ROLLER_DOOR.TcPOU
FUNCTION_BLOCK ROLLER_DOOR
VAR_INPUT
	Door_Open_LS      : BOOL;
    Door_Close_LS     : BOOL;

    Open_CMD          : BOOL;
    Close_CMD         : BOOL;

    Auto_Mode         : BOOL;
    Manual_Mode       : BOOL;

    Man_Open_PB       : BOOL;
    Man_Close_PB      : BOOL;

    Safety_Beam       : BOOL;
    Reset_Fault       : BOOL;
END_VAR
VAR_OUTPUT
	ENO : BOOL;
	Motor_Open        : BOOL;
    Motor_Close       : BOOL;

END_VAR
VAR
	 State             : INT := 0;
    // Timers
    T_Open            : TON;
    T_Close           : TON;
	 // Status
    Door_Open_OK      : BOOL;
    Door_Close_OK     : BOOL;
    Busy              : BOOL;
    Fault             : BOOL;

    // Alarms
    Alarm_OpenTimeout : BOOL;
    Alarm_CloseTimeout: BOOL;
    Alarm_SensorFault : BOOL;
    Alarm_Obstacle    : BOOL;

END_VAR

// SENSOR VALIDATION
// ------------------------------------
IF Door_Open_LS AND Door_Close_LS THEN
    Alarm_SensorFault := TRUE;
    Fault := TRUE;
    State := 99;
END_IF;
// ------------------------------------
// AUTO MODE
// ------------------------------------
IF Auto_Mode AND NOT Manual_Mode THEN
    IF Open_CMD AND NOT Door_Open_LS THEN
        Motor_Open := TRUE;
    ELSE
        Motor_Open := FALSE;
    END_IF;
	
    IF Close_CMD AND NOT Door_Close_LS AND NOT Safety_Beam THEN
        Motor_Close := TRUE;
    ELSE
        Motor_Close := FALSE;
    END_IF;
	END_IF;


// ------------------------------------
// MANUAL MODE
// ------------------------------------
IF Manual_Mode AND NOT Auto_Mode THEN

    // Manual OPEN
    IF Man_Open_PB AND NOT Door_Open_LS THEN
        Motor_Open := TRUE;
    ELSE
        Motor_Open := FALSE;
    END_IF;


    // Manual CLOSE
    IF Man_Close_PB AND NOT Door_Close_LS AND NOT Safety_Beam THEN
        Motor_Close := TRUE;
    ELSE
        Motor_Close := FALSE;
    END_IF;
	END_IF;


// ------------------------------------
// FINAL SAFETY INTERLOCK
// ------------------------------------
IF Motor_Open AND Motor_Close THEN
    Motor_Open := FALSE;
    Motor_Close := FALSE;
	END_IF;

END_FUNCTION_BLOCK

// ---- POUs/RollerDoor.TcPOU
FUNCTION_BLOCK PUBLIC RollerDoor
VAR_INPUT
	
    bOpenButton     : BOOL;     // Pushbutton / Pull-cord
    bCloseButton    : BOOL;     // Pushbutton
    bSafetyEdge     : BOOL;     // Bottom edge sensor (Normally Closed for safety)
    bPhotoeye       : BOOL;     // Obstruction sensor (Normally Closed)
    bLimitUp        : BOOL;     // Door fully open sensor
    bLimitDown      : BOOL;     // Door fully closed sensor


END_VAR
VAR_OUTPUT
	ENO             : BOOL;
    bMotorUp        : BOOL;     // Up Contactor
    bMotorDown      : BOOL;     // Down Contactor

END_VAR
VAR
	
    nState          : INT;      // 0: Stopped, 10: Opening, 20: Closing, 99: Error
    fbAutoCloseTimer: TON;      // Automatically close after opening

END_VAR

// Auto-Close Timer: Starts when door is fully open
//fbAutoCloseTimer(IN := bLimitUp, PT := T#10S);

CASE nState OF
    0: // STOPPED
        bMotorUp   := FALSE;
        bMotorDown := FALSE;
        
        IF bOpenButton AND NOT bLimitUp THEN
            nState := 10;
        ELSIF bCloseButton  AND NOT bLimitDown THEN
            // Only allow closing if safety is clear
            IF bSafetyEdge AND bPhotoeye THEN
                nState := 20;
            END_IF
        END_IF

    10: // OPENING
        bMotorUp   := TRUE;
        bMotorDown := FALSE;
        
        IF bLimitUp OR bCloseButton THEN
            nState := 0; // Stop if reached limit or close pressed
        END_IF

    20: // CLOSING
        bMotorUp   := FALSE;
        bMotorDown := TRUE;
        
        // Safety Reversal: If something is hit or detected, open immediately
        IF NOT bSafetyEdge OR NOT bPhotoeye THEN
            nState := 10; 
        ELSIF bLimitDown OR bOpenButton THEN
            nState := 0;
        END_IF

    99: // ERROR / EMERGENCY STOP
        bMotorUp   := FALSE;
        bMotorDown := FALSE;
END_CASE

END_FUNCTION_BLOCK

// ---- POUs/WELD_ROBOT.TcPOU
FUNCTION_BLOCK WELD_ROBOT
VAR_INPUT
	StartPB : BOOL;
	RobotReady : BOOL;
	
	
	RobotFault : BOOL;
	SafetyOK : BOOL;
	WeldProgram : INT;
	ResetPB : BOOL;
	
END_VAR
VAR_OUTPUT
	Eno : BOOL;
	RobotStart : BOOL;
	RobotReset : BOOL;
	RobotBusy : BOOL;
	RobotComplete : BOOL;
	RobotHOME : BOOL;
	ProgBit0 : BOOL;
	ProgBit1 : BOOL;
	ProgBit2 : BOOL;
	ProgBit3 : BOOL;
	
END_VAR
VAR
	ProgNum: INT;
	T_Weld_Time : TON;
	
	AutoRequest : BOOL;
    StartEdge   : R_TRIG;
    CycleRun    : BOOL;
    FaultLamp  : BOOL;
	CycleComplete : BOOL;
	Step : INT;
END_VAR

(*0 = Idle
10 = Send Program Number
20 = Start Robot
30 = Wait Busy
40 = Wait Complete
50 = Cycle Finish
900 = Fault*)
IF NOT SafetyOK THEN Step := 0;
	
END_IF
CASE Step OF

0:   RobotHOME := TRUE;
     //RobotStart := FALSE;
     RobotBusy := FALSE;
	 T_Weld_Time(IN :=FALSE);
	 
	 RobotComplete := FALSE;
    IF StartPB AND SafetyOK THEN
       Step := 10;
    END_IF;

10:
    WeldProgram := 5;
	RobotBusy := TRUE;
	RobotHOME := FALSE;
    Step := 20;

20:
    //RobotStart := TRUE;
	//RobotBusy := FALSE;
	//RobotComplete := TRUE;
	T_Weld_Time(IN := TRUE, PT :=T#5S);
   
    IF T_Weld_Time.Q THEN
       RobotComplete := TRUE; RobotStart := FALSE; RobotBusy := FALSE;
       Step := 30;
    END_IF;

30:
    IF RobotComplete THEN
		//T_Weld_Time.Q :=FALSE;
       Step := 0;
    END_IF;



END_CASE;

END_FUNCTION_BLOCK

// ---- POUs/MH_ROBOT.TcPOU
FUNCTION_BLOCK MH_ROBOT
VAR_INPUT
	StartPB : BOOL;
	RobotReady : BOOL;
	
	
	RobotFault : BOOL;
	SafetyOK : BOOL;
	MHProgram : INT;
	ResetPB : BOOL;
	
END_VAR
VAR_OUTPUT
	Eno : BOOL;
	RobotStart : BOOL;
	RobotReset : BOOL;
	RobotBusy : BOOL;
	RobotComplete : BOOL;
	RobotHOME : BOOL;
	ProgBit0 : BOOL;
	ProgBit1 : BOOL;
	ProgBit2 : BOOL;
	ProgBit3 : BOOL;
	
END_VAR
VAR
	ProgNum: INT;
	T_MH_Time : TON;
	
	AutoRequest : BOOL;
    StartEdge   : R_TRIG;
    CycleRun    : BOOL;
    FaultLamp  : BOOL;
	CycleComplete : BOOL;
	Step : INT;
END_VAR

(*0 = Idle
10 = Send Program Number
20 = Start Robot
30 = Wait Busy
40 = Wait Complete
50 = Cycle Finish
900 = Fault*)
IF NOT SafetyOK THEN Step := 0;
	
END_IF
CASE Step OF

0:   RobotHOME := TRUE;
     //RobotStart := FALSE;
     RobotBusy := FALSE;
	 T_MH_Time(IN :=FALSE);
	 
	 RobotComplete := FALSE;
    IF StartPB AND SafetyOK THEN
       Step := 10;
    END_IF;

10:
    MHProgram := 5;
	RobotBusy := TRUE;
	RobotHOME := FALSE;
    Step := 20;

20:
    //RobotStart := TRUE;
	//RobotBusy := FALSE;
	//RobotComplete := TRUE;
	T_MH_Time(IN := TRUE, PT :=T#7S);
   
    IF T_MH_Time.Q THEN
       RobotComplete := TRUE; RobotStart := FALSE; RobotBusy := FALSE;
       Step := 30;
    END_IF;

30:
    IF RobotComplete THEN
		//T_Weld_Time.Q :=FALSE;
       Step := 0;
    END_IF;



END_CASE;

END_FUNCTION_BLOCK

// ---- POUs/MODE_CONTROL.TcPOU
FUNCTION_BLOCK MODE_CONTROL
VAR_INPUT
	PowerON : BOOL;
	AutoSel : BOOL;
	ManualSel : BOOL;
	StartPB : BOOL;
	StopPB : BOOL;
	ResetPB : BOOL;
	SafetyOK : BOOL;
	CLAMP_CLOSE_1 : BOOL;
	CLAMP_CLOSE_2 : BOOL;
	CLAMP_OPEN_1 : BOOL;
	CLAMP_OPEN_2 : BOOL;
	Sensor_1ST_FB : BOOL;
	Sensor_2ND_FB : BOOL;
	Sensor_3RD_FB : BOOL;
	Sensor_4TH_FB : BOOL;
	Palm_Button : BOOL;
	Turntable_0 : BOOL;
	Turntable_180 : BOOL;
	Trunion_0 : BOOL;
	Trunion_20 : BOOL;
	RD_Open : BOOL;
	RD_Close : BOOL;
	
	JogRobotPB : BOOL;
	ClampClosePB : BOOL;
	ALL_CLAMP_HOME : BOOL;
	ClampClosedSensor : BOOL;
	WELD_RobotBusy : BOOL;
	WELD_Robotcomplete : BOOL;
	WELD_RobotHome : BOOL;
	WELD_RobotReady : BOOL;
	MH_RobotBusy : BOOL;
	MH_Robotcomplete : BOOL;
	MH_RobotHome : BOOL;
	MH_RobotReady : BOOL;
END_VAR
VAR_OUTPUT
	ENO : BOOL;
	AutoMode :BOOL;
	ManualMode : BOOL;
	WELD_RobotStart : BOOL;
	MH_RobotStart : BOOL;
	RobotJog : BOOL;
	ClampClose_1 : BOOL;
	ClampClose_2 : BOOL;
	ClampClose_3 : BOOL;
	ClampClose_4 : BOOL;
	ClampClose_5 : BOOL;
	ClampClose_6 : BOOL;
	ClampOpen_1 : BOOL;
	ClampOpen_2 : BOOL;
	ClampOpen_3 : BOOL;
	ClampOpen_4 : BOOL;
	ClampOpen_5 : BOOL;
	ClampOpen_6 : BOOL;
	Sensor_1ST : BOOL;
	Sensor_2ND : BOOL;
	Sensor_3RD : BOOL;
	Sensor_4TH : BOOL;
	Turntable_0_CMD : BOOL;
	Turntable_180_CMD : BOOL;
	Trunion_0_CMD : BOOL;
	Trunion_20_CMD : BOOL;
	RD_CLOSE_CMD : BOOL;
	RD_OPEN_CMD : BOOL;
	FaultLamp : BOOL;
	
END_VAR
VAR
	AutoMode_Sel_db       : BOOL;
    ManualMode_Sel_db     : BOOL;

    CycleRun       : BOOL;
    FaultLatch     : BOOL;

    Step           : INT := 0;

    StartEdge      : R_TRIG;
END_VAR


// ---------------------------------------
// Mode Selection
// ---------------------------------------

IF PowerON AND AutoSel AND SafetyOK THEN
    AutoMode := TRUE;
    ManualMode := FALSE;
END_IF;

IF PowerON AND NOT AutoSel THEN
    ManualMode := TRUE;
    AutoMode := FALSE;
	
	Step := 0;
END_IF;


// ---------------------------------------
// Fault Handling
// ---------------------------------------

IF NOT SafetyOK THEN
    FaultLatch := TRUE;
END_IF;

IF ResetPB THEN
    FaultLatch := FALSE;
END_IF;

FaultLamp := FaultLatch;
// ---------------------------------------
// MANUAL MODE
// ---------------------------------------

IF ManualMode AND NOT FaultLatch THEN

    // Manual Robot Jog
    RobotJog := JogRobotPB;
    RD_CLOSE_CMD :=FALSE;
	RD_OPEN_CMD :=FALSE;
    // Manual Clamp Control
    //ClampClose := ClampClosePB;

END_IF;


// ---------------------------------------
// AUTO MODE
// ---------------------------------------

IF AutoMode THEN //AND ALL_CLAMP_HOME AND Turntable_0 AND Trunion_0 AND RD_Open AND NOT FaultLatch THEN

    StartEdge(CLK := StartPB);

    CASE Step OF
    // -----------------------------------
    // CYCLE START
    // -----------------------------------

    0:
        WELD_RobotStart := FALSE;
		MH_RobotStart := FALSE;
		//RD_OPEN_CMD :=FALSE;
		//RD_CLOSE_CMD :=FALSE;
		
        CycleRun := FALSE;

        IF  StartEdge.Q AND WELD_RobotReady THEN
            Step := 10;
            
        END_IF;
    // -----------------------------------
    // RD_CLOSE-0
    // -----------------------------------

    10:
        RD_CLOSE_CMD := TRUE;

        IF RD_Close THEN
			RD_CLOSE_CMD := FALSE;
            Step := 20;
        END_IF;
	// -----------------------------------
    // TRUNION-20
    // -----------------------------------

    20:
        Trunion_20_CMD := TRUE;

        IF Trunion_20 THEN
			Trunion_20_CMD:=FALSE;
            Step := 30;
        END_IF;
    // -----------------------------------
    // RD_OPEN-0
    // -----------------------------------

    30:
        RD_OPEN_CMD := TRUE;

        IF RD_Open THEN
            Step := 40;
			 RD_OPEN_CMD := FALSE;
        END_IF;
	// -----------------------------------
    // Operator Load_1ST PART
    // -----------------------------------

    40:
        

        Sensor_1ST := TRUE ;
        //Sensor_2ND := TRUE;
        //Sensor_3RD := TRUE;
        //Sensor_4TH := TRUE; 
	   IF  Sensor_1ST_FB AND Palm_Button THEN
            Step := 50;
        END_IF;
	// -----------------------------------
    // Operator Load_2ND PART
    // -----------------------------------
     50:
        // Sensor_1ST := TRUE ;
        Sensor_2ND := TRUE;
        //Sensor_3RD := TRUE;
        //Sensor_4TH := TRUE; 
	   IF Sensor_2ND_FB AND Palm_Button THEN
            Step := 60;
        END_IF;
		
    // -----------------------------------
    // Clamp Close_1ST,3RD,5TH
    // -----------------------------------

    60:
        ClampClose_1 := TRUE;
		ClampClose_3 := TRUE;
		ClampClose_5 := TRUE;
        IF ClampClosedSensor THEN
            Step := 70;
        END_IF;
   // -----------------------------------
    // RD_CLOSE-0
    // -----------------------------------

    70:
        RD_CLOSE_CMD := TRUE;
        ClampClose_1 := FALSE;
		ClampClose_3 := FALSE;
		ClampClose_5 := FALSE;
        IF CLAMP_CLOSE_1 AND RD_Close THEN
            Step := 80;
        END_IF;
	// -----------------------------------
    // TRUNION-80
    // -----------------------------------

    80:
        Trunion_20_CMD := TRUE;
        RD_CLOSE_CMD := FALSE;
        IF Trunion_20 THEN
			 Trunion_20_CMD := FALSE;
            Step := 90;
        END_IF;
    // -----------------------------------
    // RD_OPEN-0
    // -----------------------------------

    90:
        RD_OPEN_CMD := TRUE;
       
        IF RD_Open THEN
			 RD_OPEN_CMD := FALSE;
            Step := 100;
        END_IF;
	// -----------------------------------
    // Operator Load_3RD_PART
    // -----------------------------------

    100:
       Sensor_3RD := TRUE ;
        //Sensor_2ND := TRUE;
        //Sensor_3RD := TRUE;
        //Sensor_4TH := TRUE; 
	   IF Sensor_3RD_FB AND Palm_Button THEN
            Step := 110;
        END_IF;
   // -----------------------------------
    // Operator Load_4TH_PART
    // -----------------------------------

    110:
       // Sensor_1ST := TRUE ;
        Sensor_4TH := TRUE;
        //Sensor_3RD := TRUE;
        //Sensor_4TH := TRUE; 
	   IF Sensor_4TH_FB AND Palm_Button THEN
            Step := 120;
        END_IF;
	//------------------------------
	// RD_CLOSE-0
    // -----------------------------------

    120:
        RD_CLOSE_CMD := TRUE;
        IF RD_Close THEN
			RD_CLOSE_CMD := FALSE;
            Step := 130;
        END_IF;
	// -----------------------------------
    //  CLAMP CLOSE 2ND,4TH, 6TH
    // -----------------------------------

    130: ClampClose_2 := TRUE;
		 ClampClose_4 := TRUE;
		 ClampClose_6 := TRUE;
         
        
        IF CLAMP_CLOSE_2 THEN
			
            Step := 140;
        END_IF;
	// -----------------------------------
    // TURNTABLE-180* AND TRUNION_0*
    // -----------------------------------

    140: ClampClose_2 := FALSE;
		 ClampClose_4 := FALSE;
		 ClampClose_6 := FALSE;
         Turntable_180_CMD := TRUE;
         Trunion_0_CMD := TRUE;
        IF Turntable_180 AND  Trunion_0 THEN
			Turntable_180_CMD := FALSE;
			Trunion_0_CMD := FALSE;
            Step := 150;
        END_IF;
   
	

    // -----------------------------------
    // Start WELD_Robot
    // -----------------------------------

    150:
        WELD_RobotStart := TRUE;

        IF WELD_Robotcomplete THEN
            WELD_RobotStart := FALSE;
            Step := 160;
        END_IF;


    // -----------------------------------
    // CLAMP OPEN 1ST,3RD,5TH
    // -----------------------------------

    160:
        CycleRun := TRUE;
		ClampOpen_1 := TRUE;
		ClampOpen_3 := TRUE;
		ClampOpen_5 := TRUE;
        IF  CLAMP_OPEN_1 THEN
	    ClampOpen_1 := FALSE;
		ClampOpen_3 := FALSE;
		ClampOpen_5 := FALSE;
            Step := 170;
        END_IF;
    // -----------------------------------
    // RD_OPEN
    // -----------------------------------
		
	170: 
        RD_OPEN_CMD := TRUE;
        
        IF RD_Open THEN
			RD_OPEN_CMD := FALSE;
            Step := 180;
        END_IF;
		
	

    // -----------------------------------
    // Start MH_Robot_1ST
    // -----------------------------------

    180:
        MH_RobotStart := TRUE;
		Sensor_1ST := FALSE;
        Sensor_2ND := FALSE;
        IF MH_Robotcomplete AND NOT Sensor_1ST_FB AND NOT Sensor_2ND_FB  THEN
            MH_RobotStart := FALSE;
            Step := 190;
        END_IF;
	// -----------------------------------
    // TRUNION_45
    // -----------------------------------	
	 190:
        Trunion_20_CMD := TRUE;
        RD_CLOSE_CMD := FALSE;
        IF Trunion_20 THEN
			 Trunion_20_CMD := FALSE;
            Step := 200;
        END_IF;
    
	// -----------------------------------
    // Start UNCLAMP 2ND, 4TH,6TH
    // -----------------------------------
		
    200:
        CycleRun := TRUE;
		ClampOpen_2 := TRUE;
		ClampOpen_4 := TRUE;
		ClampOpen_6 := TRUE;
        IF CLAMP_OPEN_2 THEN
	    ClampOpen_2 := FALSE;
		ClampOpen_4 := FALSE;
		ClampOpen_6 := FALSE;
            Step := 210;
        END_IF;
	// -----------------------------------
    // Start MH_Robot_2ND
    // -----------------------------------
		
     210:
        MH_RobotStart := TRUE;
		Sensor_3RD := FALSE;
		Sensor_4TH := FALSE;
        IF MH_RobotBusy AND NOT Sensor_3RD_FB AND NOT Sensor_4TH_FB THEN
            MH_RobotStart := FALSE;
            Step := 220;
        END_IF;
// -----------------------------------
    // Cycle Finish
    // -----------------------------------

    220:
        CycleRun := FALSE;
        
        Step := 0;

    END_CASE;

END_IF;

END_FUNCTION_BLOCK

// ---- POUs/SENSOR.TcPOU
FUNCTION_BLOCK SENSOR
VAR_INPUT
	SENSOR_1 : BOOL;
	SENSOR_2 : BOOL;
	SENSOR_3 : BOOL;
	SENSOR_4 : BOOL;
	SENSOR_5 : BOOL;
	SENSOR_6 : BOOL;
	SENSOR_7 : BOOL;
	SENSOR_8 : BOOL;
	SENSOR_9 : BOOL;
	SENSOR_10 : BOOL;
	SENSOR_11 : BOOL;
	SENSOR_12 : BOOL;
	SENSOR_13 : BOOL;
	SENSOR_14 : BOOL;
	SENSOR_15 : BOOL;
	SENSOR_16 : BOOL;
	SENSOR_17 : BOOL;
	SENSOR_18 : BOOL;
	SENSOR_19 : BOOL;
	SENSOR_20 : BOOL;
	SENSOR_21 : BOOL;
	SENSOR_22 : BOOL;
	SENSOR_23 : BOOL;
	SENSOR_24 : BOOL;
	SENSOR_25 : BOOL;
	SENSOR_26 : BOOL;
	SENSOR_27 : BOOL;
	SENSOR_28 : BOOL;
	
	
	
	
	
	
END_VAR
VAR_OUTPUT
	ENO : BOOL;
    SENSOR_SET_1 : BOOL;
	SENSOR_SET_2 : BOOL;
	SENSOR_SET_3 : BOOL;
	SENSOR_SET_4 : BOOL;
	SENSOR_SET_5 : BOOL;
	SENSOR_SET_6 : BOOL;
	
	
END_VAR
VAR
END_VAR

IF    (SENSOR_1 AND SENSOR_2 AND SENSOR_3 AND SENSOR_4 AND SENSOR_5 AND SENSOR_6 AND SENSOR_7)
OR	  (SENSOR_2 AND SENSOR_3 AND SENSOR_4 AND SENSOR_5 AND SENSOR_6 AND SENSOR_7)
THEN  SENSOR_SET_1 := TRUE; 

ELSIF (SENSOR_15 AND SENSOR_16 AND SENSOR_17 AND SENSOR_18 AND SENSOR_19 AND SENSOR_20 AND SENSOR_21)
OR    (SENSOR_16 AND SENSOR_17 AND SENSOR_18 AND SENSOR_19 AND SENSOR_20 AND SENSOR_21)	   
THEN  SENSOR_SET_2 := TRUE;	
 
ELSIF (SENSOR_8 AND SENSOR_9 AND SENSOR_10 AND SENSOR_11 AND SENSOR_12 AND SENSOR_13 AND SENSOR_14)
OR    (SENSOR_8 AND SENSOR_9 AND SENSOR_10 AND SENSOR_11 AND SENSOR_12 AND SENSOR_13 )
THEN  SENSOR_SET_3 := TRUE;

ELSIF (SENSOR_22 AND SENSOR_23 AND SENSOR_24 AND SENSOR_25 AND SENSOR_26 AND SENSOR_27 AND SENSOR_28)
OR    (SENSOR_22 AND SENSOR_23 AND SENSOR_24 AND SENSOR_25 AND SENSOR_26 AND SENSOR_27 )
THEN  SENSOR_SET_4 := TRUE;

ELSIF NOT SENSOR_1 AND NOT SENSOR_2 AND NOT SENSOR_3 AND NOT SENSOR_4 AND NOT SENSOR_5 AND NOT SENSOR_6 AND NOT SENSOR_7 AND
	 NOT SENSOR_8 AND NOT SENSOR_9 AND NOT SENSOR_10 AND NOT SENSOR_11 AND NOT SENSOR_12 AND NOT SENSOR_13 AND NOT SENSOR_14 AND
	  NOT SENSOR_15 AND NOT SENSOR_16 AND NOT SENSOR_17 AND NOT SENSOR_18 AND NOT SENSOR_19 AND NOT SENSOR_20 AND NOT SENSOR_21 
THEN  SENSOR_SET_5 := TRUE;
	
   
ELSIF NOT SENSOR_8 AND NOT SENSOR_9 AND NOT SENSOR_10 AND NOT SENSOR_11 AND NOT SENSOR_12 AND NOT SENSOR_13 AND NOT SENSOR_14 AND
	  NOT SENSOR_22 AND NOT SENSOR_23 AND NOT SENSOR_24 AND NOT SENSOR_25 AND NOT SENSOR_26 AND NOT SENSOR_27 AND NOT SENSOR_28 
THEN  SENSOR_SET_6 := TRUE;
END_IF

(*IF CLAMP_1_WORK AND CLAMP_2_WORK AND CLAMP_3_WORK AND CLAMP_4_WORK AND CLAMP_5_WORK AND CLAMP_6_WORK
THEN ALL_CLAMP_WORK := TRUE;
END_IF
IF CLAMP_1_HOME AND CLAMP_2_HOME AND CLAMP_3_HOME AND CLAMP_4_HOME AND CLAMP_5_HOME AND CLAMP_6_HOME
THEN ALL_CLAMP_HOME := TRUE;
END_IF   
IF CLAMP_1_WORK 
THEN CLAMP_SET_1 :=TRUE;
END_IF
IF CLAMP_1_HOME 
THEN CLAMP_RESET_1 :=TRUE;
END_IF

IF CLAMP_2_WORK 
THEN  CLAMP_SET_2 :=TRUE;
END_IF

IF CLAMP_2_HOME  
THEN  CLAMP_RESET_2 :=TRUE;
END_IF

IF CLAMP_3_WORK 
THEN  CLAMP_SET_3 :=TRUE;
END_IF

IF CLAMP_3_HOME 
THEN  CLAMP_RESET_3 :=TRUE;
END_IF
IF CLAMP_4_WORK 
THEN  CLAMP_SET_4 :=TRUE;
END_IF
IF CLAMP_4_HOME
THEN  CLAMP_RESET_4 :=TRUE;
END_IF
IF CLAMP_5_WORK 
THEN  CLAMP_SET_5 :=TRUE;
END_IF
IF CLAMP_5_HOME 
THEN  CLAMP_RESET_5 :=TRUE;
END_IF
IF CLAMP_6_WORK 
THEN  CLAMP_SET_6 :=TRUE;
END_IF
IF CLAMP_6_HOME 
THEN  CLAMP_RESET_6 :=TRUE;
END_IF*)

(*IF CLAMP_1_HOME AND CLAMP_2_HOME AND CLAMP_3_HOME AND CLAMP_4_HOME AND CLAMP_5_HOME AND CLAMP_6_HOME
THEN ALL_CLAMP_HOME := TRUE;
   
ELSIF CLAMP_1_HOME AND CLAMP_3_HOME AND CLAMP_5_HOME
THEN CLAMP_RESET_1 :=TRUE;

ELSIF CLAMP_2_HOME AND CLAMP_4_HOME AND CLAMP_6_HOME
THEN  CLAMP_RESET_2 :=TRUE;

ELSIF CLAMP_2_HOME AND CLAMP_4_HOME AND CLAMP_6_HOME
THEN  CLAMP_RESET_2 :=TRUE;

END_IF*)

END_FUNCTION_BLOCK

// ---- POUs/BIW/Trunion.TcPOU
FUNCTION_BLOCK PUBLIC Trunion
VAR_INPUT
	
    bStart          : BOOL;     // Start rotation command
    bHomeSensor     : BOOL;     // Proximity sensor for position  
  
END_VAR

VAR_OUTPUT
	ENO             : BOOL;
    bMotorRun       : BOOL;     // Command to the motor/drive 

END_VAR

VAR	
    nState          : INT := 0; // 0: Idle, 10: Starting, 20: Rotating, 30: Stopping
    fbTimer         : TON;      // Safety timeout timer

END_VAR

CASE nState OF
    0: // IDLE - Wait for Start Command
        bMotorRun := FALSE;
        IF bStart THEN
            nState := 10;
        END_IF
        
    10: // STARTING - Turn on motor and wait for sensor to clear
        bMotorRun := TRUE;
        IF NOT bHomeSensor THEN // Wait for current part to move away
            nState := 20;
        END_IF
        
    20: // ROTATING - Looking for the next slot
        bMotorRun := TRUE;
        IF bHomeSensor THEN // Sensor detects the next 90-degree slot
            nState := 30;
        END_IF
        
    30: // STOPPING - Stop motor and return to Idle
        bMotorRun := FALSE;
        IF NOT bStart THEN // Require button release to reset
            nState := 0;
        END_IF
END_CASE

// Optional: Safety Timeout to prevent motor burnout if sensor fails
fbTimer(IN := (nState = 20), PT := T#5S);
IF fbTimer.Q THEN
    bMotorRun := FALSE;
    nState := 0; // Or transition to an Error State
END_IF

END_FUNCTION_BLOCK

// ---- POUs/BIW/Callblocks.TcPOU
PROGRAM Callblocks
VAR
	
CC1_Clamp_Unit1_3 : clamp;
CC2_Clamp_Unit2_3 : clamp;
CC3_Clamp_Unit3_3 : clamp;
CC4_Clamp_Unit4_3 : clamp;
CC5_Clamp_Unit5_1 : clamp;
CC6_Clamp_Unit6_1 : clamp;

Temp_bool : BOOL;
Feedback_Unit1  : Feedback_FB;
Feedback_Unit2  : Feedback_FB;
Feedback_Unit3  : Feedback_FB;
Feedback_Unit4  : Feedback_FB;
Feedback_Unit5  : Feedback_FB;
Feedback_Unit6  : Feedback_FB;


Door           : RollerDoor;
Trunion        : Trunion;
TT             : Turntable ;
Robot1         : Weldrobot;
Robot2         : MHrobot;

END_VAR

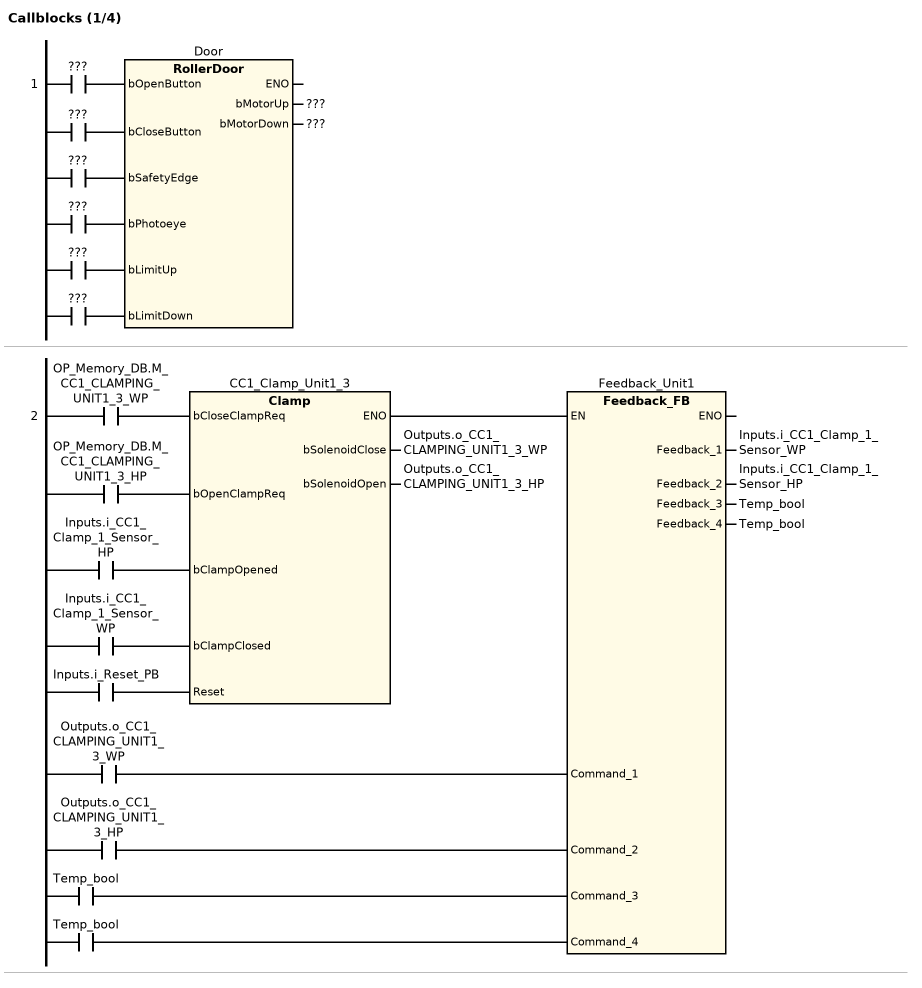
// NETWORK 1
Door(); // RollerDoor

// NETWORK 2
CC1_Clamp_Unit1_3(
    bCloseClampReq := OP_Memory_DB.M_CC1_CLAMPING_UNIT1_3_WP,
    bOpenClampReq := OP_Memory_DB.M_CC1_CLAMPING_UNIT1_3_HP,
    bClampOpened := Inputs.i_CC1_Clamp_1_Sensor_HP,
    bClampClosed := Inputs.i_CC1_Clamp_1_Sensor_WP,
    Reset := Inputs.i_Reset_PB,
    bSolenoidClose => Outputs.o_CC1_CLAMPING_UNIT1_3_WP,
    bSolenoidOpen => Outputs.o_CC1_CLAMPING_UNIT1_3_HP); // Clamp
Feedback_Unit1(
    EN := TRUE,
    Command_1 := Outputs.o_CC1_CLAMPING_UNIT1_3_WP,
    Command_2 := Outputs.o_CC1_CLAMPING_UNIT1_3_HP,
    Command_3 := Temp_bool,
    Command_4 := Temp_bool,
    Feedback_1 => Inputs.i_CC1_Clamp_1_Sensor_WP,
    Feedback_2 => Inputs.i_CC1_Clamp_1_Sensor_HP,
    Feedback_3 => Temp_bool,
    Feedback_4 => Temp_bool); // Feedback_FB

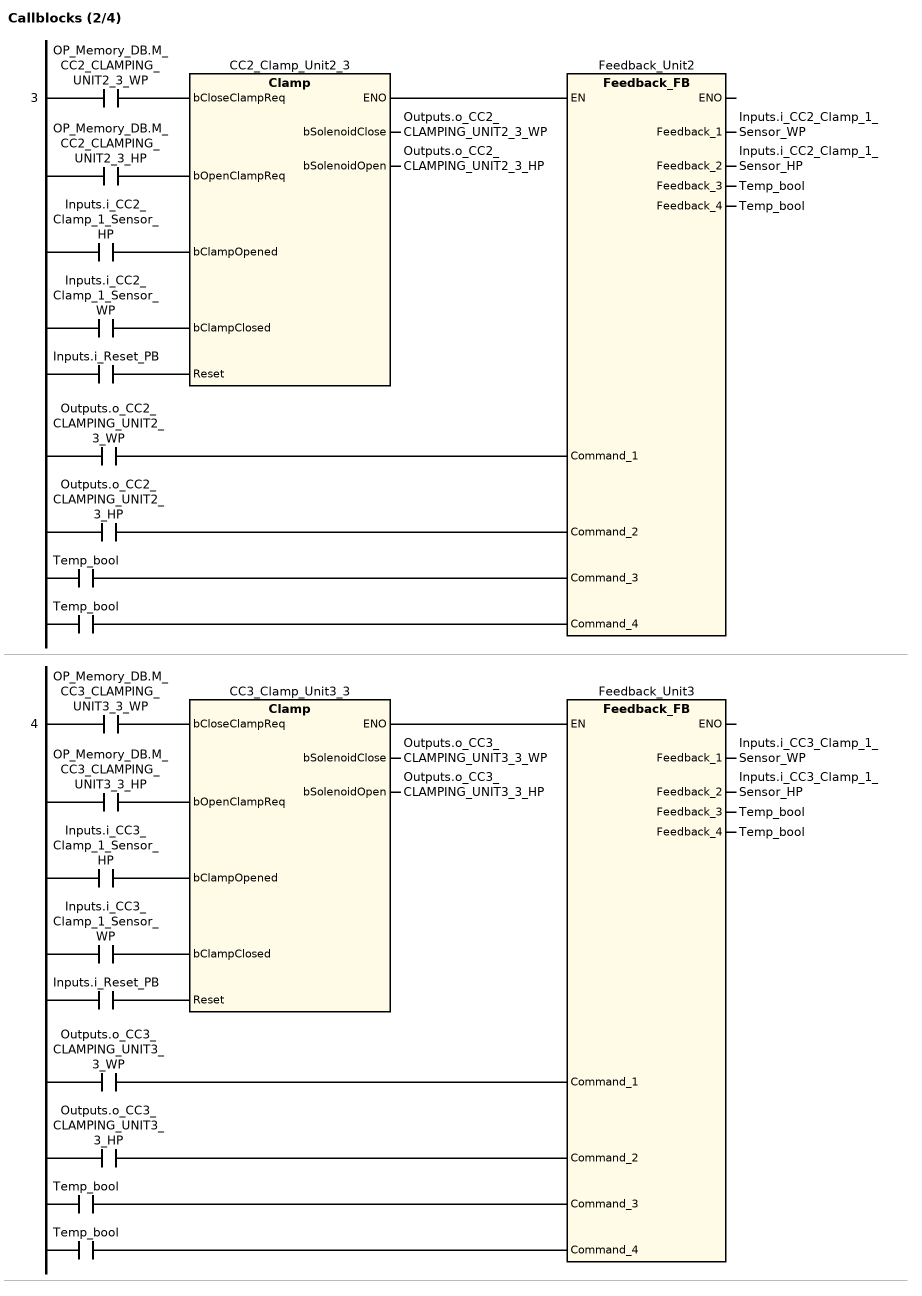
// NETWORK 3
CC2_Clamp_Unit2_3(
    bCloseClampReq := OP_Memory_DB.M_CC2_CLAMPING_UNIT2_3_WP,
    bOpenClampReq := OP_Memory_DB.M_CC2_CLAMPING_UNIT2_3_HP,
    bClampOpened := Inputs.i_CC2_Clamp_1_Sensor_HP,
    bClampClosed := Inputs.i_CC2_Clamp_1_Sensor_WP,
    Reset := Inputs.i_Reset_PB,
    bSolenoidClose => Outputs.o_CC2_CLAMPING_UNIT2_3_WP,
    bSolenoidOpen => Outputs.o_CC2_CLAMPING_UNIT2_3_HP); // Clamp
Feedback_Unit2(
    EN := TRUE,
    Command_1 := Outputs.o_CC2_CLAMPING_UNIT2_3_WP,
    Command_2 := Outputs.o_CC2_CLAMPING_UNIT2_3_HP,
    Command_3 := Temp_bool,
    Command_4 := Temp_bool,
    Feedback_1 => Inputs.i_CC2_Clamp_1_Sensor_WP,
    Feedback_2 => Inputs.i_CC2_Clamp_1_Sensor_HP,
    Feedback_3 => Temp_bool,
    Feedback_4 => Temp_bool); // Feedback_FB

// NETWORK 4
CC3_Clamp_Unit3_3(
    bCloseClampReq := OP_Memory_DB.M_CC3_CLAMPING_UNIT3_3_WP,
    bOpenClampReq := OP_Memory_DB.M_CC3_CLAMPING_UNIT3_3_HP,
    bClampOpened := Inputs.i_CC3_Clamp_1_Sensor_HP,
    bClampClosed := Inputs.i_CC3_Clamp_1_Sensor_WP,
    Reset := Inputs.i_Reset_PB,
    bSolenoidClose => Outputs.o_CC3_CLAMPING_UNIT3_3_WP,
    bSolenoidOpen => Outputs.o_CC3_CLAMPING_UNIT3_3_HP); // Clamp
Feedback_Unit3(
    EN := TRUE,
    Command_1 := Outputs.o_CC3_CLAMPING_UNIT3_3_WP,
    Command_2 := Outputs.o_CC3_CLAMPING_UNIT3_3_HP,
    Command_3 := Temp_bool,
    Command_4 := Temp_bool,
    Feedback_1 => Inputs.i_CC3_Clamp_1_Sensor_WP,
    Feedback_2 => Inputs.i_CC3_Clamp_1_Sensor_HP,
    Feedback_3 => Temp_bool,
    Feedback_4 => Temp_bool); // Feedback_FB

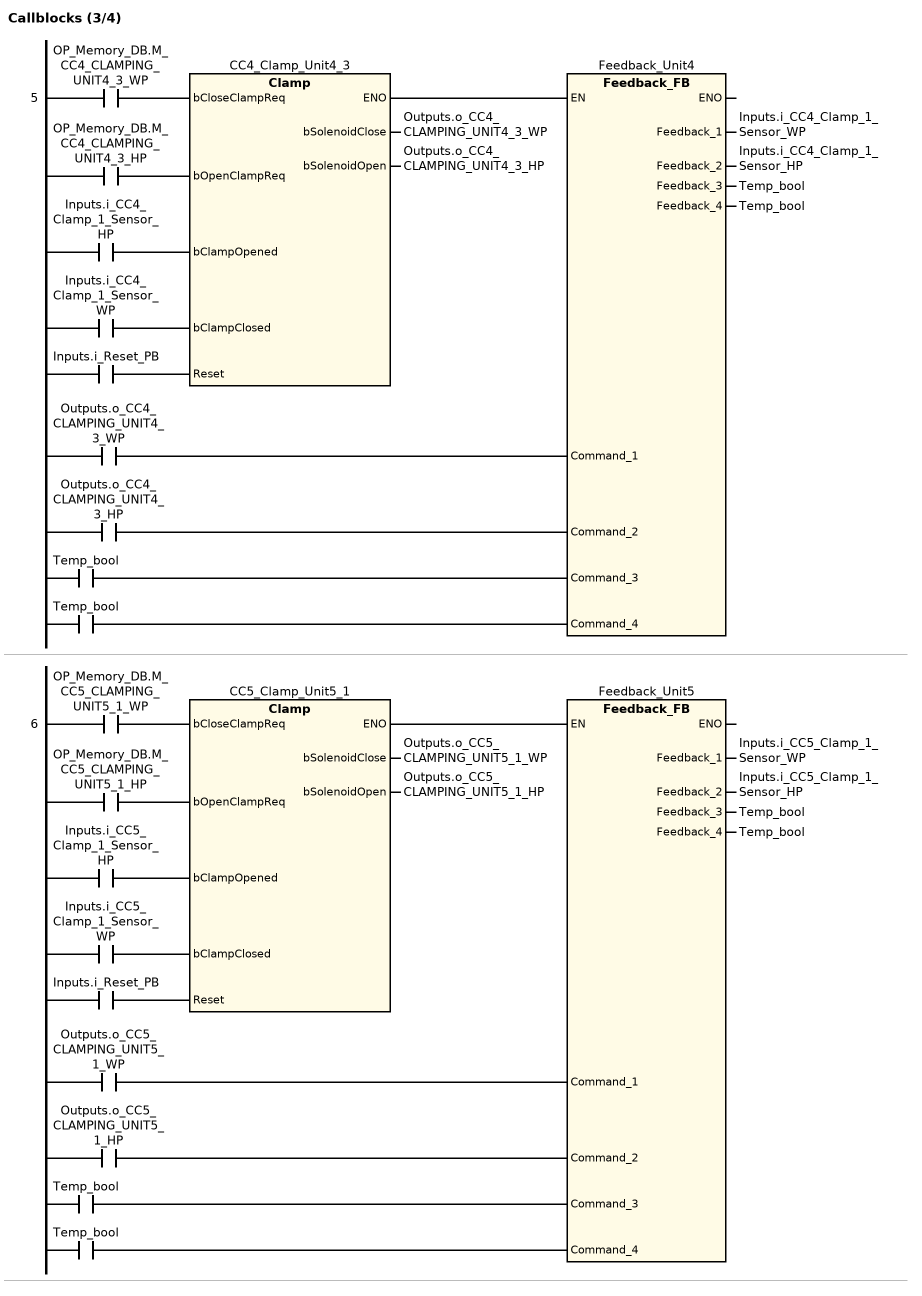
// NETWORK 5
CC4_Clamp_Unit4_3(
    bCloseClampReq := OP_Memory_DB.M_CC4_CLAMPING_UNIT4_3_WP,
    bOpenClampReq := OP_Memory_DB.M_CC4_CLAMPING_UNIT4_3_HP,
    bClampOpened := Inputs.i_CC4_Clamp_1_Sensor_HP,
    bClampClosed := Inputs.i_CC4_Clamp_1_Sensor_WP,
    Reset := Inputs.i_Reset_PB,
    bSolenoidClose => Outputs.o_CC4_CLAMPING_UNIT4_3_WP,
    bSolenoidOpen => Outputs.o_CC4_CLAMPING_UNIT4_3_HP); // Clamp
Feedback_Unit4(
    EN := TRUE,
    Command_1 := Outputs.o_CC4_CLAMPING_UNIT4_3_WP,
    Command_2 := Outputs.o_CC4_CLAMPING_UNIT4_3_HP,
    Command_3 := Temp_bool,
    Command_4 := Temp_bool,
    Feedback_1 => Inputs.i_CC4_Clamp_1_Sensor_WP,
    Feedback_2 => Inputs.i_CC4_Clamp_1_Sensor_HP,
    Feedback_3 => Temp_bool,
    Feedback_4 => Temp_bool); // Feedback_FB

// NETWORK 6
CC5_Clamp_Unit5_1(
    bCloseClampReq := OP_Memory_DB.M_CC5_CLAMPING_UNIT5_1_WP,
    bOpenClampReq := OP_Memory_DB.M_CC5_CLAMPING_UNIT5_1_HP,
    bClampOpened := Inputs.i_CC5_Clamp_1_Sensor_HP,
    bClampClosed := Inputs.i_CC5_Clamp_1_Sensor_WP,
    Reset := Inputs.i_Reset_PB,
    bSolenoidClose => Outputs.o_CC5_CLAMPING_UNIT5_1_WP,
    bSolenoidOpen => Outputs.o_CC5_CLAMPING_UNIT5_1_HP); // Clamp
Feedback_Unit5(
    EN := TRUE,
    Command_1 := Outputs.o_CC5_CLAMPING_UNIT5_1_WP,
    Command_2 := Outputs.o_CC5_CLAMPING_UNIT5_1_HP,
    Command_3 := Temp_bool,
    Command_4 := Temp_bool,
    Feedback_1 => Inputs.i_CC5_Clamp_1_Sensor_WP,
    Feedback_2 => Inputs.i_CC5_Clamp_1_Sensor_HP,
    Feedback_3 => Temp_bool,
    Feedback_4 => Temp_bool); // Feedback_FB

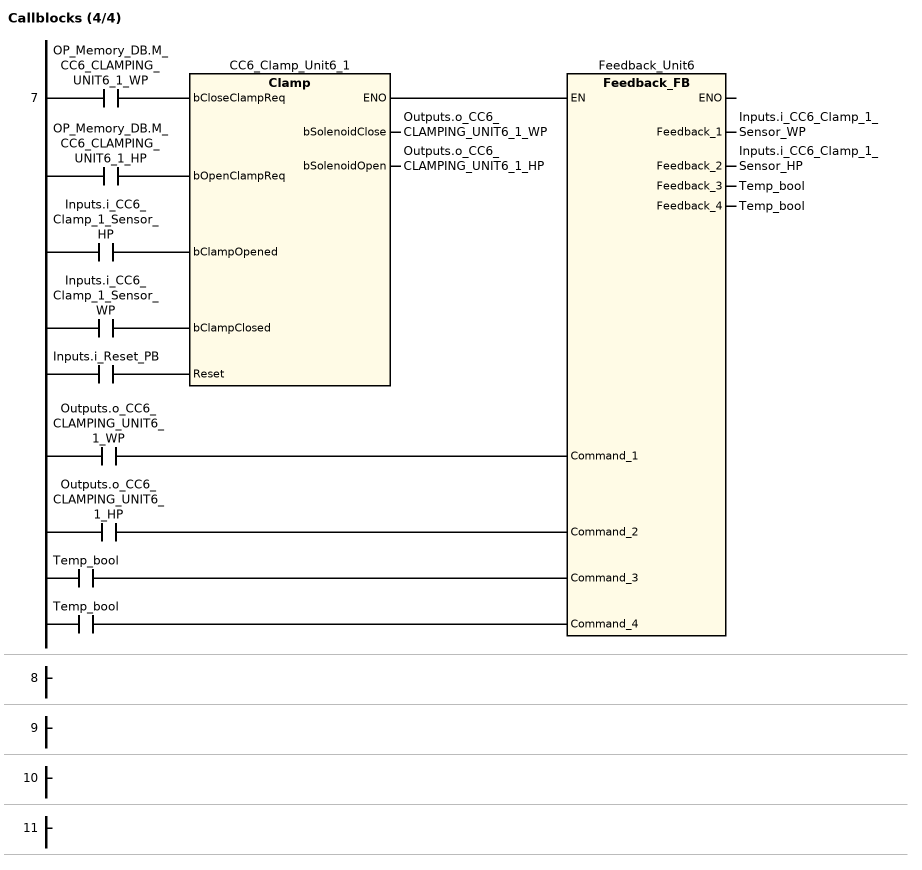
// NETWORK 7
CC6_Clamp_Unit6_1(
    bCloseClampReq := OP_Memory_DB.M_CC6_CLAMPING_UNIT6_1_WP,
    bOpenClampReq := OP_Memory_DB.M_CC6_CLAMPING_UNIT6_1_HP,
    bClampOpened := Inputs.i_CC6_Clamp_1_Sensor_HP,
    bClampClosed := Inputs.i_CC6_Clamp_1_Sensor_WP,
    Reset := Inputs.i_Reset_PB,
    bSolenoidClose => Outputs.o_CC6_CLAMPING_UNIT6_1_WP,
    bSolenoidOpen => Outputs.o_CC6_CLAMPING_UNIT6_1_HP); // Clamp
Feedback_Unit6(
    EN := TRUE,
    Command_1 := Outputs.o_CC6_CLAMPING_UNIT6_1_WP,
    Command_2 := Outputs.o_CC6_CLAMPING_UNIT6_1_HP,
    Command_3 := Temp_bool,
    Command_4 := Temp_bool,
    Feedback_1 => Inputs.i_CC6_Clamp_1_Sensor_WP,
    Feedback_2 => Inputs.i_CC6_Clamp_1_Sensor_HP,
    Feedback_3 => Temp_bool,
    Feedback_4 => Temp_bool); // Feedback_FB

// NETWORK 8

// NETWORK 9

// NETWORK 10

// NETWORK 11

END_PROGRAM

// ---- POUs/BIW/Clamp.TcPOU
FUNCTION_BLOCK PUBLIC Clamp
VAR_INPUT
	
    bCloseClampReq  : BOOL;     // Command to close (from HMI or Logic)
    bOpenClampReq   : BOOL;     // Command to open
    
    bClampOpened    : BOOL;     // Sensor: Clamp is fully back
    bClampClosed    : BOOL;     // Sensor: Clamp is fully forward/extended
	Reset		    : BOOL;
    
END_VAR
VAR_OUTPUT
	ENO             : BOOL;
    bSolenoidClose  : BOOL;     // Output to Valve (Close coil)
    bSolenoidOpen   : BOOL;     // Output to Valve (Open coil)	
	//Timeout 		: BOOL;

END_VAR
VAR
    nState          : INT;      // 0: Idle, 10: Closing, 20: Closed, 30: Opening
    fbTimeout       : TON;      // Watchdog timer for sensor failure
    sAlarm          : STRING;   // Error message
	
END_VAR

// Watchdog timer: If clamp doesn't reach sensor in 2 seconds, trigger error
fbTimeout(IN := (nState = 10 OR nState = 30), PT := T#2S);

CASE nState OF
    0: // IDLE / OPEN
        bSolenoidClose := FALSE;
        bSolenoidOpen  := TRUE; // Maintain open pressure
        IF bCloseClampReq AND NOT bOpenClampReq THEN
            nState := 10;
        END_IF

    10: // CLOSING
        bSolenoidOpen  := FALSE;
        bSolenoidClose := TRUE;
        
        IF bClampClosed THEN
            nState := 20;
        ELSIF fbTimeout.Q THEN
            sAlarm := 'Error: Clamp Close Timeout';
            nState := 99; // Error State
        END_IF

    20: // FULLY CLOSED
        bSolenoidClose := TRUE; // Maintain grip pressure
        IF bOpenClampReq THEN
            nState := 30;
        END_IF

    30: // OPENING
        bSolenoidClose := FALSE;
        bSolenoidOpen  := TRUE;
        
        IF bClampOpened THEN
            nState := 0;
        ELSIF fbTimeout.Q THEN
            sAlarm := 'Error: Clamp Open Timeout';
            nState := 99;
        END_IF

    99: // ERROR STATE
        bSolenoidClose := FALSE;
        bSolenoidOpen  := FALSE; // De-energize for safety
        IF NOT bCloseClampReq AND NOT bOpenClampReq THEN
            nState := 0; // Reset after clearing request
        END_IF
END_CASE

IF reset THEN
	nState := 0; // Reset after clearing request
	sAlarm := '';
	END_IF;

END_FUNCTION_BLOCK

// ---- POUs/BIW/Turntable.TcPOU
FUNCTION_BLOCK PUBLIC Turntable
VAR_INPUT
  
    bStartCW        : BOOL;     // Command: Move Clockwise
    bStartCCW       : BOOL;     // Command: Move Counter-Clockwise
    bPosSensor      : BOOL;     // Index sensor (detects the 4 positions)
     
  
END_VAR
VAR_OUTPUT
    ENO             : BOOL;
    bMotorRun       : BOOL;     // Output to Drive: Run
    bMotorDir       : BOOL;     // Output to Drive: FALSE = FWD, TRUE = REV
      
    
END_VAR
VAR

    nState          : INT := 0; 
    nCurrentPos     : INT := 1; // 1, 2, 3, 4
    fbTrigSensor    : R_TRIG;   		 

END_VAR

fbTrigSensor(CLK := bPosSensor);

CASE nState OF
    0: // IDLE
        bMotorRun := FALSE;
        
        IF bStartCW THEN
            bMotorDir := FALSE; // Forward
            nState    := 10;
        ELSIF bStartCCW THEN
            bMotorDir := TRUE;  // Reverse
            nState    := 10;
        END_IF
        
    10: // START MOVING (Clear current sensor)
        bMotorRun := TRUE;
        IF NOT bPosSensor THEN 
            nState := 20;
        END_IF
        
    20: // MONITOR SENSOR & UPDATE POSITION
        IF fbTrigSensor.Q THEN
            // Update position based on direction
            IF NOT bMotorDir THEN // CW Logic
                nCurrentPos := nCurrentPos + 1;
                IF nCurrentPos > 4 THEN nCurrentPos := 1; END_IF;
            ELSE // CCW Logic
                nCurrentPos := nCurrentPos - 1;
                IF nCurrentPos < 1 THEN nCurrentPos := 4; END_IF;
            END_IF
            
            nState := 30;
        END_IF
        
    30: // STOPPING
        bMotorRun := FALSE;
        // Wait for buttons to be released before allowing next move
        IF NOT bStartCW AND NOT bStartCCW THEN
            nState := 0;
        END_IF
END_CASE

END_FUNCTION_BLOCK

// ---- POUs/BIW/WeldRobot.TcPOU
FUNCTION_BLOCK PUBLIC WeldRobot
VAR_INPUT
	
	// Inputs from Robot (to PLC)
    bRobotInHome      : BOOL;    // Robot is at safe perch
    bRobotBusy        : BOOL;    // Robot is currently welding
    bRobotFinished    : BOOL;    // Robot completed the weld cycle
      
END_VAR
VAR_OUTPUT
	
	// Outputs to Robot (from PLC)
	ENO               : BOOL;
    bStartWeld        : BOOL;    // Signal to Robot to start its internal program
    nJobNumber        : INT;     // Tells robot which weld path to use (1-4 for our table)

END_VAR
VAR

// Cell Status (Internal)
    bPartReady        : BOOL;    // From our "Part Present & Clamped" logic
    nState            : INT;     
    fbTimeout         : TON;     // Safety watchdog	

END_VAR

CASE nState OF
    0: // IDLE - Wait for Part and Robot Home
        bStartWeld := FALSE;
        IF bPartReady AND bRobotInHome THEN
            nState := 10;
        END_IF
        
    10: // PREPARE - Set Job Number for the current table station
        nJobNumber := 1; // Example: Station 1
        nState     := 20;
        
    20: // START ROBOT
        IF bRobotInHome THEN
            bStartWeld := TRUE; // Pulse the start signal
            nState     := 30;
        END_IF
        
    30: // WAIT FOR ACKNOWLEDGEMENT
        IF bRobotBusy THEN
            bStartWeld := FALSE; // Turn off start signal once robot moves
            nState     := 40;
        END_IF
        
    40: // MONITOR WELDING
        // Watchdog: If robot stays busy for > 60s, something is wrong
        fbTimeout(IN := bRobotBusy, PT := T#60S);
        
        IF bRobotFinished THEN
            nState := 50;
        ELSIF fbTimeout.Q THEN
            nState := 99; // Error: Robot Stuck
        END_IF
        
    50: // CYCLE COMPLETE
        IF NOT bRobotFinished THEN // Wait for robot to reset its finish signal
            nState := 0;
        END_IF
        
    99: // ERROR STATE
        bStartWeld := FALSE;
END_CASE

END_FUNCTION_BLOCK

// ---- POUs/BIW/MHRobot.TcPOU
FUNCTION_BLOCK PUBLIC MHRobot
VAR_INPUT
	// Inputs from Robot
    bRobotInHome      : BOOL;    // Safe position
    bRobotHasPart     : BOOL;    // Gripper sensor status (from Robot)
    bRobotAtPick      : BOOL;    // Robot is positioned at the pick station
    bRobotAtDrop      : BOOL;    // Robot is positioned at the drop station
    
END_VAR
VAR_OUTPUT
	 // Outputs to Robot
	 ENO              : BOOL;
    bEnablePick       : BOOL;    // OK to enter Pick Zone and grab
    bEnableDrop       : BOOL;    // OK to enter Drop Zone and release

END_VAR
VAR
	// Cell Logic
    bPickStationReady : BOOL;    // e.g., Turntable is indexed and Part Present
    bDropStationEmpty : BOOL;    // e.g., Outfeed conveyor is clear
    nState            : INT;

END_VAR

CASE nState OF
    0: // IDLE - Evaluate next move
        bEnablePick := FALSE;
        bEnableDrop := FALSE;
        
        IF bRobotInHome AND bPickStationReady AND NOT bRobotHasPart THEN
            nState := 10; // Go Pick
        ELSIF bRobotInHome AND bDropStationEmpty AND bRobotHasPart THEN
            nState := 20; // Go Drop
        END_IF

    10: // PICK SEQUENCE
        bEnablePick := TRUE;
        // Wait until robot confirms it has grabbed the part and left the zone
        IF bRobotHasPart AND bRobotInHome THEN
            bEnablePick := FALSE;
            nState := 0;
        END_IF

    20: // DROP SEQUENCE
        bEnableDrop := TRUE;
        // Wait until robot confirms it has released the part and left the zone
        IF NOT bRobotHasPart AND bRobotInHome THEN
            bEnableDrop := FALSE;
            nState := 0;
        END_IF
END_CASE

END_FUNCTION_BLOCK

// ---- POUs/BIW/Fixture.TcPOU
PROGRAM Fixture
VAR
	
    bPartPresent1   : BOOL;     // Sensor 1 
    bPartPresent2   : BOOL;     // Sensor 2 
    bOperatorClear  : BOOL;     // Light curtain or "Load Complete" button
    

    bPartIsLoaded   : BOOL;     // Status for other POUs
    fbPartDebounce  : TON;      // Filters shaky sensor signals
    nStep           : INT;      // Load sequence tracking
    sLoadStatus     : STRING;   // Operator feedback

END_VAR

// 1. Debounce Sensors: Part must be stable for 0.5s to be "Present"
fbPartDebounce(IN := (bPartPresent1 AND bPartPresent2), PT := T#500MS);

CASE nStep OF
    0: // WAIT FOR LOAD
        bPartIsLoaded := FALSE;
        sLoadStatus   := 'Waiting for operator to load part...';
        
        IF fbPartDebounce.Q THEN
            nStep := 10;
        END_IF
        
    10: // PART DETECTED - WAIT FOR OPERATOR CLEARANCE
        sLoadStatus := 'Part detected. Confirm clear (Light Curtain/Button).';
        
        // Ensure operator is clear and part is still there
        IF bOperatorClear AND fbPartDebounce.Q THEN
            bPartIsLoaded := TRUE;
            sLoadStatus   := 'Ready to Clamp';
            // Transition to Clamping Logic here
        ELSIF NOT fbPartDebounce.Q THEN
            nStep := 0; // Part was removed
        END_IF
        
    // Reset after station cycle completes
    100: 
        bPartIsLoaded := FALSE;
        nStep := 0;
END_CASE

END_PROGRAM

// ---- GlobalTextList.TcGTLO
TEXTLIST GlobalTextList
  864 = '-20*'
  71 = '0*'
  264 = '180*'
  59 = 'ALARM'
  942 = 'AUTO / MAN'
  853 = 'BUSY'
  686 = 'CLAMP_1_HOME'
  638 = 'CLAMP_1_WORK'
  203 = 'CLAMP_2_HOME'
  914 = 'CLAMP_2_WORK'
  734 = 'CLAMP_3_HOME'
  770 = 'CLAMP_3_WORK'
  279 = 'CLAMP_4_HOME'
  508 = 'CLAMP_4_WORK'
  856 = 'CLAMP_5_HOME'
  852 = 'CLAMP_5_WORK'
  25 = 'CLAMP_6_HOME'
  108 = 'CLAMP_6_WORK'
  552 = 'CLOSE'
  153 = 'CONTROL ON'
  909 = 'CYCLE START'
  312 = 'FIX_1'
  949 = 'FIX_2'
  854 = 'HOME'
  869 = 'HOME cmd'
  2 = 'MH_ROBOT'
  12 = 'OPEN'
  527 = 'OPERATOR'
  792 = 'OP_Memory_DB.A_FIX1_PART_2ND'
  905 = 'OP_Memory_DB.A_FIX1_PD'
  785 = 'POWER ON'
  218 = 'RESET'
  553 = 'RLD_CLS'
  657 = 'RLD_OPN'
  972 = 'ROLLER DOOR'
  988 = 'Safety ok'
  324 = 'SAFETY_OK'
  258 = 'SENSOR'
  928 = 'SENSOR1'
  950 = 'SENSOR2'
  163 = 'SENSOR3'
  838 = 'SENSOR4'
  858 = 'START'
  486 = 'Trn_FWD'
  780 = 'Trn_REV'
  503 = 'TRUNION'
  295 = 'TT_FWD'
  229 = 'TT_REV'
  67 = 'TURN TABLE'
  308 = 'WELD_ROBOT'
  135 = 'WORK '
  438 = 'work cmd'
  653 = 'WORK cmd '
  49 = 'WORK cmd cmd'
END_TEXTLIST

// ---- POUs/FiX_1.TcTLO
TEXTLIST FiX_1
  0 = 'CYCLE START'
  10 = 'RD_CLOSE'
  20 = 'TRUNION ROTATES -20*'
  30 = 'RD OPEN'
  40 = 'OPERATOR LOAD 1ST PART'
  50 = 'OPERATOR LOAD 2ND PART'
  60 = 'Clamp Close_1ST,3RD,5TH'
  70 = 'RD_CLOSE'
  80 = 'TRUNION ROTATES -80*'
  90 = 'RD OPEN'
  100 = ' Operator Load_3RD_PART'
  110 = ' Operator Load_4TH_PART'
  120 = 'RD_CLOSE'
  130 = ' CLAMP CLOSE 2ND,4TH, 6TH'
  140 = 'TURNTABLE-180* AND TRUNION_0*'
  150 = 'Start WELD_Robot FOR WELD'
  160 = 'CLAMP OPEN 1ST,3RD,5TH'
  170 = 'RD OPEN'
  180 = 'Start MH_Robot_1ST TIME'
  190 = 'TRUNION ROTATES -45*'
  200 = 'UNCLAMP 2ND, 4TH,6TH'
  210 = 'Start MH_Robot_2ND TIME'
  220 = 'CYCLE COMPLETE'
   = ''
END_TEXTLIST

// ---- VISUs/AUTO_PROCESS.TcVIS
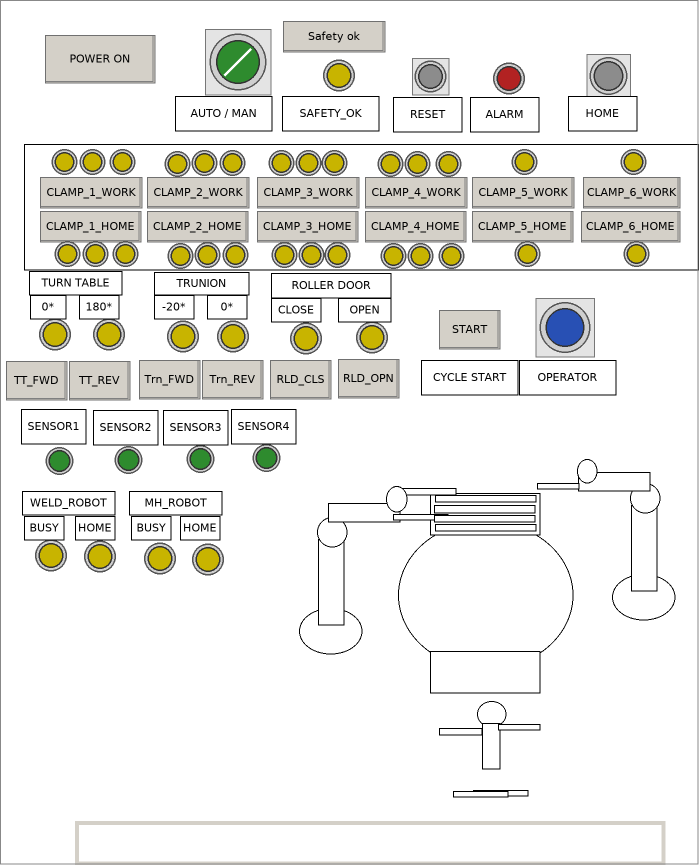
VISUALIZATION AUTO_PROCESS  // 699x865
    Rectangle (24,144 675x126)
    Lamp1 (314,57 50x37), variable: OP_Memory_DB.SAFETY_OK, style: Lamp-Lamp1-Yellow
    RotarySwitch (205,23 66x78), variable: OP_Memory_DB.Auto_mode, behaviour: TOGGLE, style: Switch-RotarySwitch-Green
    Rectangle (175,96 97x35), "AUTO / MAN"
    Rectangle (393,97 69x35), "RESET"
    Button (45,35 110x48), "POWER ON", colour toggle: OP_Memory_DB.POWER_ON
        toggle OP_Memory_DB.POWER_ON
    Button (40,177 102x31), "CLAMP_1_WORK", colour toggle: OP_Memory_DB.M_CC1_CLAMPING_UNIT1_3_WP
        toggle OP_Memory_DB.M_CC1_CLAMPING_UNIT1_3_WP
    Button (40,211 101x31), "CLAMP_1_HOME", colour toggle: OP_Memory_DB.M_CC1_CLAMPING_UNIT1_3_HP
        toggle OP_Memory_DB.M_CC1_CLAMPING_UNIT1_3_HP
    Button (583,177 97x31), "CLAMP_6_WORK", colour toggle: OP_Memory_DB.M_CC6_CLAMPING_UNIT6_1_WP
        toggle OP_Memory_DB.M_CC6_CLAMPING_UNIT6_1_WP
    Button (472,177 102x31), "CLAMP_5_WORK", colour toggle: OP_Memory_DB.M_CC5_CLAMPING_UNIT5_1_WP
        toggle OP_Memory_DB.M_CC5_CLAMPING_UNIT5_1_WP
    Button (472,211 101x31), "CLAMP_5_HOME", colour toggle: OP_Memory_DB.M_CC5_CLAMPING_UNIT5_1_HP
        toggle OP_Memory_DB.M_CC5_CLAMPING_UNIT5_1_HP
    Button (581,211 99x31), "CLAMP_6_HOME", colour toggle: OP_Memory_DB.M_CC6_CLAMPING_UNIT6_1_HP
        toggle OP_Memory_DB.M_CC6_CLAMPING_UNIT6_1_HP
    Rectangle (29,271 93x24), "TURN TABLE"
    Rectangle (154,272 95x23), "TRUNION"
    Rectangle (271,273 120x25), "ROLLER DOOR"
    Lamp1 (30,316 50x37), variable: Inputs.i_1st_TT_Pos, style: Lamp-Lamp1-Yellow
    Lamp1 (84,316 50x37), variable: Inputs.i_2nd_TT_Pos, style: Lamp-Lamp1-Yellow
    Lamp1 (158,318 50x37), variable: Inputs.i_Trunion_1st_Pos, style: Lamp-Lamp1-Yellow
    Lamp1 (208,318 50x37), variable: Inputs.i_Trunion_2nd_Pos, style: Lamp-Lamp1-Yellow
    Lamp1 (281,320 50x37), variable: Inputs.i_ROLL_DR_Close_Pos_LS, style: Lamp-Lamp1-Yellow
    Lamp1 (347,319 50x37), variable: Inputs.i_ROLL_DR_Open_Pos_LS, style: Lamp-Lamp1-Yellow
    Button (147,177 102x31), "CLAMP_2_WORK", colour toggle: OP_Memory_DB.M_CC2_CLAMPING_UNIT2_3_WP
        toggle OP_Memory_DB.M_CC2_CLAMPING_UNIT2_3_WP
    Button (147,211 101x31), "CLAMP_2_HOME", colour toggle: OP_Memory_DB.M_CC2_CLAMPING_UNIT2_3_HP
        toggle OP_Memory_DB.M_CC2_CLAMPING_UNIT2_3_HP
    Button (257,177 102x31), "CLAMP_3_WORK", colour toggle: OP_Memory_DB.M_CC3_CLAMPING_UNIT3_3_WP
        toggle OP_Memory_DB.M_CC3_CLAMPING_UNIT3_3_WP
    Button (257,211 101x31), "CLAMP_3_HOME", colour toggle: OP_Memory_DB.M_CC3_CLAMPING_UNIT3_3_HP
        toggle OP_Memory_DB.M_CC3_CLAMPING_UNIT3_3_HP
    Button (365,177 102x31), "CLAMP_4_WORK", colour toggle: OP_Memory_DB.M_CC4_CLAMPING_UNIT4_3_WP
        toggle OP_Memory_DB.M_CC4_CLAMPING_UNIT4_3_WP
    Button (365,211 101x31), "CLAMP_4_HOME", colour toggle: OP_Memory_DB.M_CC4_CLAMPING_UNIT4_3_HP
        toggle OP_Memory_DB.M_CC4_CLAMPING_UNIT4_3_HP
    Rectangle (30,295 36x24), "0*"
    Rectangle (79,295 40x24), "180*"
    Rectangle (154,295 40x24), "-20*"
    Rectangle (207,295 40x24), "0*"
    Rectangle (271,298 50x24), "CLOSE"
    Rectangle (338,298 53x24), "OPEN"
    Button (6,361 61x39), "TT_FWD", colour toggle: OP_Memory_DB.M_2ND_POSITION_TT_CMD
        tap OP_Memory_DB.M_2ND_POSITION_TT_CMD
    Button (69,361 61x39), "TT_REV", colour toggle: OP_Memory_DB.M_1ST_POSITION_TT_CMD
        tap OP_Memory_DB.M_1ST_POSITION_TT_CMD
    Button (139,360 61x39), "Trn_FWD", colour toggle: OP_Memory_DB.M_Fwd_POSITION
        tap OP_Memory_DB.M_Fwd_POSITION
    Button (202,360 61x39), "Trn_REV", colour toggle: OP_Memory_DB.M_Rev_POSITION
        tap OP_Memory_DB.M_Rev_POSITION
    Button (338,359 61x39), "RLD_OPN", colour toggle: OP_Memory_DB.M_Roll_Dr_Open
        tap OP_Memory_DB.M_Roll_Dr_Open
    Button (270,360 61x39), "RLD_CLS", colour toggle: OP_Memory_DB.M_Roll_Dr_Close
        tap OP_Memory_DB.M_Roll_Dr_Close
    PushSwitch (535,298 60x59), variable: Inputs.i_OPERATE_START_PB, behaviour: TAP, style: Switch-PushSwitch-Blue
    Rectangle (519,360 97x35), "OPERATOR"
    Rectangle (21,409 65x35), "SENSOR1"
    Lamp1 (178,443 45x32), variable: Inputs.i_PART_CONTROL_B8, style: Lamp-Lamp1-Green
    Lamp1 (247,442 39x32), variable: Inputs.i_PART_CONTROL_B22, style: Lamp-Lamp1-Green
    Rectangle (93,410 65x35), "SENSOR2"
    Rectangle (163,410 65x35), "SENSOR3"
    Rectangle (231,409 65x35), "SENSOR4"
    Lamp1 (37,445 45x32), variable: Inputs.i_PART_CONTROL_B1, style: Lamp-Lamp1-Green
    Lamp1 (106,444 45x32), variable: Inputs.i_PART_CONTROL_B15, style: Lamp-Lamp1-Green
    Ellipse (398,521 175x148)
    Rectangle (430,493 110x42)
    Rectangle (430,651 110x42)
    Ellipse (612,574 63x46)
    Rectangle (631,505 26x86)
    Ellipse (630,483 30x30)
    Rectangle (578,472 72x19), angle 26
    Rectangle (537,483 42x6), angle 337, colour toggle: OP_Memory_DB.ROBOT_BUSY
    Ellipse (299,608 63x46)
    Rectangle (318,539 26x86)
    Ellipse (317,517 30x30)
    Rectangle (328,503 72x19), angle 335
    Rectangle (399,488 57x7), angle 349, colour toggle: OP_Memory_DB.MH_ROBOT_BUSY
    Rectangle (393,514 55x6), angle 54, colour toggle: OP_Memory_DB.MH_ROBOT_BUSY
    Ellipse (577,459 20x24)
    Ellipse (386,486 21x26)
    Ellipse (477,701 29x26)
    Rectangle (482,723 18x46)
    Rectangle (498,724 42x6), angle 337, colour toggle: Inputs.i_OPERATE_START_PB
    Rectangle (473,790 55x6), angle 69
    Rectangle (453,791 55x6), angle 111
    Rectangle (439,728 43x7), angle 9, colour toggle: Inputs.i_OPERATE_START_PB
    Lamp1 (45,147 39x30), variable: Inputs.i_CC1_Clamp_1_Sensor_WP, style: Lamp-Lamp1-Yellow
    PushSwitch (409,58 43x37), variable: Inputs.i_Reset_PB, behaviour: TAP, style: Switch-PushSwitch-Gray
    Rectangle (282,96 97x35), "SAFETY_OK"
    Lamp1 (484,60 50x37), variable: Outputs.O_FAULT_LAMP, style: Lamp-Lamp1-Red
    Rectangle (470,97 69x35), "ALARM"
    Lamp1 (158,149 39x30), variable: Inputs.i_CC2_Clamp_1_Sensor_WP, style: Lamp-Lamp1-Yellow
    Lamp1 (262,148 39x30), variable: Inputs.i_CC3_Clamp_1_Sensor_WP, style: Lamp-Lamp1-Yellow
    Lamp1 (371,149 39x30), variable: Inputs.i_CC4_Clamp_1_Sensor_WP, style: Lamp-Lamp1-Yellow
    Lamp1 (505,147 39x30), variable: Inputs.i_CC5_Clamp_1_Sensor_WP, style: Lamp-Lamp1-Yellow
    Lamp1 (614,147 39x30), variable: Inputs.i_CC6_Clamp_1_Sensor_WP, style: Lamp-Lamp1-Yellow
    PushSwitch (580,54 57x44), variable: OP_Memory_DB.M_FIX1_ALL_CLAMP_HOME_PB, behaviour: TAP, style: Switch-PushSwitch-Gray
    Rectangle (568,96 69x35), "HOME"
    Lamp1 (73,147 39x30), variable: Inputs.i_CC1_Clamp_2_Sensor_WP, style: Lamp-Lamp1-Yellow
    Lamp1 (103,147 39x30), variable: Inputs.i_CC1_Clamp_3_Sensor_WP, style: Lamp-Lamp1-Yellow
    Lamp1 (185,148 39x30), variable: Inputs.i_CC2_Clamp_2_Sensor_WP, style: Lamp-Lamp1-Yellow
    Lamp1 (213,148 39x30), variable: Inputs.i_CC2_Clamp_3_Sensor_WP, style: Lamp-Lamp1-Yellow
    Lamp1 (289,148 39x30), variable: Inputs.i_CC3_Clamp_2_Sensor_WP, style: Lamp-Lamp1-Yellow
    Lamp1 (315,148 39x30), variable: Inputs.i_CC3_Clamp_3_Sensor_WP, style: Lamp-Lamp1-Yellow
    Lamp1 (398,149 39x30), variable: Inputs.i_CC4_Clamp_2_Sensor_WP, style: Lamp-Lamp1-Yellow
    Lamp1 (429,149 39x30), variable: Inputs.i_CC4_Clamp_3_Sensor_WP, style: Lamp-Lamp1-Yellow
    Button (283,21 102x31), "Safety ok", colour toggle: OP_Memory_DB.SAFETY_OK
        toggle OP_Memory_DB.SAFETY_OK
    Rectangle (421,360 97x35), "CYCLE START"
    Lamp1 (48,239 39x30), variable: Inputs.i_CC1_Clamp_1_Sensor_HP, style: Lamp-Lamp1-Yellow
    Lamp1 (161,241 39x30), variable: Inputs.i_CC2_Clamp_1_Sensor_HP, style: Lamp-Lamp1-Yellow
    Lamp1 (265,240 39x30), variable: Inputs.i_CC3_Clamp_1_Sensor_HP, style: Lamp-Lamp1-Yellow
    Lamp1 (374,241 39x30), variable: Inputs.i_CC4_Clamp_1_Sensor_HP, style: Lamp-Lamp1-Yellow
    Lamp1 (508,239 39x30), variable: Inputs.i_CC5_Clamp_1_Sensor_HP, style: Lamp-Lamp1-Yellow
    Lamp1 (617,239 39x30), variable: Inputs.i_CC6_Clamp_1_Sensor_HP, style: Lamp-Lamp1-Yellow
    Lamp1 (76,239 39x30), variable: Inputs.i_CC1_Clamp_2_Sensor_HP, style: Lamp-Lamp1-Yellow
    Lamp1 (106,239 39x30), variable: Inputs.i_CC1_Clamp_3_Sensor_HP, style: Lamp-Lamp1-Yellow
    Lamp1 (188,240 39x30), variable: Inputs.i_CC2_Clamp_2_Sensor_HP, style: Lamp-Lamp1-Yellow
    Lamp1 (216,240 39x30), variable: Inputs.i_CC2_Clamp_3_Sensor_HP, style: Lamp-Lamp1-Yellow
    Lamp1 (292,240 39x30), variable: Inputs.i_CC3_Clamp_2_Sensor_HP, style: Lamp-Lamp1-Yellow
    Lamp1 (318,240 39x30), variable: Inputs.i_CC3_Clamp_3_Sensor_HP, style: Lamp-Lamp1-Yellow
    Lamp1 (401,241 39x30), variable: Inputs.i_CC4_Clamp_2_Sensor_HP, style: Lamp-Lamp1-Yellow
    Lamp1 (432,241 39x30), variable: Inputs.i_CC4_Clamp_3_Sensor_HP, style: Lamp-Lamp1-Yellow
    Button (439,310 61x39), "START", colour toggle: Inputs.i_CYCLE_START_PB
        tap Inputs.i_CYCLE_START_PB
    Rectangle (22,491 93x24), "WELD_ROBOT"
    Lamp1 (135,540 50x37), variable: OP_Memory_DB.MH_ROBOT_BUSY, style: Lamp-Lamp1-Yellow
    Lamp1 (183,541 50x37), variable: OP_Memory_DB.MH_ROBOT_HOME, style: Lamp-Lamp1-Yellow
    Rectangle (129,491 93x24), "MH_ROBOT"
    Lamp1 (26,537 50x37), variable: OP_Memory_DB.ROBOT_BUSY, style: Lamp-Lamp1-Yellow
    Lamp1 (75,538 50x37), variable: OP_Memory_DB.ROBOT_HOME, style: Lamp-Lamp1-Yellow
    Rectangle (24,516 40x24), "BUSY"
    Rectangle (75,516 40x24), "HOME"
    Rectangle (131,516 40x24), "BUSY"
    Rectangle (180,516 40x24), "HOME"
    Textfield (75,821 590x44), text list: 'FiX_1', text index: BLOCK_CALL.MODE_CONTROL_DB.Step
    Rectangle (435,495 101x7), colour toggle: Inputs.i_PART_CONTROL_B1
    Rectangle (434,505 101x8), colour toggle: Inputs.i_PART_CONTROL_B15
    Rectangle (434,515 101x7), colour toggle: Inputs.i_PART_CONTROL_B8
    Rectangle (435,524 101x7), colour toggle: Inputs.i_PART_CONTROL_B22
END_VISUALIZATION

// ---- VISUs/Visualization.TcVIS
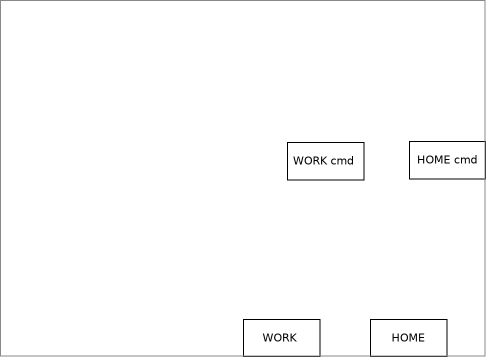
VISUALIZATION Visualization  // 486x357
    Rectangle (287,142 77x38), "WORK cmd"
    Rectangle (409,141 77x38), "HOME cmd"
    Rectangle (243,319 77x38), "WORK"
    Rectangle (370,319 77x38), "HOME"
END_VISUALIZATION
